REGION Network 17: IMMEDIATE STOP ALARMS / IMMEDIATE STOP
   RUNG wire#powerrail
      I_Contact( #CH_NOT_IN_SOFT_MODE )
      Not()
      { S7_GenerateENO := "TRUE" } Move(in := #DB_NUMBER, out1 => "DB440_MACHINE_ALARM_DECODING".GLOBAL_ALARMS_MACHINE.ALARM_DECODING)
      wire#w1
      { S7_Templates := "SrcType := Int" } EQ_Contact(in1 := #CHANNEL_NUM, in2 := 1)
      S_Coil( "DB440_MACHINE_ALARM_DECODING".ALARMS_UNIT_01.ST0_TRANSFER.IS_SEOC_ALARMS )
   END_RUNG
   RUNG wire#w1
      { S7_Templates := "SrcType := Int" } EQ_Contact(in1 := #CHANNEL_NUM, in2 := 2)
      S_Coil( "DB440_MACHINE_ALARM_DECODING".ALARMS_UNIT_01.ST3_CLADDING.IS_SEOC_ALARMS )
   END_RUNG
   RUNG wire#w1
      { S7_Templates := "SrcType := Int" } EQ_Contact(in1 := #CHANNEL_NUM, in2 := 3)
      S_Coil( "DB440_MACHINE_ALARM_DECODING".ALARMS_UNIT_01.ST4_CLEANING.IS_SEOC_ALARMS )
   END_RUNG
   RUNG wire#w1
      { S7_Templates := "SrcType := Int" } EQ_Contact(in1 := #CHANNEL_NUM, in2 := 4)
      S_Coil( "DB440_MACHINE_ALARM_DECODING".ALARMS_UNIT_02.ST0_TRANSFER.IS_SEOC_ALARMS )
   END_RUNG
   RUNG wire#w1
      { S7_Templates := "SrcType := Int" } EQ_Contact(in1 := #CHANNEL_NUM, in2 := 5)
      S_Coil( "DB440_MACHINE_ALARM_DECODING".ALARMS_UNIT_02.ST2_MEASURING.IS_SEOC_ALARMS )
   END_RUNG
   RUNG wire#w1
      { S7_Templates := "SrcType := Int" } EQ_Contact(in1 := #CHANNEL_NUM, in2 := 6)
      S_Coil( "DB440_MACHINE_ALARM_DECODING".ALARMS_UNIT_02.ST3_CLADDING.IS_SEOC_ALARMS )
   END_RUNG
   RUNG wire#w1
      { S7_Templates := "SrcType := Int" } EQ_Contact(in1 := #CHANNEL_NUM, in2 := 7)
      S_Coil( "DB440_MACHINE_ALARM_DECODING".ALARMS_UNIT_02.ST4_CLEANING.IS_SEOC_ALARMS )
   END_RUNG
   RUNG wire#w1
      { S7_Templates := "SrcType := Int" } EQ_Contact(in1 := #CHANNEL_NUM, in2 := 8)
      S_Coil( "DB440_MACHINE_ALARM_DECODING".ALARMS_UNIT_03.IS_SEOC_ALARMS )
   END_RUNG
   RUNG wire#w1
      { S7_Templates := "SrcType := Int" } EQ_Contact(in1 := #CHANNEL_NUM, in2 := 9)
      S_Coil( "DB440_MACHINE_ALARM_DECODING".ALARMS_UNIT_04.IS_SEOC_ALARMS )
   END_RUNG
   // the same network as SCL:
   // ENO of a box is taken as its EN; it also drops when the box reports an error
   #_w1 := NOT (NOT #CH_NOT_IN_SOFT_MODE);
   IF #_w1 THEN "DB440_MACHINE_ALARM_DECODING".GLOBAL_ALARMS_MACHINE.ALARM_DECODING := #DB_NUMBER; END_IF;
   IF #_w1 AND (#CHANNEL_NUM = 1) THEN
       "DB440_MACHINE_ALARM_DECODING".ALARMS_UNIT_01.ST0_TRANSFER.IS_SEOC_ALARMS := TRUE;
   END_IF;
   IF #_w1 AND (#CHANNEL_NUM = 2) THEN
       "DB440_MACHINE_ALARM_DECODING".ALARMS_UNIT_01.ST3_CLADDING.IS_SEOC_ALARMS := TRUE;
   END_IF;
   IF #_w1 AND (#CHANNEL_NUM = 3) THEN
       "DB440_MACHINE_ALARM_DECODING".ALARMS_UNIT_01.ST4_CLEANING.IS_SEOC_ALARMS := TRUE;
   END_IF;
   IF #_w1 AND (#CHANNEL_NUM = 4) THEN
       "DB440_MACHINE_ALARM_DECODING".ALARMS_UNIT_02.ST0_TRANSFER.IS_SEOC_ALARMS := TRUE;
   END_IF;
   IF #_w1 AND (#CHANNEL_NUM = 5) THEN
       "DB440_MACHINE_ALARM_DECODING".ALARMS_UNIT_02.ST2_MEASURING.IS_SEOC_ALARMS := TRUE;
   END_IF;
   IF #_w1 AND (#CHANNEL_NUM = 6) THEN
       "DB440_MACHINE_ALARM_DECODING".ALARMS_UNIT_02.ST3_CLADDING.IS_SEOC_ALARMS := TRUE;
   END_IF;
   IF #_w1 AND (#CHANNEL_NUM = 7) THEN
       "DB440_MACHINE_ALARM_DECODING".ALARMS_UNIT_02.ST4_CLEANING.IS_SEOC_ALARMS := TRUE;
   END_IF;
   IF #_w1 AND (#CHANNEL_NUM = 8) THEN
       "DB440_MACHINE_ALARM_DECODING".ALARMS_UNIT_03.IS_SEOC_ALARMS := TRUE;
   END_IF;
   IF #_w1 AND (#CHANNEL_NUM = 9) THEN
       "DB440_MACHINE_ALARM_DECODING".ALARMS_UNIT_04.IS_SEOC_ALARMS := TRUE;
   END_IF;
END_REGION

REGION Network 18: ANY AXIS OR CHANNEL BYPASSED
   RUNG wire#powerrail
      I_Contact( #NC_START_DUMMY_FOR_OPT )
      Not()
      S_Coil( "DB2100_GENERAL".ANY_AXIS_OR_CH_BYPASSED )
   END_RUNG
   // the same network as SCL:
   IF NOT (NOT #NC_START_DUMMY_FOR_OPT) THEN "DB2100_GENERAL".ANY_AXIS_OR_CH_BYPASSED := TRUE; END_IF;
END_REGION

REGION Network 19: PROGRAMMING ALARM
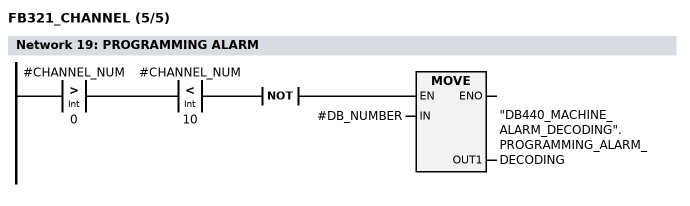
   RUNG wire#powerrail
      { S7_Templates := "SrcType := Int" } GT_Contact(in1 := #CHANNEL_NUM, in2 := 0)
      { S7_Templates := "SrcType := Int" } LT_Contact(in1 := #CHANNEL_NUM, in2 := 10)
      Not()
      Move(in := #DB_NUMBER, out1 => "DB440_MACHINE_ALARM_DECODING".PROGRAMMING_ALARM_DECODING)
   END_RUNG
   // the same network as SCL:
   IF NOT ((#CHANNEL_NUM > 0) AND (#CHANNEL_NUM < 10)) THEN
       "DB440_MACHINE_ALARM_DECODING".PROGRAMMING_ALARM_DECODING := #DB_NUMBER;
   END_IF;
END_REGION
END_FUNCTION_BLOCK

FUNCTION_BLOCK "FB331_M_CODE_EXTENDED"   // FB331, LAD
{ S7_Optimized_Access := 'FALSE' }
AUTHOR : ETXETAR
VERSION : 1.0
// stored: AutoNumber false, IsIECCheckEnabled false, SetENOAutomatically false, UDAEnableTagReadback false
   VAR_INPUT
      NC_Chan_Num_Chan : Int;   // Channel Number to monitoring
   END_VAR
   VAR DB_SPECIFIC
      INDEX : Int;
      M_code : Array[100..999] of Bool;   // EXTENDED M CODE
   END_VAR
   VAR_TEMP
      TEMP0 : Int;
      DB_Channel : Int;
      Inst_DB : Int;
   END_VAR
BEGIN

NETWORK
TITLE = READ DATA / Data block for monitoring channel

//DB from channel
      L     #NC_Chan_Num_Chan;
      +     20;
      T     #DB_Channel;
//set DB instance assigned to FB
      L     DINO;
      T     #Inst_DB;
      NOP   0;

NETWORK
TITLE = Reset signal from M Code
      LAR1  P#0.0;
      L     900;
R001: T     #TEMP0;
      OPN   DB [#Inst_DB];
      A     "M_ONE";
      R     DBX [AR1, P#4.0];
      +AR1  P#0.1;
      L     #TEMP0;
      LOOP  R001;

NETWORK
TITLE = Set signal from "M function 1 (DInt)"
      OPN   DB [#DB_Channel];
      A     %DBX58.0;  // M function 1 change
      JCN   END1;

      LAR1  P#0.0;
      L     100;
      T     #INDEX;
      L     900;
S001: T     #TEMP0;

      L     %DBW72;
      L     #INDEX;
      ==I;
      JC    Mse1;
      L     #INDEX;
      +     1;
      T     #INDEX;
      +AR1  P#0.1;
      L     #TEMP0;
      LOOP  S001;
      JU    END1;
Mse1: OPN   DB [#Inst_DB];
      S     DBX [AR1, P#4.0];

END1: NOP   0;

NETWORK
TITLE = Set signal from "M function 2 (DInt)"
      OPN   DB [#DB_Channel];
      A     %DBX58.1;  // M function 2 change
      JCN   END2;

      LAR1  P#0.0;
      L     100;
      T     #INDEX;
      L     900;
S002: T     #TEMP0;

      L     %DBW78;
      L     #INDEX;
      ==I;
      JC    Mse2;
      L     #INDEX;
      +     1;
      T     #INDEX;
      +AR1  P#0.1;
      L     #TEMP0;
      LOOP  S002;
      JU    END2;
Mse2: OPN   DB [#Inst_DB];
      S     DBX [AR1, P#4.0];

END2: NOP   0;

NETWORK
TITLE = Set signal from "M function 3 (DInt)"
      OPN   DB [#DB_Channel];
      A     %DBX58.2;  // M function 3 change
      JCN   END3;

      LAR1  P#0.0;
      L     100;
      T     #INDEX;
      L     900;
S003: T     #TEMP0;

      L     %DBW84;
      L     #INDEX;
      ==I;
      JC    Mse3;
      L     #INDEX;
      +     1;
      T     #INDEX;
      +AR1  P#0.1;
      L     #TEMP0;
      LOOP  S003;
      JU    END3;
Mse3: OPN   DB [#Inst_DB];
      S     DBX [AR1, P#4.0];

END3: NOP   0;

NETWORK
TITLE = Set signal from "M function 4 (DInt)"
      OPN   DB [#DB_Channel];
      A     %DBX58.3;  // M function 4 change
      JCN   END4;

      LAR1  P#0.0;
      L     100;
      T     #INDEX;
      L     900;
S004: T     #TEMP0;

      L     %DBW90;
      L     #INDEX;
      ==I;
      JC    Mse4;
      L     #INDEX;
      +     1;
      T     #INDEX;
      +AR1  P#0.1;
      L     #TEMP0;
      LOOP  S004;
      JU    END4;
Mse4: OPN   DB [#Inst_DB];
      S     DBX [AR1, P#4.0];

END4: NOP   0;

NETWORK
TITLE = Set signal from "M function 5 (DInt)"
      OPN   DB [#DB_Channel];
      A     %DBX58.4;  // M function 5 change
      JCN   END5;

      LAR1  P#0.0;
      L     100;
      T     #INDEX;
      L     900;
S005: T     #TEMP0;

      L     %DBW96;
      L     #INDEX;
      ==I;
      JC    Mse5;
      L     #INDEX;
      +     1;
      T     #INDEX;
      +AR1  P#0.1;
      L     #TEMP0;
      LOOP  S005;
      JU    END5;
Mse5: OPN   DB [#Inst_DB];
      S     DBX [AR1, P#4.0];

END5: NOP   0;

NETWORK
TITLE = 
      BE;

END_FUNCTION_BLOCK

FUNCTION "FC1100_MAIN_SEQUENCES" : Void   // FC1100, LAD
{ S7_Optimized_Access := 'FALSE' }
AUTHOR : ETXETAR
VERSION : 1.0
// stored: AutoNumber false, IsIECCheckEnabled false, SetENOAutomatically false, UDAEnableTagReadback false
   VAR_TEMP
      STEP_NUMBER : Int;
   END_VAR
BEGIN

REGION Network 1: CALL FC1103 MACHINING TWIN TWIN+
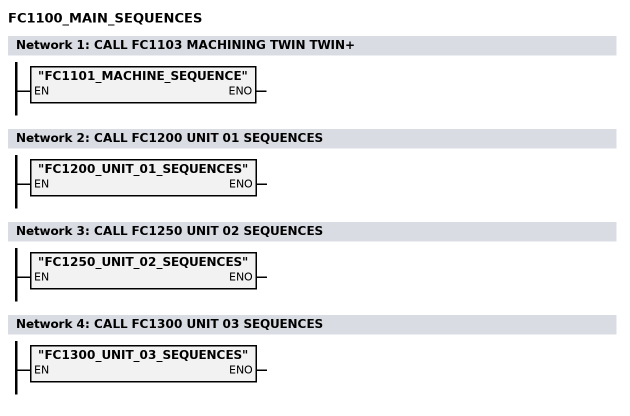
   RUNG wire#powerrail
      "FC1101_MACHINE_SEQUENCE"()
   END_RUNG
   // the same network as SCL:
   "FC1101_MACHINE_SEQUENCE"();
END_REGION

REGION Network 2: CALL FC1200 UNIT 01 SEQUENCES
   RUNG wire#powerrail
      "FC1200_UNIT_01_SEQUENCES"()
   END_RUNG
   // the same network as SCL:
   "FC1200_UNIT_01_SEQUENCES"();
END_REGION

REGION Network 3: CALL FC1250 UNIT 02 SEQUENCES
   RUNG wire#powerrail
      "FC1250_UNIT_02_SEQUENCES"()
   END_RUNG
   // the same network as SCL:
   "FC1250_UNIT_02_SEQUENCES"();
END_REGION

REGION Network 4: CALL FC1300 UNIT 03 SEQUENCES
   RUNG wire#powerrail
      "FC1300_UNIT_03_SEQUENCES"()
   END_RUNG
   // the same network as SCL:
   "FC1300_UNIT_03_SEQUENCES"();
END_REGION
END_FUNCTION

FUNCTION "FC1400_SERVICES_GENERAL" : Void   // FC1400, LAD
{ S7_Optimized_Access := 'FALSE' }
AUTHOR : ETXETAR
VERSION : 1.0
// stored: AutoNumber false, IsIECCheckEnabled false, SetENOAutomatically false, UDAEnableTagReadback false
BEGIN

REGION Network 1: CALL FC1401_UTILITY_SKIDS
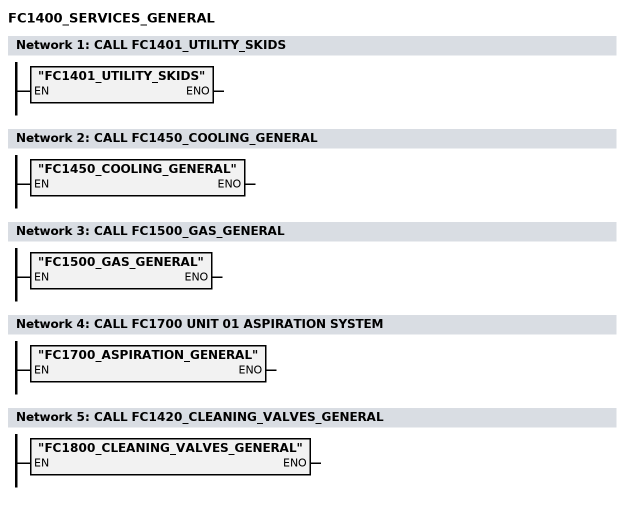
   RUNG wire#powerrail
      "FC1401_UTILITY_SKIDS"()
   END_RUNG
   // the same network as SCL:
   "FC1401_UTILITY_SKIDS"();
END_REGION

REGION Network 2: CALL FC1450_COOLING_GENERAL
   RUNG wire#powerrail
      "FC1450_COOLING_GENERAL"()
   END_RUNG
   // the same network as SCL:
   "FC1450_COOLING_GENERAL"();
END_REGION

REGION Network 3: CALL FC1500_GAS_GENERAL
   RUNG wire#powerrail
      "FC1500_GAS_GENERAL"()
   END_RUNG
   // the same network as SCL:
   "FC1500_GAS_GENERAL"();
END_REGION

REGION Network 4: CALL FC1700 UNIT 01 ASPIRATION SYSTEM
   RUNG wire#powerrail
      "FC1700_ASPIRATION_GENERAL"()
   END_RUNG
   // the same network as SCL:
   "FC1700_ASPIRATION_GENERAL"();
END_REGION

REGION Network 5: CALL FC1420_CLEANING_VALVES_GENERAL
   RUNG wire#powerrail
      "FC1800_CLEANING_VALVES_GENERAL"()
   END_RUNG
   // the same network as SCL:
   "FC1800_CLEANING_VALVES_GENERAL"();
END_REGION
END_FUNCTION

FUNCTION "FC1401_UTILITY_SKIDS" : Void   // FC1401, LAD
{ S7_Optimized_Access := 'TRUE' }
VERSION : 0.1
// stored: AutoNumber false, IsIECCheckEnabled false, SetENOAutomatically false, UDAEnableTagReadback false
   VAR CONSTANT
      FC_NUMBER : DInt := 1401;
   END_VAR
   VAR_TEMP   // added for the SCL form of the ladder/FBD networks
      _w1 : Bool;
      _w2 : Bool;
   END_VAR
BEGIN

REGION Network 1: <<<<<<<<<<<<<<<<<<<< PNEUMATIC SYSTEM >>>>>>>>>>>>>>>>>>>>
END_REGION

REGION Network 2: CALL FB1401 PNEUMATIC SYSTEM
   // 2#0000_0001 OPTIONS 0 BIT 0 PRESSURE PRESENT OPTION
   // 2#0000_0010 OPTIONS 0 BIT 1 CONNECTION SENSOR 1 OPTION
   // 2#0000_0100 OPTIONS 0 BIT 2 CONNECTION SENSOR 2 OPTION
   // 2#0000_1000 OPTIONS 0 BIT 3 DRIVE UNBLOCKED OPTION
   // 2#0001_0000 OPTIONS 0 BIT 4 PRESSURIZED OPTION
   // 2#0010_0000 OPTIONS 0 BIT 5 UNIT 01 GRIPPER PRESSURIZED OPTION
   // 2#0100_0000 OPTIONS 0 BIT 6 UNIT 01 LABERINT PRESSURIZED OPTION
   // 2#1000_0000 OPTIONS 0 BIT 7 UNIT 01 UPPER TABLE PRESSURIZED OPTION
   // 
   // 2#0000_0001 OPTIONS 1 BIT 0 UNIT 01 LOWER TABLE PRESSURIZED OPTION
   // 2#0000_0010 OPTIONS 1 BIT 1 UNIT 01 AXIS X CART PRESSURIZED OPTION
   // 2#0000_0100 OPTIONS 1 BIT 2 UNIT 01 STATION 3 MEASURMENT UNIT PRESSURIZED OPTION
   // 2#0000_1000 OPTIONS 1 BIT 3 UNIT 01 STATION 4 MEASURMENT UNIT PRESSURIZED OPTION
   // 2#0001_0000 OPTIONS 1 BIT 4 UNIT 02 GRIPPER PRESSURIZEDPRESSURIZED OPTION
   // 2#0010_0000 OPTIONS 1 BIT 5 UNIT 02 LABERINT PRESSURIZED OPTION
   // 2#0100_0000 OPTIONS 1 BIT 6 UNIT 02 UPPER TABLE PRESSURIZED OPTION
   // 2#1000_0000 OPTIONS 1 BIT 7 UNIT 02 LOWER TABLE PRESSURIZED OPTION
   // 
   // 2#0000_0001 OPTIONS 2 BIT 0 UNIT 02 AXIS X CART PRESSURIZED OPTION
   // 2#0000_0010 OPTIONS 2 BIT 1 UNIT 02 STATION 3 MEASURMENT UNIT PRESSURIZED OPTION
   // 2#0000_0100 OPTIONS 2 BIT 2 UNIT 02 STATION 4 MEASURMENT UNIT PRESSURIZED OPTION
   // 2#0000_1000 OPTIONS 2 BIT 3 INPUT FLOW  OPTION
   // 2#0001_0000 OPTIONS 2 BIT 4 INPUT TEMPERATURE OPTION
   // 2#0010_0000 OPTIONS 2 BIT 5 SPARE OPTION
   // 2#0100_0000 OPTIONS 2 BIT 6 SPARE OPTION
   // 2#1000_0000 OPTIONS 2 BIT 7 SPARE OPTION
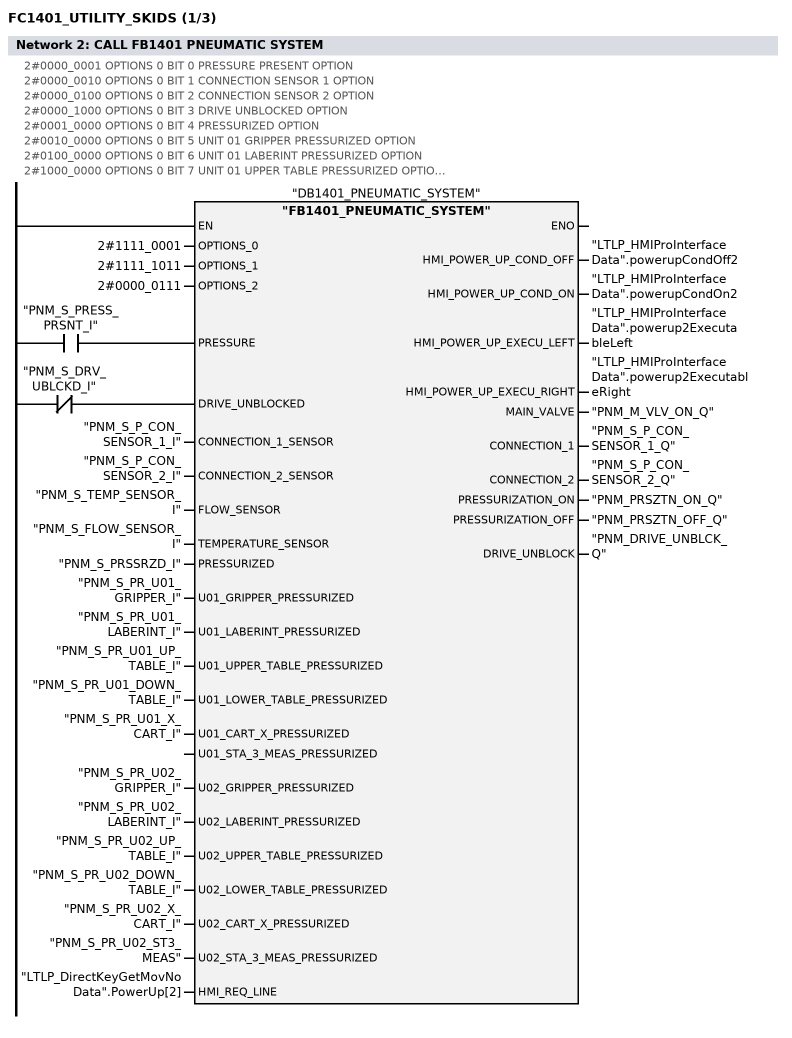
   RUNG wire#powerrail
      "DB1401_PNEUMATIC_SYSTEM"(PRESSURE := wire#w1, DRIVE_UNBLOCKED := wire#w2, OPTIONS_0 := 2#1111_0001, OPTIONS_1 := 2#1111_1011, OPTIONS_2 := 2#0000_0111, CONNECTION_1_SENSOR := "PNM_S_P_CON_SENSOR_1_I", CONNECTION_2_SENSOR := "PNM_S_P_CON_SENSOR_2_I", FLOW_SENSOR := "PNM_S_TEMP_SENSOR_I", TEMPERATURE_SENSOR := "PNM_S_FLOW_SENSOR_I", PRESSURIZED := "PNM_S_PRSSRZD_I", U01_GRIPPER_PRESSURIZED := "PNM_S_PR_U01_GRIPPER_I", U01_LABERINT_PRESSURIZED := "PNM_S_PR_U01_LABERINT_I", U01_UPPER_TABLE_PRESSURIZED := "PNM_S_PR_U01_UP_TABLE_I", U01_LOWER_TABLE_PRESSURIZED := "PNM_S_PR_U01_DOWN_TABLE_I", U01_CART_X_PRESSURIZED := "PNM_S_PR_U01_X_CART_I", U01_STA_3_MEAS_PRESSURIZED :=, U02_GRIPPER_PRESSURIZED := "PNM_S_PR_U02_GRIPPER_I", U02_LABERINT_PRESSURIZED := "PNM_S_PR_U02_LABERINT_I", U02_UPPER_TABLE_PRESSURIZED := "PNM_S_PR_U02_UP_TABLE_I", U02_LOWER_TABLE_PRESSURIZED := "PNM_S_PR_U02_DOWN_TABLE_I", U02_CART_X_PRESSURIZED := "PNM_S_PR_U02_X_CART_I", U02_STA_3_MEAS_PRESSURIZED := "PNM_S_PR_U02_ST3_MEAS", HMI_REQ_LINE := "LTLP_DirectKeyGetMovNoData".PowerUp[2], HMI_POWER_UP_COND_OFF => "LTLP_HMIProInterfaceData".powerupCondOff2, HMI_POWER_UP_COND_ON => "LTLP_HMIProInterfaceData".powerupCondOn2, HMI_POWER_UP_EXECU_LEFT => "LTLP_HMIProInterfaceData".powerup2ExecutableLeft, HMI_POWER_UP_EXECU_RIGHT => "LTLP_HMIProInterfaceData".powerup2ExecutableRight, MAIN_VALVE => "PNM_M_VLV_ON_Q", CONNECTION_1 => "PNM_S_P_CON_SENSOR_1_Q", CONNECTION_2 => "PNM_S_P_CON_SENSOR_2_Q", PRESSURIZATION_ON => "PNM_PRSZTN_ON_Q", PRESSURIZATION_OFF => "PNM_PRSZTN_OFF_Q", DRIVE_UNBLOCK => "PNM_DRIVE_UNBLCK_Q")
   END_RUNG
   RUNG wire#powerrail
      Contact( "PNM_S_PRESS_PRSNT_I" )
   END_RUNG wire#w1
   RUNG wire#powerrail
      I_Contact( "PNM_S_DRV_UBLCKD_I" )
   END_RUNG wire#w2
   // the same network as SCL:
   "DB1401_PNEUMATIC_SYSTEM"(OPTIONS_0 := 2#1111_0001,   // "FB1401_PNEUMATIC_SYSTEM"
                           OPTIONS_1 := 2#1111_1011,
                           OPTIONS_2 := 2#0000_0111,
                           PRESSURE := "PNM_S_PRESS_PRSNT_I",
                           DRIVE_UNBLOCKED := NOT "PNM_S_DRV_UBLCKD_I",
                           CONNECTION_1_SENSOR := "PNM_S_P_CON_SENSOR_1_I",
                           CONNECTION_2_SENSOR := "PNM_S_P_CON_SENSOR_2_I",
                           FLOW_SENSOR := "PNM_S_TEMP_SENSOR_I",
                           TEMPERATURE_SENSOR := "PNM_S_FLOW_SENSOR_I",
                           PRESSURIZED := "PNM_S_PRSSRZD_I",
                           U01_GRIPPER_PRESSURIZED := "PNM_S_PR_U01_GRIPPER_I",
                           U01_LABERINT_PRESSURIZED := "PNM_S_PR_U01_LABERINT_I",
                           U01_UPPER_TABLE_PRESSURIZED := "PNM_S_PR_U01_UP_TABLE_I",
                           U01_LOWER_TABLE_PRESSURIZED := "PNM_S_PR_U01_DOWN_TABLE_I",
                           U01_CART_X_PRESSURIZED := "PNM_S_PR_U01_X_CART_I",
                           U02_GRIPPER_PRESSURIZED := "PNM_S_PR_U02_GRIPPER_I",
                           U02_LABERINT_PRESSURIZED := "PNM_S_PR_U02_LABERINT_I",
                           U02_UPPER_TABLE_PRESSURIZED := "PNM_S_PR_U02_UP_TABLE_I",
                           U02_LOWER_TABLE_PRESSURIZED := "PNM_S_PR_U02_DOWN_TABLE_I",
                           U02_CART_X_PRESSURIZED := "PNM_S_PR_U02_X_CART_I",
                           U02_STA_3_MEAS_PRESSURIZED := "PNM_S_PR_U02_ST3_MEAS",
                           HMI_REQ_LINE := "LTLP_DirectKeyGetMovNoData".PowerUp[2],
                           HMI_POWER_UP_COND_OFF => "LTLP_HMIProInterfaceData".powerupCondOff2,
                           HMI_POWER_UP_COND_ON => "LTLP_HMIProInterfaceData".powerupCondOn2,
                           HMI_POWER_UP_EXECU_LEFT => "LTLP_HMIProInterfaceData".powerup2ExecutableLeft,
                           HMI_POWER_UP_EXECU_RIGHT => "LTLP_HMIProInterfaceData".powerup2ExecutableRight,
                           MAIN_VALVE => "PNM_M_VLV_ON_Q",
                           CONNECTION_1 => "PNM_S_P_CON_SENSOR_1_Q",
                           CONNECTION_2 => "PNM_S_P_CON_SENSOR_2_Q",
                           PRESSURIZATION_ON => "PNM_PRSZTN_ON_Q",
                           PRESSURIZATION_OFF => "PNM_PRSZTN_OFF_Q",
                           DRIVE_UNBLOCK => "PNM_DRIVE_UNBLCK_Q");
END_REGION

REGION Network 3: <<<<<<<<<<<<<<<<<<<< LUBRICATION SYSTEM >>>>>>>>>>>>>>>>>>>>
END_REGION

REGION Network 4: CALL FB1421 PROGRESSIVE LUBRICATION WITH GREASE
   // 2#0000_0001 OPTIONS 0 BIT 0 CIRCUIT BREAKER OPTION
   // 2#0000_0010 OPTIONS 0 BIT 1 LOW LEVEL ALARM OPTION
   // 2#0000_0100 OPTIONS 0 BIT 2 OVERPRESSURE ALARM OPTION
   // 2#0000_1000 OPTIONS 0 BIT 3 LUBRICATION BY TIME VALVE 1 AXIS X OPTION
   // 2#0001_0000 OPTIONS 0 BIT 4 LUBRICATION BY TIME VALVE 2 AXIS Z OPTION
   // 2#0010_0000 OPTIONS 0 BIT 5 LUBRICATION BY TIME VALVE 3 TURN UNIT OPTION
   // 2#0100_0000 OPTIONS 0 BIT 6 LUBRICATION BY TIME VALVE 4 OPTION
   // 2#1000_0000 OPTIONS 0 BIT 7 LUBRICATION DONE VALVE 1  AXIS X OPTION
   // 
   // 2#0000_0001 OPTIONS 1 BIT 0 LUBRICATION DONE VALVE 2 AXIS Z OPTION
   // 2#0000_0010 OPTIONS 1 BIT 1 LUBRICATION DONE VALVE 3 TURN UNIT OPTION
   // 2#0000_0100 OPTIONS 1 BIT 2 LUBRICATION DONE VALVE 4 OPTION
   // 2#0000_1000 OPTIONS 1 BIT 3 LUBRICATION DONE VALVE 5 OPTION
   // 2#0001_0000 OPTIONS 1 BIT 4 LUBRICATION DONE VALVE 6 OPTION
   // 2#0010_0000 OPTIONS 1 BIT 5 LUBRICATION DONE VALVE 7 OPTION
   // 2#0100_0000 OPTIONS 1 BIT 6 LUBRICATION DONE VALVE 8 OPTION
   // 2#1000_0000 OPTIONS 1 BIT 7 LUBRICATION DONE VALVE 9 OPTION
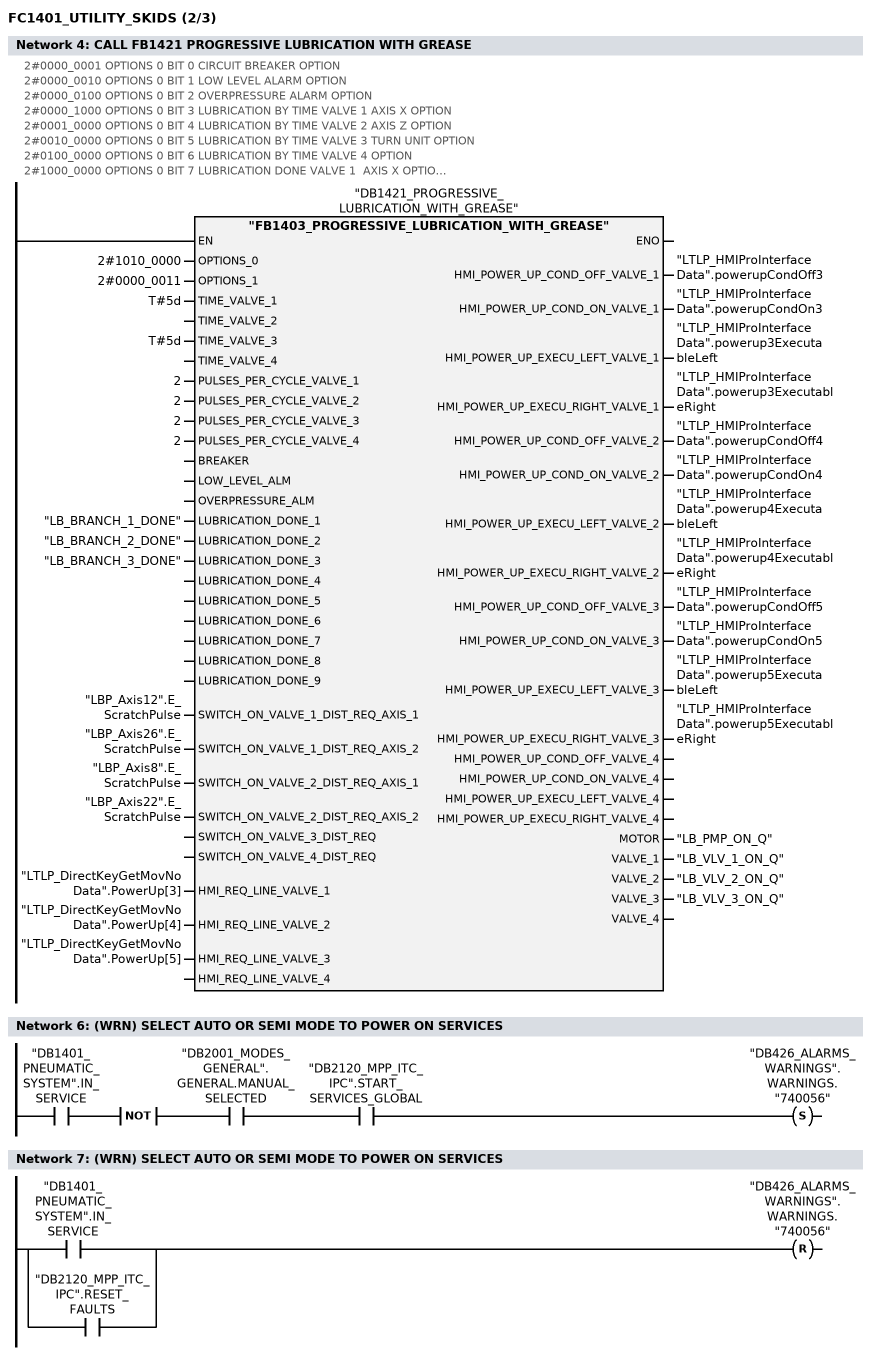
   RUNG wire#powerrail
      "DB1421_PROGRESSIVE_LUBRICATION_WITH_GREASE"(OPTIONS_0 := 2#1010_0000, OPTIONS_1 := 2#0000_0011, TIME_VALVE_1 := T#5d, TIME_VALVE_2 :=, TIME_VALVE_3 := T#5d, TIME_VALVE_4 :=, PULSES_PER_CYCLE_VALVE_1 := 2, PULSES_PER_CYCLE_VALVE_2 := 2, PULSES_PER_CYCLE_VALVE_3 := 2, PULSES_PER_CYCLE_VALVE_4 := 2, BREAKER :=, LOW_LEVEL_ALM :=, OVERPRESSURE_ALM :=, LUBRICATION_DONE_1 := "LB_BRANCH_1_DONE", LUBRICATION_DONE_2 := "LB_BRANCH_2_DONE", LUBRICATION_DONE_3 := "LB_BRANCH_3_DONE", LUBRICATION_DONE_4 :=, LUBRICATION_DONE_5 :=, LUBRICATION_DONE_6 :=, LUBRICATION_DONE_7 :=, LUBRICATION_DONE_8 :=, LUBRICATION_DONE_9 :=, SWITCH_ON_VALVE_1_DIST_REQ_AXIS_1 := "LBP_Axis12".E_ScratchPulse, SWITCH_ON_VALVE_1_DIST_REQ_AXIS_2 := "LBP_Axis26".E_ScratchPulse, SWITCH_ON_VALVE_2_DIST_REQ_AXIS_1 := "LBP_Axis8".E_ScratchPulse, SWITCH_ON_VALVE_2_DIST_REQ_AXIS_2 := "LBP_Axis22".E_ScratchPulse, SWITCH_ON_VALVE_3_DIST_REQ :=, SWITCH_ON_VALVE_4_DIST_REQ :=, HMI_REQ_LINE_VALVE_1 := "LTLP_DirectKeyGetMovNoData".PowerUp[3], HMI_REQ_LINE_VALVE_2 := "LTLP_DirectKeyGetMovNoData".PowerUp[4], HMI_REQ_LINE_VALVE_3 := "LTLP_DirectKeyGetMovNoData".PowerUp[5], HMI_REQ_LINE_VALVE_4 :=, HMI_POWER_UP_COND_OFF_VALVE_1 => "LTLP_HMIProInterfaceData".powerupCondOff3, HMI_POWER_UP_COND_ON_VALVE_1 => "LTLP_HMIProInterfaceData".powerupCondOn3, HMI_POWER_UP_EXECU_LEFT_VALVE_1 => "LTLP_HMIProInterfaceData".powerup3ExecutableLeft, HMI_POWER_UP_EXECU_RIGHT_VALVE_1 => "LTLP_HMIProInterfaceData".powerup3ExecutableRight, HMI_POWER_UP_COND_OFF_VALVE_2 => "LTLP_HMIProInterfaceData".powerupCondOff4, HMI_POWER_UP_COND_ON_VALVE_2 => "LTLP_HMIProInterfaceData".powerupCondOn4, HMI_POWER_UP_EXECU_LEFT_VALVE_2 => "LTLP_HMIProInterfaceData".powerup4ExecutableLeft, HMI_POWER_UP_EXECU_RIGHT_VALVE_2 => "LTLP_HMIProInterfaceData".powerup4ExecutableRight, HMI_POWER_UP_COND_OFF_VALVE_3 => "LTLP_HMIProInterfaceData".powerupCondOff5, HMI_POWER_UP_COND_ON_VALVE_3 => "LTLP_HMIProInterfaceData".powerupCondOn5, HMI_POWER_UP_EXECU_LEFT_VALVE_3 => "LTLP_HMIProInterfaceData".powerup5ExecutableLeft, HMI_POWER_UP_EXECU_RIGHT_VALVE_3 => "LTLP_HMIProInterfaceData".powerup5ExecutableRight, HMI_POWER_UP_COND_OFF_VALVE_4 =>, HMI_POWER_UP_COND_ON_VALVE_4 =>, HMI_POWER_UP_EXECU_LEFT_VALVE_4 =>, HMI_POWER_UP_EXECU_RIGHT_VALVE_4 =>, MOTOR => "LB_PMP_ON_Q", VALVE_1 => "LB_VLV_1_ON_Q", VALVE_2 => "LB_VLV_2_ON_Q", VALVE_3 => "LB_VLV_3_ON_Q", VALVE_4 =>)
   END_RUNG
   // the same network as SCL:
   "DB1421_PROGRESSIVE_LUBRICATION_WITH_GREASE"(OPTIONS_0 := 2#1010_0000,   // "FB1403_PROGRESSIVE_LUBRICATION_WITH_GREASE"
                           OPTIONS_1 := 2#0000_0011,
                           TIME_VALVE_1 := T#5d,
                           TIME_VALVE_3 := T#5d,
                           PULSES_PER_CYCLE_VALVE_1 := 2,
                           PULSES_PER_CYCLE_VALVE_2 := 2,
                           PULSES_PER_CYCLE_VALVE_3 := 2,
                           PULSES_PER_CYCLE_VALVE_4 := 2,
                           LUBRICATION_DONE_1 := "LB_BRANCH_1_DONE",
                           LUBRICATION_DONE_2 := "LB_BRANCH_2_DONE",
                           LUBRICATION_DONE_3 := "LB_BRANCH_3_DONE",
                           SWITCH_ON_VALVE_1_DIST_REQ_AXIS_1 := "LBP_Axis12".E_ScratchPulse,
                           SWITCH_ON_VALVE_1_DIST_REQ_AXIS_2 := "LBP_Axis26".E_ScratchPulse,
                           SWITCH_ON_VALVE_2_DIST_REQ_AXIS_1 := "LBP_Axis8".E_ScratchPulse,
                           SWITCH_ON_VALVE_2_DIST_REQ_AXIS_2 := "LBP_Axis22".E_ScratchPulse,
                           HMI_REQ_LINE_VALVE_1 := "LTLP_DirectKeyGetMovNoData".PowerUp[3],
                           HMI_REQ_LINE_VALVE_2 := "LTLP_DirectKeyGetMovNoData".PowerUp[4],
                           HMI_REQ_LINE_VALVE_3 := "LTLP_DirectKeyGetMovNoData".PowerUp[5],
                           HMI_POWER_UP_COND_OFF_VALVE_1 => "LTLP_HMIProInterfaceData".powerupCondOff3,
                           HMI_POWER_UP_COND_ON_VALVE_1 => "LTLP_HMIProInterfaceData".powerupCondOn3,
                           HMI_POWER_UP_EXECU_LEFT_VALVE_1 => "LTLP_HMIProInterfaceData".powerup3ExecutableLeft,
                           HMI_POWER_UP_EXECU_RIGHT_VALVE_1 => "LTLP_HMIProInterfaceData".powerup3ExecutableRight,
                           HMI_POWER_UP_COND_OFF_VALVE_2 => "LTLP_HMIProInterfaceData".powerupCondOff4,
                           HMI_POWER_UP_COND_ON_VALVE_2 => "LTLP_HMIProInterfaceData".powerupCondOn4,
                           HMI_POWER_UP_EXECU_LEFT_VALVE_2 => "LTLP_HMIProInterfaceData".powerup4ExecutableLeft,
                           HMI_POWER_UP_EXECU_RIGHT_VALVE_2 => "LTLP_HMIProInterfaceData".powerup4ExecutableRight,
                           HMI_POWER_UP_COND_OFF_VALVE_3 => "LTLP_HMIProInterfaceData".powerupCondOff5,
                           HMI_POWER_UP_COND_ON_VALVE_3 => "LTLP_HMIProInterfaceData".powerupCondOn5,
                           HMI_POWER_UP_EXECU_LEFT_VALVE_3 => "LTLP_HMIProInterfaceData".powerup5ExecutableLeft,
                           HMI_POWER_UP_EXECU_RIGHT_VALVE_3 => "LTLP_HMIProInterfaceData".powerup5ExecutableRight,
                           MOTOR => "LB_PMP_ON_Q",
                           VALVE_1 => "LB_VLV_1_ON_Q",
                           VALVE_2 => "LB_VLV_2_ON_Q",
                           VALVE_3 => "LB_VLV_3_ON_Q");
END_REGION

REGION Network 5: <<<<<<<<<<<<<<<<<<<< GENERAL WARNINGS >>>>>>>>>>>>>>>>>>>>
END_REGION

REGION Network 6: (WRN) SELECT AUTO OR SEMI MODE TO POWER ON SERVICES
   RUNG wire#powerrail
      Contact( "DB1401_PNEUMATIC_SYSTEM".IN_SERVICE )
      Not()
      Contact( "DB2001_MODES_GENERAL".GENERAL.MANUAL_SELECTED )
      Contact( "DB2120_MPP_ITC_IPC".START_SERVICES_GLOBAL )
      S_Coil( "DB426_ALARMS_WARNINGS".WARNINGS."740056" )
   END_RUNG
   // the same network as SCL:
   IF NOT "DB1401_PNEUMATIC_SYSTEM".IN_SERVICE AND "DB2001_MODES_GENERAL".GENERAL.MANUAL_SELECTED AND "DB2120_MPP_ITC_IPC".START_SERVICES_GLOBAL THEN
       "DB426_ALARMS_WARNINGS".WARNINGS."740056" := TRUE;
   END_IF;
END_REGION

REGION Network 7: (WRN) SELECT AUTO OR SEMI MODE TO POWER ON SERVICES
   RUNG wire#powerrail
      Contact( "DB1401_PNEUMATIC_SYSTEM".IN_SERVICE )
      wire#w1
      R_Coil( "DB426_ALARMS_WARNINGS".WARNINGS."740056" )
   END_RUNG
   RUNG wire#powerrail
      Contact( "DB2120_MPP_ITC_IPC".RESET_FAULTS )
   END_RUNG wire#w1
   // the same network as SCL:
   IF "DB1401_PNEUMATIC_SYSTEM".IN_SERVICE OR "DB2120_MPP_ITC_IPC".RESET_FAULTS THEN
       "DB426_ALARMS_WARNINGS".WARNINGS."740056" := FALSE;
   END_IF;
END_REGION

REGION Network 8: WARNINGS
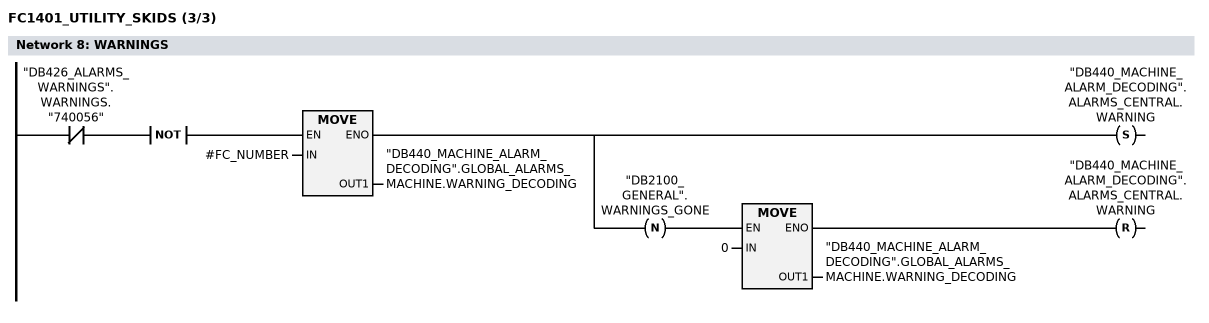
   RUNG wire#powerrail
      I_Contact( "DB426_ALARMS_WARNINGS".WARNINGS."740056" )
      Not()
      { S7_GenerateENO := "TRUE" } Move(in := #FC_NUMBER, out1 => "DB440_MACHINE_ALARM_DECODING".GLOBAL_ALARMS_MACHINE.WARNING_DECODING)
      wire#w1
      S_Coil( "DB440_MACHINE_ALARM_DECODING".ALARMS_CENTRAL.WARNING )
   END_RUNG
   RUNG wire#w1
      N_Trig( "DB2100_GENERAL".WARNINGS_GONE )
      { S7_GenerateENO := "TRUE" } Move(in := 0, out1 => "DB440_MACHINE_ALARM_DECODING".GLOBAL_ALARMS_MACHINE.WARNING_DECODING)
      R_Coil( "DB440_MACHINE_ALARM_DECODING".ALARMS_CENTRAL.WARNING )
   END_RUNG
   // the same network as SCL:
   // ENO of a box is taken as its EN; it also drops when the box reports an error
   #_w1 := NOT (NOT "DB426_ALARMS_WARNINGS".WARNINGS."740056");
   IF #_w1 THEN
       "DB440_MACHINE_ALARM_DECODING".GLOBAL_ALARMS_MACHINE.WARNING_DECODING := #FC_NUMBER;
       "DB440_MACHINE_ALARM_DECODING".ALARMS_CENTRAL.WARNING := TRUE;
   END_IF;
   #_w2 := NOT #_w1 AND "DB2100_GENERAL".WARNINGS_GONE;   // falling edge
   "DB2100_GENERAL".WARNINGS_GONE := #_w1;
   IF #_w2 THEN
       "DB440_MACHINE_ALARM_DECODING".GLOBAL_ALARMS_MACHINE.WARNING_DECODING := 0;
       "DB440_MACHINE_ALARM_DECODING".ALARMS_CENTRAL.WARNING := FALSE;
   END_IF;
END_REGION
END_FUNCTION

FUNCTION "FC1450_COOLING_GENERAL" : Void   // FC1450, LAD
{ S7_Optimized_Access := 'TRUE' }
VERSION : 0.1
// stored: AutoNumber false, IsIECCheckEnabled false, SetENOAutomatically false, UDAEnableTagReadback false
BEGIN

REGION Network 1: CALL FC1451_MACHINE_MAIN_COOLING_SYSTEM
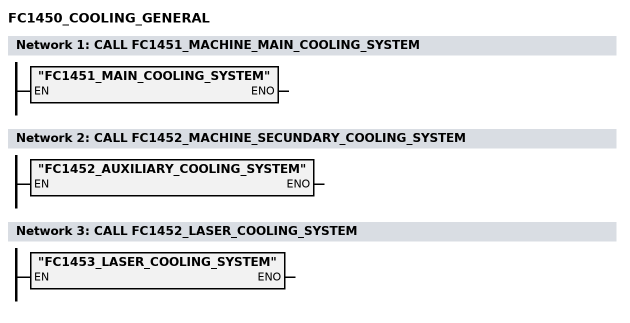
   RUNG wire#powerrail
      "FC1451_MAIN_COOLING_SYSTEM"()
   END_RUNG
   // the same network as SCL:
   "FC1451_MAIN_COOLING_SYSTEM"();
END_REGION

REGION Network 2: CALL FC1452_MACHINE_SECUNDARY_COOLING_SYSTEM
   RUNG wire#powerrail
      "FC1452_AUXILIARY_COOLING_SYSTEM"()
   END_RUNG
   // the same network as SCL:
   "FC1452_AUXILIARY_COOLING_SYSTEM"();
END_REGION

REGION Network 3: CALL FC1452_LASER_COOLING_SYSTEM
   RUNG wire#powerrail
      "FC1453_LASER_COOLING_SYSTEM"()
   END_RUNG
   // the same network as SCL:
   "FC1453_LASER_COOLING_SYSTEM"();
END_REGION
END_FUNCTION

FUNCTION "FC1500_GAS_GENERAL" : Void   // FC1500, LAD
{ S7_Optimized_Access := 'TRUE' }
VERSION : 0.1
// stored: AutoNumber false, IsIECCheckEnabled false, SetENOAutomatically false, UDAEnableTagReadback false
BEGIN

REGION Network 1: CALL FC1501_MAIN_GAS_VALVE
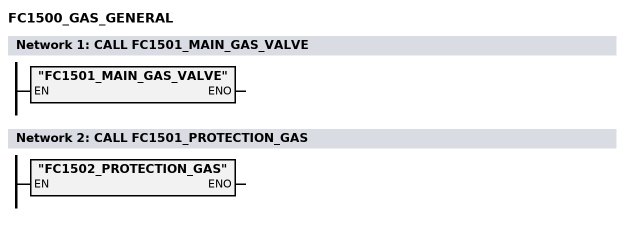
   RUNG wire#powerrail
      "FC1501_MAIN_GAS_VALVE"()
   END_RUNG
   // the same network as SCL:
   "FC1501_MAIN_GAS_VALVE"();
END_REGION

REGION Network 2: CALL FC1501_PROTECTION_GAS
   RUNG wire#powerrail
      "FC1502_PROTECTION_GAS"()
   END_RUNG
   // the same network as SCL:
   "FC1502_PROTECTION_GAS"();
END_REGION
END_FUNCTION

FUNCTION "FC1700_ASPIRATION_GENERAL" : Void   // FC1700, LAD
{ S7_Optimized_Access := 'FALSE' }
AUTHOR : ETXETAR
VERSION : 1.0
// stored: AutoNumber false, IsIECCheckEnabled false, SetENOAutomatically false, UDAEnableTagReadback false
   VAR CONSTANT
      FC_NUMBER : DInt := 1700;
   END_VAR
BEGIN

REGION Network 1: CALL FC1701_KELLER_ASPIRATION_CONTROL
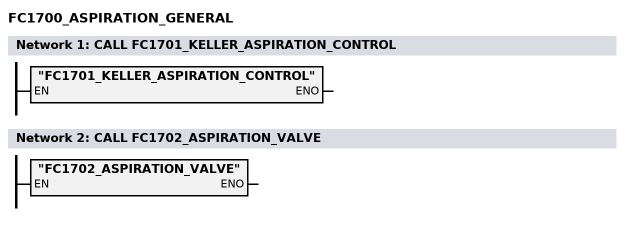
   RUNG wire#powerrail
      "FC1701_KELLER_ASPIRATION_CONTROL"()
   END_RUNG
   // the same network as SCL:
   "FC1701_KELLER_ASPIRATION_CONTROL"();
END_REGION

REGION Network 2: CALL FC1702_ASPIRATION_VALVE
   RUNG wire#powerrail
      "FC1702_ASPIRATION_VALVE"()
   END_RUNG
   // the same network as SCL:
   "FC1702_ASPIRATION_VALVE"();
END_REGION
END_FUNCTION

FUNCTION "FC1800_CLEANING_VALVES_GENERAL" : Void   // FC1800, LAD
{ S7_Optimized_Access := 'TRUE' }
VERSION : 0.1
// stored: AutoNumber false, IsIECCheckEnabled false, SetENOAutomatically false, UDAEnableTagReadback false
BEGIN

REGION Network 1: <<<<<<<<<<<<<<<<<<<< CLEANING VALVES >>>>>>>>>>>>>>>>>>>>
END_REGION

REGION Network 2: UNIT 01CLEANING VALVE
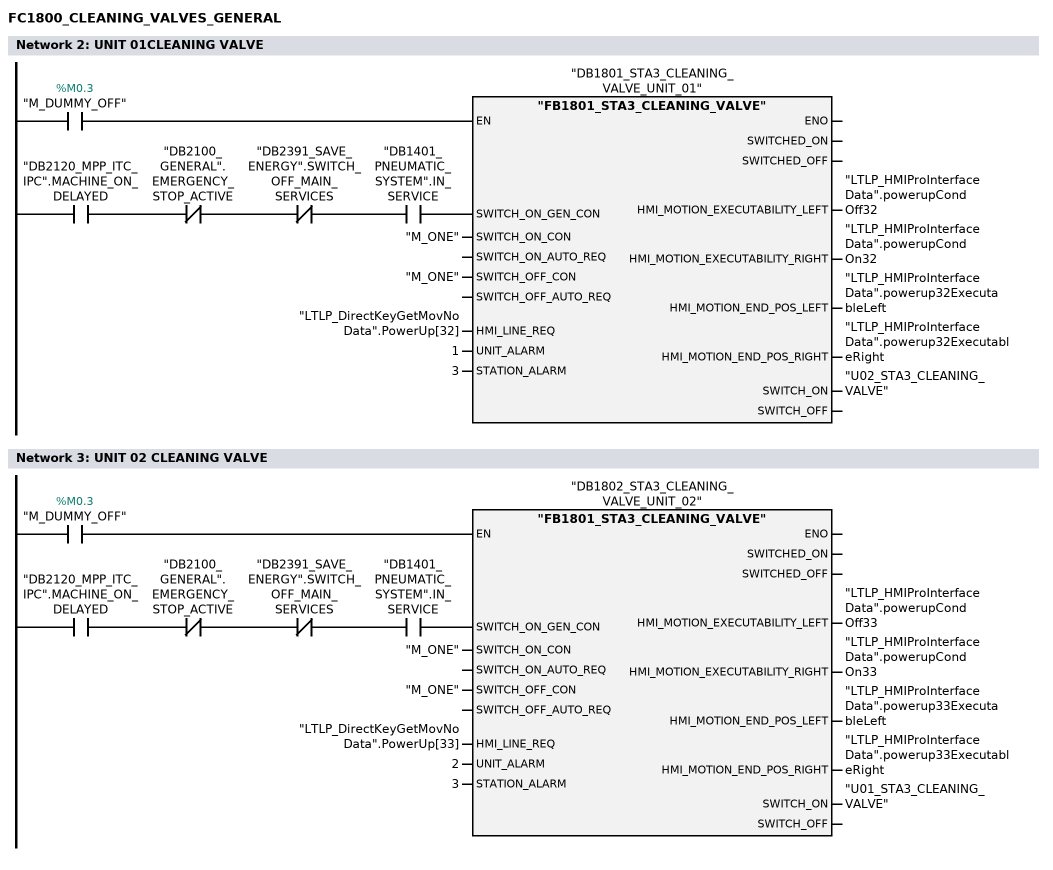
   RUNG wire#powerrail
      Contact( "M_DUMMY_OFF" )
      "DB1801_STA3_CLEANING_VALVE_UNIT_01"(SWITCH_ON_GEN_CON := wire#w1, SWITCH_ON_CON := "M_ONE", SWITCH_ON_AUTO_REQ :=, SWITCH_OFF_CON := "M_ONE", SWITCH_OFF_AUTO_REQ :=, HMI_LINE_REQ := "LTLP_DirectKeyGetMovNoData".PowerUp[32], UNIT_ALARM := 1, STATION_ALARM := 3, SWITCHED_ON =>, SWITCHED_OFF =>, HMI_MOTION_EXECUTABILITY_LEFT => "LTLP_HMIProInterfaceData".powerupCondOff32, HMI_MOTION_EXECUTABILITY_RIGHT => "LTLP_HMIProInterfaceData".powerupCondOn32, HMI_MOTION_END_POS_LEFT => "LTLP_HMIProInterfaceData".powerup32ExecutableLeft, HMI_MOTION_END_POS_RIGHT => "LTLP_HMIProInterfaceData".powerup32ExecutableRight, SWITCH_ON => "U02_STA3_CLEANING_VALVE", SWITCH_OFF =>)
   END_RUNG
   RUNG wire#powerrail
      Contact( "DB2120_MPP_ITC_IPC".MACHINE_ON_DELAYED )
      I_Contact( "DB2100_GENERAL".EMERGENCY_STOP_ACTIVE )
      I_Contact( "DB2391_SAVE_ENERGY".SWITCH_OFF_MAIN_SERVICES )
      Contact( "DB1401_PNEUMATIC_SYSTEM".IN_SERVICE )
   END_RUNG wire#w1
   // the same network as SCL:
   IF "M_DUMMY_OFF" THEN
       "DB1801_STA3_CLEANING_VALVE_UNIT_01"(SWITCH_ON_GEN_CON := "DB2120_MPP_ITC_IPC".MACHINE_ON_DELAYED AND NOT "DB2100_GENERAL".EMERGENCY_STOP_ACTIVE AND NOT "DB2391_SAVE_ENERGY".SWITCH_OFF_MAIN_SERVICES AND "DB1401_PNEUMATIC_SYSTEM".IN_SERVICE,   // "FB1801_STA3_CLEANING_VALVE"
                               SWITCH_ON_CON := "M_ONE",
                               SWITCH_OFF_CON := "M_ONE",
                               HMI_LINE_REQ := "LTLP_DirectKeyGetMovNoData".PowerUp[32],
                               UNIT_ALARM := 1,
                               STATION_ALARM := 3,
                               HMI_MOTION_EXECUTABILITY_LEFT => "LTLP_HMIProInterfaceData".powerupCondOff32,
                               HMI_MOTION_EXECUTABILITY_RIGHT => "LTLP_HMIProInterfaceData".powerupCondOn32,
                               HMI_MOTION_END_POS_LEFT => "LTLP_HMIProInterfaceData".powerup32ExecutableLeft,
                               HMI_MOTION_END_POS_RIGHT => "LTLP_HMIProInterfaceData".powerup32ExecutableRight,
                               SWITCH_ON => "U02_STA3_CLEANING_VALVE");
   END_IF;
END_REGION

REGION Network 3: UNIT 02 CLEANING VALVE
   RUNG wire#powerrail
      Contact( "M_DUMMY_OFF" )
      "DB1802_STA3_CLEANING_VALVE_UNIT_02"(SWITCH_ON_GEN_CON := wire#w1, SWITCH_ON_CON := "M_ONE", SWITCH_ON_AUTO_REQ :=, SWITCH_OFF_CON := "M_ONE", SWITCH_OFF_AUTO_REQ :=, HMI_LINE_REQ := "LTLP_DirectKeyGetMovNoData".PowerUp[33], UNIT_ALARM := 2, STATION_ALARM := 3, SWITCHED_ON =>, SWITCHED_OFF =>, HMI_MOTION_EXECUTABILITY_LEFT => "LTLP_HMIProInterfaceData".powerupCondOff33, HMI_MOTION_EXECUTABILITY_RIGHT => "LTLP_HMIProInterfaceData".powerupCondOn33, HMI_MOTION_END_POS_LEFT => "LTLP_HMIProInterfaceData".powerup33ExecutableLeft, HMI_MOTION_END_POS_RIGHT => "LTLP_HMIProInterfaceData".powerup33ExecutableRight, SWITCH_ON => "U01_STA3_CLEANING_VALVE", SWITCH_OFF =>)
   END_RUNG
   RUNG wire#powerrail
      Contact( "DB2120_MPP_ITC_IPC".MACHINE_ON_DELAYED )
      I_Contact( "DB2100_GENERAL".EMERGENCY_STOP_ACTIVE )
      I_Contact( "DB2391_SAVE_ENERGY".SWITCH_OFF_MAIN_SERVICES )
      Contact( "DB1401_PNEUMATIC_SYSTEM".IN_SERVICE )
   END_RUNG wire#w1
   // the same network as SCL:
   IF "M_DUMMY_OFF" THEN
       "DB1802_STA3_CLEANING_VALVE_UNIT_02"(SWITCH_ON_GEN_CON := "DB2120_MPP_ITC_IPC".MACHINE_ON_DELAYED AND NOT "DB2100_GENERAL".EMERGENCY_STOP_ACTIVE AND NOT "DB2391_SAVE_ENERGY".SWITCH_OFF_MAIN_SERVICES AND "DB1401_PNEUMATIC_SYSTEM".IN_SERVICE,   // "FB1801_STA3_CLEANING_VALVE"
                               SWITCH_ON_CON := "M_ONE",
                               SWITCH_OFF_CON := "M_ONE",
                               HMI_LINE_REQ := "LTLP_DirectKeyGetMovNoData".PowerUp[33],
                               UNIT_ALARM := 2,
                               STATION_ALARM := 3,
                               HMI_MOTION_EXECUTABILITY_LEFT => "LTLP_HMIProInterfaceData".powerupCondOff33,
                               HMI_MOTION_EXECUTABILITY_RIGHT => "LTLP_HMIProInterfaceData".powerupCondOn33,
                               HMI_MOTION_END_POS_LEFT => "LTLP_HMIProInterfaceData".powerup33ExecutableLeft,
                               HMI_MOTION_END_POS_RIGHT => "LTLP_HMIProInterfaceData".powerup33ExecutableRight,
                               SWITCH_ON => "U01_STA3_CLEANING_VALVE");
   END_IF;
END_REGION
END_FUNCTION

FUNCTION "FC2030_MACHINE_CYCLES" : Void   // FC2030, LAD
{ S7_Optimized_Access := 'FALSE' }
AUTHOR : ETXETAR
VERSION : 1.0
// stored: AutoNumber false, IsIECCheckEnabled false, SetENOAutomatically false, UDAEnableTagReadback false
BEGIN

REGION Network 1: CALL FC2031 MACHINE CONTINUOUS CYCLE
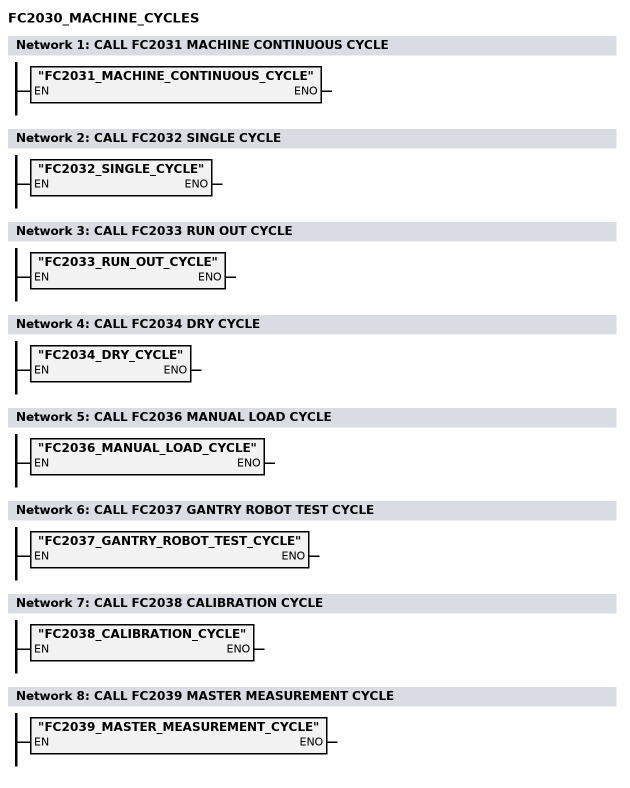
   RUNG wire#powerrail
      "FC2031_MACHINE_CONTINUOUS_CYCLE"()
   END_RUNG
   // the same network as SCL:
   "FC2031_MACHINE_CONTINUOUS_CYCLE"();
END_REGION

REGION Network 2: CALL FC2032 SINGLE CYCLE
   RUNG wire#powerrail
      "FC2032_SINGLE_CYCLE"()
   END_RUNG
   // the same network as SCL:
   "FC2032_SINGLE_CYCLE"();
END_REGION

REGION Network 3: CALL FC2033 RUN OUT CYCLE
   RUNG wire#powerrail
      "FC2033_RUN_OUT_CYCLE"()
   END_RUNG
   // the same network as SCL:
   "FC2033_RUN_OUT_CYCLE"();
END_REGION

REGION Network 4: CALL FC2034 DRY CYCLE
   RUNG wire#powerrail
      "FC2034_DRY_CYCLE"()
   END_RUNG
   // the same network as SCL:
   "FC2034_DRY_CYCLE"();
END_REGION

REGION Network 5: CALL FC2036 MANUAL LOAD CYCLE
   RUNG wire#powerrail
      "FC2036_MANUAL_LOAD_CYCLE"()
   END_RUNG
   // the same network as SCL:
   "FC2036_MANUAL_LOAD_CYCLE"();
END_REGION

REGION Network 6: CALL FC2037 GANTRY ROBOT TEST CYCLE
   RUNG wire#powerrail
      "FC2037_GANTRY_ROBOT_TEST_CYCLE"()
   END_RUNG
   // the same network as SCL:
   "FC2037_GANTRY_ROBOT_TEST_CYCLE"();
END_REGION

REGION Network 7: CALL FC2038 CALIBRATION CYCLE
   RUNG wire#powerrail
      "FC2038_CALIBRATION_CYCLE"()
   END_RUNG
   // the same network as SCL:
   "FC2038_CALIBRATION_CYCLE"();
END_REGION

REGION Network 8: CALL FC2039 MASTER MEASUREMENT CYCLE
   RUNG wire#powerrail
      "FC2039_MASTER_MEASUREMENT_CYCLE"()
   END_RUNG
   // the same network as SCL:
   "FC2039_MASTER_MEASUREMENT_CYCLE"();
END_REGION
END_FUNCTION

FUNCTION_BLOCK "FB2002_BA_MODE"   // FB2002, LAD
{ S7_Optimized_Access := 'FALSE' }
VERSION : 0.1
// stored: AutoNumber false, IsIECCheckEnabled false, SetENOAutomatically false, UDAEnableTagReadback false
   VAR_INPUT
      OPTIONS_0 { ExternalAccessible := 'False'; ExternalVisible := 'False'; ExternalWritable := 'False'} : Byte := 2#0000_0000;   // OPTIONS BYTE 0
      BA1_BUTTON_I { ExternalAccessible := 'False'; ExternalVisible := 'False'; ExternalWritable := 'False'} : Bool;   // BA1 BUTTON INPUT
      BA2_BUTTON_I { ExternalAccessible := 'False'; ExternalVisible := 'False'; ExternalWritable := 'False'} : Bool;   // BA2 BUTTON INPUT
      BA3_BUTTON_I { ExternalAccessible := 'False'; ExternalVisible := 'False'; ExternalWritable := 'False'} : Bool;   // BA3 BUTTON INPUT
      BA5_BUTTON_I { ExternalAccessible := 'False'; ExternalVisible := 'False'; ExternalWritable := 'False'} : Bool;   // BA5 BUTTON INPUT
      SAFETY_ENABLED_W_DOOR_OPENED { ExternalAccessible := 'False'; ExternalVisible := 'False'; ExternalWritable := 'False'} : Bool;   // SAFETY ENABLED WITH DOOR OPENED (ENABLING DEVICE AND HT10 ENABLE BUTTON)
      SAFETY_GATES_CLSD_AND_LCKD { ExternalAccessible := 'False'; ExternalVisible := 'False'; ExternalWritable := 'False'} : Bool;   // SAFETY GATES CLOSED AND LOCKED
      START_SERVICES_GLOBAL { ExternalAccessible := 'False'; ExternalVisible := 'False'; ExternalWritable := 'False'} : Bool;   // START SERVICES GLOBAL
      ANY_MCH_CYCLE_RUN { ExternalAccessible := 'False'; ExternalVisible := 'False'; ExternalWritable := 'False'} : Bool;   // ANY MACHINE CYCLE RUNNING
      MCH_RESET_FAULTS { ExternalAccessible := 'False'; ExternalVisible := 'False'; ExternalWritable := 'False'} : Bool;   // MACHINE_RESET_FAULTS
   END_VAR
   VAR_OUTPUT
      NO_BA_MODE_SLCTD_WRN { ExternalAccessible := 'False'; ExternalVisible := 'False'; ExternalWritable := 'False'} : Bool;   // NO BA MODE SELECTED WARNING
      CHANGE_TO_BA1_MODE_WRN { ExternalAccessible := 'False'; ExternalVisible := 'False'; ExternalWritable := 'False'} : Bool;   // CHANGE TO BA1 MODE WARNING
      CHANGE_TO_BA2_MODE_WRN { ExternalAccessible := 'False'; ExternalVisible := 'False'; ExternalWritable := 'False'} : Bool;   // CHANGE TO BA2 MODE WARNING
      CHANGE_TO_BA3_MODE_WRN { ExternalAccessible := 'False'; ExternalVisible := 'False'; ExternalWritable := 'False'} : Bool;   // CHANGE TO BA3 MODE WARNING
      CHANGE_TO_BA5_MODE_WRN { ExternalAccessible := 'False'; ExternalVisible := 'False'; ExternalWritable := 'False'} : Bool;   // CHANGE TO BA5 MODE WARNING
      BA1_MODE_LED_O { ExternalAccessible := 'False'; ExternalVisible := 'False'; ExternalWritable := 'False'} : Bool;   // BA1 MODE BUTTON LED OUTPUT
      BA2_MODE_LED_O { ExternalAccessible := 'False'; ExternalVisible := 'False'; ExternalWritable := 'False'} : Bool;   // BA2 MODE BUTTON LED OUTPUT
      BA3_MODE_LED_O { ExternalAccessible := 'False'; ExternalVisible := 'False'; ExternalWritable := 'False'} : Bool;   // BA3 MODE BUTTON LED OUTPUT
   END_VAR
   VAR_IN_OUT
      MODE_GROUP_GENERAL_DB : "AUTO_SINGLE_SEMI_MANUAL";
      MODE_GROUP_BA_DB : "BA_MODE";
   END_VAR
   VAR_TEMP
      INPUTS_MASK : Byte;   // INPUT MASK
      O_BYTE_0 : Struct   // OPTIONS BYTE 0
         BA_BUTTONS : Bool;   // BA MODE BUTTONS OPTION
         CHANGE_MODE_SEOC_ALARM : Bool;   // CHANGE MODE SEOC ALARM OPTION
         MODE_SELECTED_MEMORY : Bool;   // MODE SELECTED MEMORY OPTION
         SPARE : Bool;
         SPARE_1 : Bool;
         SPARE_2 : Bool;
         SPARE_3 : Bool;
         SPARE_4 : Bool;
      END_STRUCT;
      DB_NUMBER : DInt;   // DB NUMBER FOR ALARM DECODING
   END_VAR
   VAR_TEMP   // added for the SCL form of the ladder/FBD networks
      _w1 : Bool;
      _w2 : Bool;
   END_VAR
BEGIN

NETWORK
TITLE = READ INSTANCE DB
      L     DINO;
      +     10#800000;
      T     #DB_NUMBER;


REGION Network 2: OPTIONS
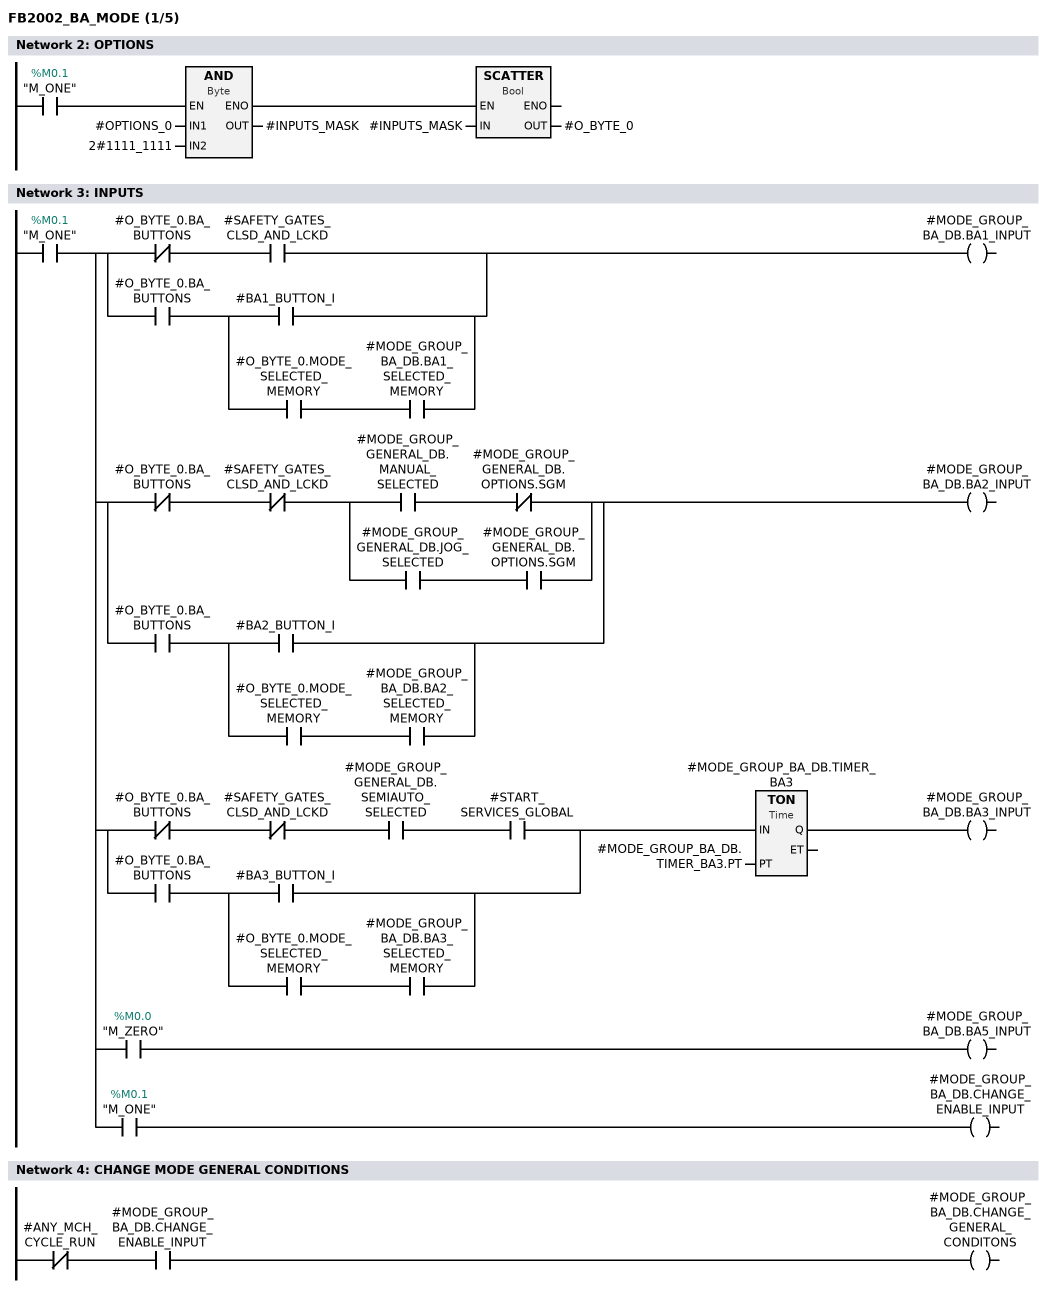
   RUNG wire#powerrail
      Contact( "M_ONE" )
      { S7_Templates := "SrcType := Byte"; S7_GenerateENO := "TRUE" } And(in1 := #OPTIONS_0, in2 := 2#1111_1111, out => #INPUTS_MASK)
      { S7_Templates := "[dest_type := Bool, src_type := Byte]" } SCATTER(IN := #INPUTS_MASK, OUT => #O_BYTE_0)
   END_RUNG
   // the same network as SCL:
   IF "M_ONE" THEN
       #INPUTS_MASK := #OPTIONS_0 AND 2#1111_1111;
       SCATTER(IN := #INPUTS_MASK, OUT => #O_BYTE_0);
   END_IF;
END_REGION

REGION Network 3: INPUTS
   RUNG wire#powerrail
      Contact( "M_ONE" )
      wire#w1
      I_Contact( #O_BYTE_0.BA_BUTTONS )
      Contact( #SAFETY_GATES_CLSD_AND_LCKD )
      wire#w2
      Coil( #MODE_GROUP_BA_DB.BA1_INPUT )
   END_RUNG
   RUNG wire#w1
      Contact( #O_BYTE_0.BA_BUTTONS )
      wire#w3
      Contact( #BA1_BUTTON_I )
   END_RUNG wire#w2
   RUNG wire#w3
      Contact( #O_BYTE_0.MODE_SELECTED_MEMORY )
      Contact( #MODE_GROUP_BA_DB.BA1_SELECTED_MEMORY )
   END_RUNG wire#w2
   RUNG wire#w1
      I_Contact( #O_BYTE_0.BA_BUTTONS )
      I_Contact( #SAFETY_GATES_CLSD_AND_LCKD )
      wire#w4
      Contact( #MODE_GROUP_GENERAL_DB.MANUAL_SELECTED )
      I_Contact( #MODE_GROUP_GENERAL_DB.OPTIONS.SGM )
      wire#w5
      Coil( #MODE_GROUP_BA_DB.BA2_INPUT )
   END_RUNG
   RUNG wire#w4
      Contact( #MODE_GROUP_GENERAL_DB.JOG_SELECTED )
      Contact( #MODE_GROUP_GENERAL_DB.OPTIONS.SGM )
   END_RUNG wire#w5
   RUNG wire#w1
      Contact( #O_BYTE_0.BA_BUTTONS )
      wire#w6
      Contact( #BA2_BUTTON_I )
   END_RUNG wire#w5
   RUNG wire#w6
      Contact( #O_BYTE_0.MODE_SELECTED_MEMORY )
      Contact( #MODE_GROUP_BA_DB.BA2_SELECTED_MEMORY )
   END_RUNG wire#w5
   RUNG wire#w1
      I_Contact( #O_BYTE_0.BA_BUTTONS )
      I_Contact( #SAFETY_GATES_CLSD_AND_LCKD )
      Contact( #MODE_GROUP_GENERAL_DB.SEMIAUTO_SELECTED )
      Contact( #START_SERVICES_GLOBAL )
      wire#w7
      { S7_Templates := "time_type := Time" } #MODE_GROUP_BA_DB.TIMER_BA3.TON(pt := #MODE_GROUP_BA_DB.TIMER_BA3.PT, et =>)
      Coil( #MODE_GROUP_BA_DB.BA3_INPUT )
   END_RUNG
   RUNG wire#w1
      Contact( #O_BYTE_0.BA_BUTTONS )
      wire#w8
      Contact( #BA3_BUTTON_I )
   END_RUNG wire#w7
   RUNG wire#w8
      Contact( #O_BYTE_0.MODE_SELECTED_MEMORY )
      Contact( #MODE_GROUP_BA_DB.BA3_SELECTED_MEMORY )
   END_RUNG wire#w7
   RUNG wire#w1
      Contact( "M_ZERO" )
      Coil( #MODE_GROUP_BA_DB.BA5_INPUT )
   END_RUNG
   RUNG wire#w1
      Contact( "M_ONE" )
      Coil( #MODE_GROUP_BA_DB.CHANGE_ENABLE_INPUT )
   END_RUNG
   // the same network as SCL:
   #MODE_GROUP_BA_DB.BA1_INPUT := "M_ONE" AND ((NOT #O_BYTE_0.BA_BUTTONS AND #SAFETY_GATES_CLSD_AND_LCKD) OR (#O_BYTE_0.BA_BUTTONS AND (#BA1_BUTTON_I OR (#O_BYTE_0.MODE_SELECTED_MEMORY AND #MODE_GROUP_BA_DB.BA1_SELECTED_MEMORY))));
   #MODE_GROUP_BA_DB.BA2_INPUT := "M_ONE" AND ((NOT #O_BYTE_0.BA_BUTTONS AND NOT #SAFETY_GATES_CLSD_AND_LCKD AND ((#MODE_GROUP_GENERAL_DB.MANUAL_SELECTED AND NOT #MODE_GROUP_GENERAL_DB.OPTIONS.SGM) OR (#MODE_GROUP_GENERAL_DB.JOG_SELECTED AND #MODE_GROUP_GENERAL_DB.OPTIONS.SGM))) OR (#O_BYTE_0.BA_BUTTONS AND (#BA2_BUTTON_I OR (#O_BYTE_0.MODE_SELECTED_MEMORY AND #MODE_GROUP_BA_DB.BA2_SELECTED_MEMORY))));
   #MODE_GROUP_BA_DB.TIMER_BA3.TON(IN := "M_ONE" AND ((NOT #O_BYTE_0.BA_BUTTONS AND NOT #SAFETY_GATES_CLSD_AND_LCKD AND #MODE_GROUP_GENERAL_DB.SEMIAUTO_SELECTED AND #START_SERVICES_GLOBAL) OR (#O_BYTE_0.BA_BUTTONS AND (#BA3_BUTTON_I OR (#O_BYTE_0.MODE_SELECTED_MEMORY AND #MODE_GROUP_BA_DB.BA3_SELECTED_MEMORY)))),
                           PT := #MODE_GROUP_BA_DB.TIMER_BA3.PT);
   #MODE_GROUP_BA_DB.BA3_INPUT := #MODE_GROUP_BA_DB.TIMER_BA3.Q;
   #MODE_GROUP_BA_DB.BA5_INPUT := "M_ONE" AND "M_ZERO";
   #MODE_GROUP_BA_DB.CHANGE_ENABLE_INPUT := "M_ONE" AND "M_ONE";
END_REGION

REGION Network 4: CHANGE MODE GENERAL CONDITIONS
   RUNG wire#powerrail
      I_Contact( #ANY_MCH_CYCLE_RUN )
      Contact( #MODE_GROUP_BA_DB.CHANGE_ENABLE_INPUT )
      Coil( #MODE_GROUP_BA_DB.CHANGE_GENERAL_CONDITONS )
   END_RUNG
   // the same network as SCL:
   #MODE_GROUP_BA_DB.CHANGE_GENERAL_CONDITONS := NOT #ANY_MCH_CYCLE_RUN AND #MODE_GROUP_BA_DB.CHANGE_ENABLE_INPUT;
END_REGION

REGION Network 5: OPERATOR HELP
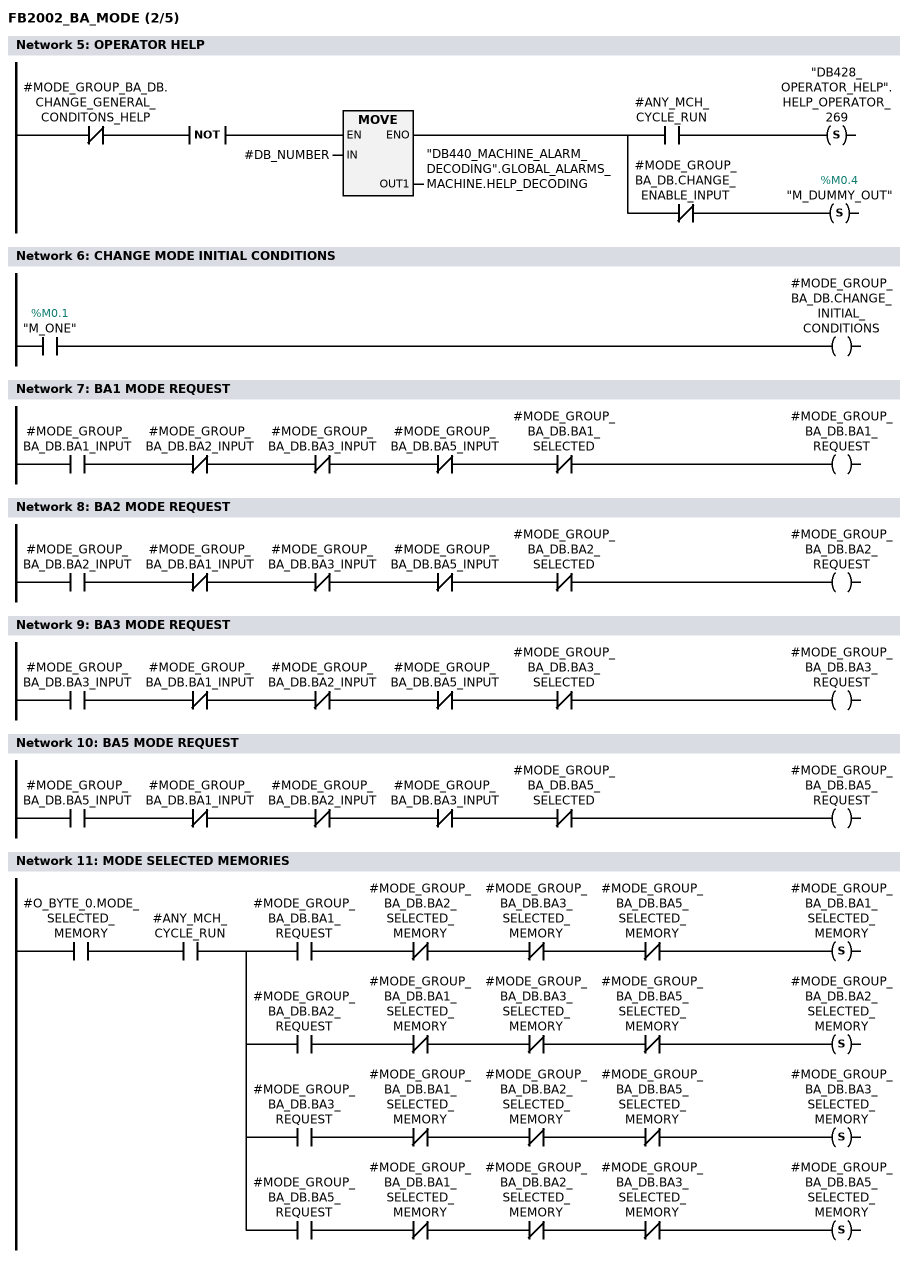
   RUNG wire#powerrail
      I_Contact( #MODE_GROUP_BA_DB.CHANGE_GENERAL_CONDITONS_HELP )
      Not()
      { S7_GenerateENO := "TRUE" } Move(in := #DB_NUMBER, out1 => "DB440_MACHINE_ALARM_DECODING".GLOBAL_ALARMS_MACHINE.HELP_DECODING)
      wire#w1
      Contact( #ANY_MCH_CYCLE_RUN )
      S_Coil( "DB428_OPERATOR_HELP".HELP_OPERATOR_269 )
   END_RUNG
   RUNG wire#w1
      I_Contact( #MODE_GROUP_BA_DB.CHANGE_ENABLE_INPUT )
      S_Coil( "M_DUMMY_OUT" )
   END_RUNG
   // the same network as SCL:
   // ENO of a box is taken as its EN; it also drops when the box reports an error
   #_w1 := NOT (NOT #MODE_GROUP_BA_DB.CHANGE_GENERAL_CONDITONS_HELP);
   IF #_w1 THEN "DB440_MACHINE_ALARM_DECODING".GLOBAL_ALARMS_MACHINE.HELP_DECODING := #DB_NUMBER; END_IF;
   IF #_w1 AND #ANY_MCH_CYCLE_RUN THEN "DB428_OPERATOR_HELP".HELP_OPERATOR_269 := TRUE; END_IF;
   IF #_w1 AND NOT #MODE_GROUP_BA_DB.CHANGE_ENABLE_INPUT THEN "M_DUMMY_OUT" := TRUE; END_IF;
END_REGION

REGION Network 6: CHANGE MODE INITIAL CONDITIONS
   RUNG wire#powerrail
      Contact( "M_ONE" )
      Coil( #MODE_GROUP_BA_DB.CHANGE_INITIAL_CONDITIONS )
   END_RUNG
   // the same network as SCL:
   #MODE_GROUP_BA_DB.CHANGE_INITIAL_CONDITIONS := "M_ONE";
END_REGION

REGION Network 7: BA1 MODE REQUEST
   RUNG wire#powerrail
      Contact( #MODE_GROUP_BA_DB.BA1_INPUT )
      I_Contact( #MODE_GROUP_BA_DB.BA2_INPUT )
      I_Contact( #MODE_GROUP_BA_DB.BA3_INPUT )
      I_Contact( #MODE_GROUP_BA_DB.BA5_INPUT )
      I_Contact( #MODE_GROUP_BA_DB.BA1_SELECTED )
      Coil( #MODE_GROUP_BA_DB.BA1_REQUEST )
   END_RUNG
   // the same network as SCL:
   #MODE_GROUP_BA_DB.BA1_REQUEST := #MODE_GROUP_BA_DB.BA1_INPUT AND NOT #MODE_GROUP_BA_DB.BA2_INPUT AND NOT #MODE_GROUP_BA_DB.BA3_INPUT AND NOT #MODE_GROUP_BA_DB.BA5_INPUT AND NOT #MODE_GROUP_BA_DB.BA1_SELECTED;
END_REGION

REGION Network 8: BA2 MODE REQUEST
   RUNG wire#powerrail
      Contact( #MODE_GROUP_BA_DB.BA2_INPUT )
      I_Contact( #MODE_GROUP_BA_DB.BA1_INPUT )
      I_Contact( #MODE_GROUP_BA_DB.BA3_INPUT )
      I_Contact( #MODE_GROUP_BA_DB.BA5_INPUT )
      I_Contact( #MODE_GROUP_BA_DB.BA2_SELECTED )
      Coil( #MODE_GROUP_BA_DB.BA2_REQUEST )
   END_RUNG
   // the same network as SCL:
   #MODE_GROUP_BA_DB.BA2_REQUEST := #MODE_GROUP_BA_DB.BA2_INPUT AND NOT #MODE_GROUP_BA_DB.BA1_INPUT AND NOT #MODE_GROUP_BA_DB.BA3_INPUT AND NOT #MODE_GROUP_BA_DB.BA5_INPUT AND NOT #MODE_GROUP_BA_DB.BA2_SELECTED;
END_REGION

REGION Network 9: BA3 MODE REQUEST
   RUNG wire#powerrail
      Contact( #MODE_GROUP_BA_DB.BA3_INPUT )
      I_Contact( #MODE_GROUP_BA_DB.BA1_INPUT )
      I_Contact( #MODE_GROUP_BA_DB.BA2_INPUT )
      I_Contact( #MODE_GROUP_BA_DB.BA5_INPUT )
      I_Contact( #MODE_GROUP_BA_DB.BA3_SELECTED )
      Coil( #MODE_GROUP_BA_DB.BA3_REQUEST )
   END_RUNG
   // the same network as SCL:
   #MODE_GROUP_BA_DB.BA3_REQUEST := #MODE_GROUP_BA_DB.BA3_INPUT AND NOT #MODE_GROUP_BA_DB.BA1_INPUT AND NOT #MODE_GROUP_BA_DB.BA2_INPUT AND NOT #MODE_GROUP_BA_DB.BA5_INPUT AND NOT #MODE_GROUP_BA_DB.BA3_SELECTED;
END_REGION

REGION Network 10: BA5 MODE REQUEST
   RUNG wire#powerrail
      Contact( #MODE_GROUP_BA_DB.BA5_INPUT )
      I_Contact( #MODE_GROUP_BA_DB.BA1_INPUT )
      I_Contact( #MODE_GROUP_BA_DB.BA2_INPUT )
      I_Contact( #MODE_GROUP_BA_DB.BA3_INPUT )
      I_Contact( #MODE_GROUP_BA_DB.BA5_SELECTED )
      Coil( #MODE_GROUP_BA_DB.BA5_REQUEST )
   END_RUNG
   // the same network as SCL:
   #MODE_GROUP_BA_DB.BA5_REQUEST := #MODE_GROUP_BA_DB.BA5_INPUT AND NOT #MODE_GROUP_BA_DB.BA1_INPUT AND NOT #MODE_GROUP_BA_DB.BA2_INPUT AND NOT #MODE_GROUP_BA_DB.BA3_INPUT AND NOT #MODE_GROUP_BA_DB.BA5_SELECTED;
END_REGION

REGION Network 11: MODE SELECTED MEMORIES
   RUNG wire#powerrail
      Contact( #O_BYTE_0.MODE_SELECTED_MEMORY )
      Contact( #ANY_MCH_CYCLE_RUN )
      wire#w1
      Contact( #MODE_GROUP_BA_DB.BA1_REQUEST )
      I_Contact( #MODE_GROUP_BA_DB.BA2_SELECTED_MEMORY )
      I_Contact( #MODE_GROUP_BA_DB.BA3_SELECTED_MEMORY )
      I_Contact( #MODE_GROUP_BA_DB.BA5_SELECTED_MEMORY )
      S_Coil( #MODE_GROUP_BA_DB.BA1_SELECTED_MEMORY )
   END_RUNG
   RUNG wire#w1
      Contact( #MODE_GROUP_BA_DB.BA2_REQUEST )
      I_Contact( #MODE_GROUP_BA_DB.BA1_SELECTED_MEMORY )
      I_Contact( #MODE_GROUP_BA_DB.BA3_SELECTED_MEMORY )
      I_Contact( #MODE_GROUP_BA_DB.BA5_SELECTED_MEMORY )
      S_Coil( #MODE_GROUP_BA_DB.BA2_SELECTED_MEMORY )
   END_RUNG
   RUNG wire#w1
      Contact( #MODE_GROUP_BA_DB.BA3_REQUEST )
      I_Contact( #MODE_GROUP_BA_DB.BA1_SELECTED_MEMORY )
      I_Contact( #MODE_GROUP_BA_DB.BA2_SELECTED_MEMORY )
      I_Contact( #MODE_GROUP_BA_DB.BA5_SELECTED_MEMORY )
      S_Coil( #MODE_GROUP_BA_DB.BA3_SELECTED_MEMORY )
   END_RUNG
   RUNG wire#w1
      Contact( #MODE_GROUP_BA_DB.BA5_REQUEST )
      I_Contact( #MODE_GROUP_BA_DB.BA1_SELECTED_MEMORY )
      I_Contact( #MODE_GROUP_BA_DB.BA2_SELECTED_MEMORY )
      I_Contact( #MODE_GROUP_BA_DB.BA3_SELECTED_MEMORY )
      S_Coil( #MODE_GROUP_BA_DB.BA5_SELECTED_MEMORY )
   END_RUNG
   // the same network as SCL:
   #_w1 := #O_BYTE_0.MODE_SELECTED_MEMORY AND #ANY_MCH_CYCLE_RUN;
   IF #_w1 AND #MODE_GROUP_BA_DB.BA1_REQUEST AND NOT #MODE_GROUP_BA_DB.BA2_SELECTED_MEMORY AND NOT #MODE_GROUP_BA_DB.BA3_SELECTED_MEMORY AND NOT #MODE_GROUP_BA_DB.BA5_SELECTED_MEMORY THEN
       #MODE_GROUP_BA_DB.BA1_SELECTED_MEMORY := TRUE;
   END_IF;
   IF #_w1 AND #MODE_GROUP_BA_DB.BA2_REQUEST AND NOT #MODE_GROUP_BA_DB.BA1_SELECTED_MEMORY AND NOT #MODE_GROUP_BA_DB.BA3_SELECTED_MEMORY AND NOT #MODE_GROUP_BA_DB.BA5_SELECTED_MEMORY THEN
       #MODE_GROUP_BA_DB.BA2_SELECTED_MEMORY := TRUE;
   END_IF;
   IF #_w1 AND #MODE_GROUP_BA_DB.BA3_REQUEST AND NOT #MODE_GROUP_BA_DB.BA1_SELECTED_MEMORY AND NOT #MODE_GROUP_BA_DB.BA2_SELECTED_MEMORY AND NOT #MODE_GROUP_BA_DB.BA5_SELECTED_MEMORY THEN
       #MODE_GROUP_BA_DB.BA3_SELECTED_MEMORY := TRUE;
   END_IF;
   IF #_w1 AND #MODE_GROUP_BA_DB.BA5_REQUEST AND NOT #MODE_GROUP_BA_DB.BA1_SELECTED_MEMORY AND NOT #MODE_GROUP_BA_DB.BA2_SELECTED_MEMORY AND NOT #MODE_GROUP_BA_DB.BA3_SELECTED_MEMORY THEN
       #MODE_GROUP_BA_DB.BA5_SELECTED_MEMORY := TRUE;
   END_IF;
END_REGION

REGION Network 12: BA1 MODE SELECTED
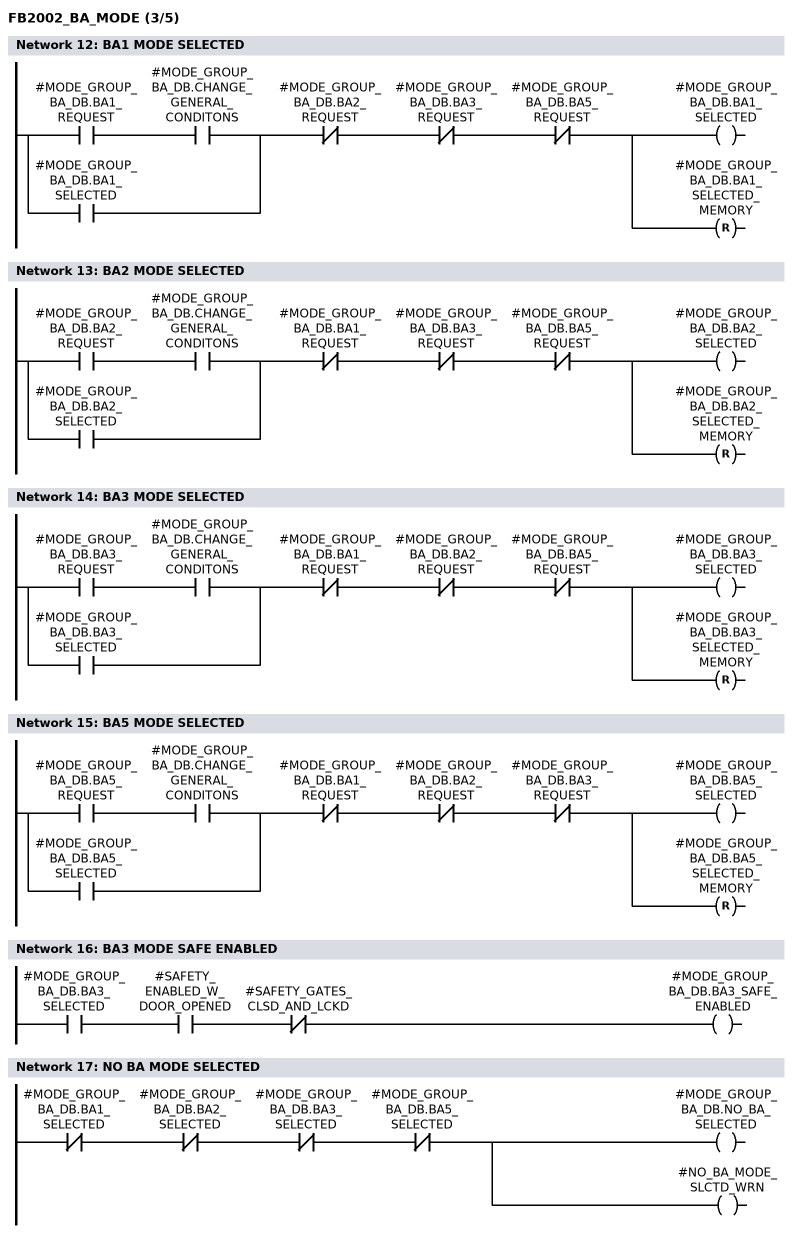
   RUNG wire#powerrail
      Contact( #MODE_GROUP_BA_DB.BA1_REQUEST )
      Contact( #MODE_GROUP_BA_DB.CHANGE_GENERAL_CONDITONS )
      wire#w1
      I_Contact( #MODE_GROUP_BA_DB.BA2_REQUEST )
      I_Contact( #MODE_GROUP_BA_DB.BA3_REQUEST )
      I_Contact( #MODE_GROUP_BA_DB.BA5_REQUEST )
      wire#w2
      Coil( #MODE_GROUP_BA_DB.BA1_SELECTED )
   END_RUNG
   RUNG wire#powerrail
      Contact( #MODE_GROUP_BA_DB.BA1_SELECTED )
   END_RUNG wire#w1
   RUNG wire#w2
      R_Coil( #MODE_GROUP_BA_DB.BA1_SELECTED_MEMORY )
   END_RUNG
   // the same network as SCL:
   #MODE_GROUP_BA_DB.BA1_SELECTED := ((#MODE_GROUP_BA_DB.BA1_REQUEST AND #MODE_GROUP_BA_DB.CHANGE_GENERAL_CONDITONS) OR #MODE_GROUP_BA_DB.BA1_SELECTED) AND NOT #MODE_GROUP_BA_DB.BA2_REQUEST AND NOT #MODE_GROUP_BA_DB.BA3_REQUEST AND NOT #MODE_GROUP_BA_DB.BA5_REQUEST;
   IF #MODE_GROUP_BA_DB.BA1_SELECTED THEN #MODE_GROUP_BA_DB.BA1_SELECTED_MEMORY := FALSE; END_IF;
END_REGION

REGION Network 13: BA2 MODE SELECTED
   RUNG wire#powerrail
      Contact( #MODE_GROUP_BA_DB.BA2_REQUEST )
      Contact( #MODE_GROUP_BA_DB.CHANGE_GENERAL_CONDITONS )
      wire#w1
      I_Contact( #MODE_GROUP_BA_DB.BA1_REQUEST )
      I_Contact( #MODE_GROUP_BA_DB.BA3_REQUEST )
      I_Contact( #MODE_GROUP_BA_DB.BA5_REQUEST )
      wire#w2
      Coil( #MODE_GROUP_BA_DB.BA2_SELECTED )
   END_RUNG
   RUNG wire#powerrail
      Contact( #MODE_GROUP_BA_DB.BA2_SELECTED )
   END_RUNG wire#w1
   RUNG wire#w2
      R_Coil( #MODE_GROUP_BA_DB.BA2_SELECTED_MEMORY )
   END_RUNG
   // the same network as SCL:
   #MODE_GROUP_BA_DB.BA2_SELECTED := ((#MODE_GROUP_BA_DB.BA2_REQUEST AND #MODE_GROUP_BA_DB.CHANGE_GENERAL_CONDITONS) OR #MODE_GROUP_BA_DB.BA2_SELECTED) AND NOT #MODE_GROUP_BA_DB.BA1_REQUEST AND NOT #MODE_GROUP_BA_DB.BA3_REQUEST AND NOT #MODE_GROUP_BA_DB.BA5_REQUEST;
   IF #MODE_GROUP_BA_DB.BA2_SELECTED THEN #MODE_GROUP_BA_DB.BA2_SELECTED_MEMORY := FALSE; END_IF;
END_REGION

REGION Network 14: BA3 MODE SELECTED
   RUNG wire#powerrail
      Contact( #MODE_GROUP_BA_DB.BA3_REQUEST )
      Contact( #MODE_GROUP_BA_DB.CHANGE_GENERAL_CONDITONS )
      wire#w1
      I_Contact( #MODE_GROUP_BA_DB.BA1_REQUEST )
      I_Contact( #MODE_GROUP_BA_DB.BA2_REQUEST )
      I_Contact( #MODE_GROUP_BA_DB.BA5_REQUEST )
      wire#w2
      Coil( #MODE_GROUP_BA_DB.BA3_SELECTED )
   END_RUNG
   RUNG wire#powerrail
      Contact( #MODE_GROUP_BA_DB.BA3_SELECTED )
   END_RUNG wire#w1
   RUNG wire#w2
      R_Coil( #MODE_GROUP_BA_DB.BA3_SELECTED_MEMORY )
   END_RUNG
   // the same network as SCL:
   #MODE_GROUP_BA_DB.BA3_SELECTED := ((#MODE_GROUP_BA_DB.BA3_REQUEST AND #MODE_GROUP_BA_DB.CHANGE_GENERAL_CONDITONS) OR #MODE_GROUP_BA_DB.BA3_SELECTED) AND NOT #MODE_GROUP_BA_DB.BA1_REQUEST AND NOT #MODE_GROUP_BA_DB.BA2_REQUEST AND NOT #MODE_GROUP_BA_DB.BA5_REQUEST;
   IF #MODE_GROUP_BA_DB.BA3_SELECTED THEN #MODE_GROUP_BA_DB.BA3_SELECTED_MEMORY := FALSE; END_IF;
END_REGION

REGION Network 15: BA5 MODE SELECTED
   RUNG wire#powerrail
      Contact( #MODE_GROUP_BA_DB.BA5_REQUEST )
      Contact( #MODE_GROUP_BA_DB.CHANGE_GENERAL_CONDITONS )
      wire#w1
      I_Contact( #MODE_GROUP_BA_DB.BA1_REQUEST )
      I_Contact( #MODE_GROUP_BA_DB.BA2_REQUEST )
      I_Contact( #MODE_GROUP_BA_DB.BA3_REQUEST )
      wire#w2
      Coil( #MODE_GROUP_BA_DB.BA5_SELECTED )
   END_RUNG
   RUNG wire#powerrail
      Contact( #MODE_GROUP_BA_DB.BA5_SELECTED )
   END_RUNG wire#w1
   RUNG wire#w2
      R_Coil( #MODE_GROUP_BA_DB.BA5_SELECTED_MEMORY )
   END_RUNG
   // the same network as SCL:
   #MODE_GROUP_BA_DB.BA5_SELECTED := ((#MODE_GROUP_BA_DB.BA5_REQUEST AND #MODE_GROUP_BA_DB.CHANGE_GENERAL_CONDITONS) OR #MODE_GROUP_BA_DB.BA5_SELECTED) AND NOT #MODE_GROUP_BA_DB.BA1_REQUEST AND NOT #MODE_GROUP_BA_DB.BA2_REQUEST AND NOT #MODE_GROUP_BA_DB.BA3_REQUEST;
   IF #MODE_GROUP_BA_DB.BA5_SELECTED THEN #MODE_GROUP_BA_DB.BA5_SELECTED_MEMORY := FALSE; END_IF;
END_REGION

REGION Network 16: BA3 MODE SAFE ENABLED
   RUNG wire#powerrail
      Contact( #MODE_GROUP_BA_DB.BA3_SELECTED )
      Contact( #SAFETY_ENABLED_W_DOOR_OPENED )
      I_Contact( #SAFETY_GATES_CLSD_AND_LCKD )
      Coil( #MODE_GROUP_BA_DB.BA3_SAFE_ENABLED )
   END_RUNG
   // the same network as SCL:
   #MODE_GROUP_BA_DB.BA3_SAFE_ENABLED := #MODE_GROUP_BA_DB.BA3_SELECTED AND #SAFETY_ENABLED_W_DOOR_OPENED AND NOT #SAFETY_GATES_CLSD_AND_LCKD;
END_REGION

REGION Network 17: NO BA MODE SELECTED
   RUNG wire#powerrail
      I_Contact( #MODE_GROUP_BA_DB.BA1_SELECTED )
      I_Contact( #MODE_GROUP_BA_DB.BA2_SELECTED )
      I_Contact( #MODE_GROUP_BA_DB.BA3_SELECTED )
      I_Contact( #MODE_GROUP_BA_DB.BA5_SELECTED )
      wire#w1
      Coil( #MODE_GROUP_BA_DB.NO_BA_SELECTED )
   END_RUNG
   RUNG wire#w1
      Coil( #NO_BA_MODE_SLCTD_WRN )
   END_RUNG
   // the same network as SCL:
   #MODE_GROUP_BA_DB.NO_BA_SELECTED := NOT #MODE_GROUP_BA_DB.BA1_SELECTED AND NOT #MODE_GROUP_BA_DB.BA2_SELECTED AND NOT #MODE_GROUP_BA_DB.BA3_SELECTED AND NOT #MODE_GROUP_BA_DB.BA5_SELECTED;
   #NO_BA_MODE_SLCTD_WRN := #MODE_GROUP_BA_DB.NO_BA_SELECTED;
END_REGION

REGION Network 18: CHANGE TO BA1 MODE ALARM
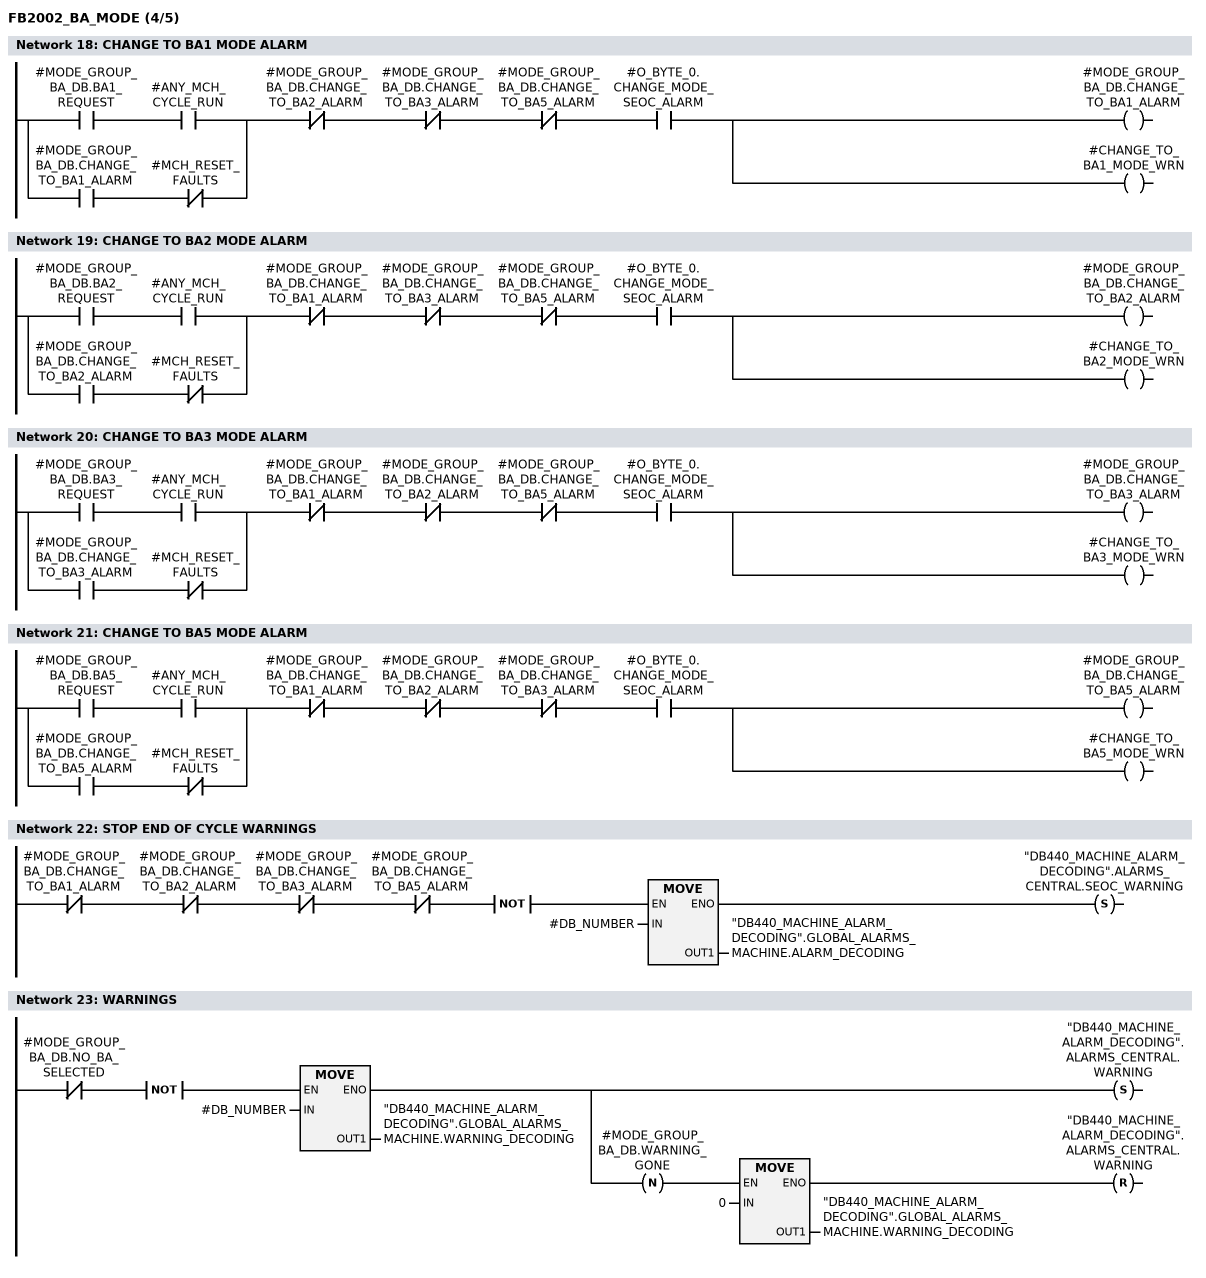
   RUNG wire#powerrail
      Contact( #MODE_GROUP_BA_DB.BA1_REQUEST )
      Contact( #ANY_MCH_CYCLE_RUN )
      wire#w1
      I_Contact( #MODE_GROUP_BA_DB.CHANGE_TO_BA2_ALARM )
      I_Contact( #MODE_GROUP_BA_DB.CHANGE_TO_BA3_ALARM )
      I_Contact( #MODE_GROUP_BA_DB.CHANGE_TO_BA5_ALARM )
      Contact( #O_BYTE_0.CHANGE_MODE_SEOC_ALARM )
      wire#w2
      Coil( #MODE_GROUP_BA_DB.CHANGE_TO_BA1_ALARM )
   END_RUNG
   RUNG wire#powerrail
      Contact( #MODE_GROUP_BA_DB.CHANGE_TO_BA1_ALARM )
      I_Contact( #MCH_RESET_FAULTS )
   END_RUNG wire#w1
   RUNG wire#w2
      Coil( #CHANGE_TO_BA1_MODE_WRN )
   END_RUNG
   // the same network as SCL:
   #MODE_GROUP_BA_DB.CHANGE_TO_BA1_ALARM := ((#MODE_GROUP_BA_DB.BA1_REQUEST AND #ANY_MCH_CYCLE_RUN) OR (#MODE_GROUP_BA_DB.CHANGE_TO_BA1_ALARM AND NOT #MCH_RESET_FAULTS)) AND NOT #MODE_GROUP_BA_DB.CHANGE_TO_BA2_ALARM AND NOT #MODE_GROUP_BA_DB.CHANGE_TO_BA3_ALARM AND NOT #MODE_GROUP_BA_DB.CHANGE_TO_BA5_ALARM AND #O_BYTE_0.CHANGE_MODE_SEOC_ALARM;
   #CHANGE_TO_BA1_MODE_WRN := #MODE_GROUP_BA_DB.CHANGE_TO_BA1_ALARM;
END_REGION

REGION Network 19: CHANGE TO BA2 MODE ALARM
   RUNG wire#powerrail
      Contact( #MODE_GROUP_BA_DB.BA2_REQUEST )
      Contact( #ANY_MCH_CYCLE_RUN )
      wire#w1
      I_Contact( #MODE_GROUP_BA_DB.CHANGE_TO_BA1_ALARM )
      I_Contact( #MODE_GROUP_BA_DB.CHANGE_TO_BA3_ALARM )
      I_Contact( #MODE_GROUP_BA_DB.CHANGE_TO_BA5_ALARM )
      Contact( #O_BYTE_0.CHANGE_MODE_SEOC_ALARM )
      wire#w2
      Coil( #MODE_GROUP_BA_DB.CHANGE_TO_BA2_ALARM )
   END_RUNG
   RUNG wire#powerrail
      Contact( #MODE_GROUP_BA_DB.CHANGE_TO_BA2_ALARM )
      I_Contact( #MCH_RESET_FAULTS )
   END_RUNG wire#w1
   RUNG wire#w2
      Coil( #CHANGE_TO_BA2_MODE_WRN )
   END_RUNG
   // the same network as SCL:
   #MODE_GROUP_BA_DB.CHANGE_TO_BA2_ALARM := ((#MODE_GROUP_BA_DB.BA2_REQUEST AND #ANY_MCH_CYCLE_RUN) OR (#MODE_GROUP_BA_DB.CHANGE_TO_BA2_ALARM AND NOT #MCH_RESET_FAULTS)) AND NOT #MODE_GROUP_BA_DB.CHANGE_TO_BA1_ALARM AND NOT #MODE_GROUP_BA_DB.CHANGE_TO_BA3_ALARM AND NOT #MODE_GROUP_BA_DB.CHANGE_TO_BA5_ALARM AND #O_BYTE_0.CHANGE_MODE_SEOC_ALARM;
   #CHANGE_TO_BA2_MODE_WRN := #MODE_GROUP_BA_DB.CHANGE_TO_BA2_ALARM;
END_REGION

REGION Network 20: CHANGE TO BA3 MODE ALARM
   RUNG wire#powerrail
      Contact( #MODE_GROUP_BA_DB.BA3_REQUEST )
      Contact( #ANY_MCH_CYCLE_RUN )
      wire#w1
      I_Contact( #MODE_GROUP_BA_DB.CHANGE_TO_BA1_ALARM )
      I_Contact( #MODE_GROUP_BA_DB.CHANGE_TO_BA2_ALARM )
      I_Contact( #MODE_GROUP_BA_DB.CHANGE_TO_BA5_ALARM )
      Contact( #O_BYTE_0.CHANGE_MODE_SEOC_ALARM )
      wire#w2
      Coil( #MODE_GROUP_BA_DB.CHANGE_TO_BA3_ALARM )
   END_RUNG
   RUNG wire#powerrail
      Contact( #MODE_GROUP_BA_DB.CHANGE_TO_BA3_ALARM )
      I_Contact( #MCH_RESET_FAULTS )
   END_RUNG wire#w1
   RUNG wire#w2
      Coil( #CHANGE_TO_BA3_MODE_WRN )
   END_RUNG
   // the same network as SCL:
   #MODE_GROUP_BA_DB.CHANGE_TO_BA3_ALARM := ((#MODE_GROUP_BA_DB.BA3_REQUEST AND #ANY_MCH_CYCLE_RUN) OR (#MODE_GROUP_BA_DB.CHANGE_TO_BA3_ALARM AND NOT #MCH_RESET_FAULTS)) AND NOT #MODE_GROUP_BA_DB.CHANGE_TO_BA1_ALARM AND NOT #MODE_GROUP_BA_DB.CHANGE_TO_BA2_ALARM AND NOT #MODE_GROUP_BA_DB.CHANGE_TO_BA5_ALARM AND #O_BYTE_0.CHANGE_MODE_SEOC_ALARM;
   #CHANGE_TO_BA3_MODE_WRN := #MODE_GROUP_BA_DB.CHANGE_TO_BA3_ALARM;
END_REGION

REGION Network 21: CHANGE TO BA5 MODE ALARM
   RUNG wire#powerrail
      Contact( #MODE_GROUP_BA_DB.BA5_REQUEST )
      Contact( #ANY_MCH_CYCLE_RUN )
      wire#w1
      I_Contact( #MODE_GROUP_BA_DB.CHANGE_TO_BA1_ALARM )
      I_Contact( #MODE_GROUP_BA_DB.CHANGE_TO_BA2_ALARM )
      I_Contact( #MODE_GROUP_BA_DB.CHANGE_TO_BA3_ALARM )
      Contact( #O_BYTE_0.CHANGE_MODE_SEOC_ALARM )
      wire#w2
      Coil( #MODE_GROUP_BA_DB.CHANGE_TO_BA5_ALARM )
   END_RUNG
   RUNG wire#powerrail
      Contact( #MODE_GROUP_BA_DB.CHANGE_TO_BA5_ALARM )
      I_Contact( #MCH_RESET_FAULTS )
   END_RUNG wire#w1
   RUNG wire#w2
      Coil( #CHANGE_TO_BA5_MODE_WRN )
   END_RUNG
   // the same network as SCL:
   #MODE_GROUP_BA_DB.CHANGE_TO_BA5_ALARM := ((#MODE_GROUP_BA_DB.BA5_REQUEST AND #ANY_MCH_CYCLE_RUN) OR (#MODE_GROUP_BA_DB.CHANGE_TO_BA5_ALARM AND NOT #MCH_RESET_FAULTS)) AND NOT #MODE_GROUP_BA_DB.CHANGE_TO_BA1_ALARM AND NOT #MODE_GROUP_BA_DB.CHANGE_TO_BA2_ALARM AND NOT #MODE_GROUP_BA_DB.CHANGE_TO_BA3_ALARM AND #O_BYTE_0.CHANGE_MODE_SEOC_ALARM;
   #CHANGE_TO_BA5_MODE_WRN := #MODE_GROUP_BA_DB.CHANGE_TO_BA5_ALARM;
END_REGION

REGION Network 22: STOP END OF CYCLE WARNINGS
   RUNG wire#powerrail
      I_Contact( #MODE_GROUP_BA_DB.CHANGE_TO_BA1_ALARM )
      I_Contact( #MODE_GROUP_BA_DB.CHANGE_TO_BA2_ALARM )
      I_Contact( #MODE_GROUP_BA_DB.CHANGE_TO_BA3_ALARM )
      I_Contact( #MODE_GROUP_BA_DB.CHANGE_TO_BA5_ALARM )
      Not()
      { S7_GenerateENO := "TRUE" } Move(in := #DB_NUMBER, out1 => "DB440_MACHINE_ALARM_DECODING".GLOBAL_ALARMS_MACHINE.ALARM_DECODING)
      S_Coil( "DB440_MACHINE_ALARM_DECODING".ALARMS_CENTRAL.SEOC_WARNING )
   END_RUNG
   // the same network as SCL:
   // ENO of a box is taken as its EN; it also drops when the box reports an error
   IF NOT (NOT #MODE_GROUP_BA_DB.CHANGE_TO_BA1_ALARM AND NOT #MODE_GROUP_BA_DB.CHANGE_TO_BA2_ALARM AND NOT #MODE_GROUP_BA_DB.CHANGE_TO_BA3_ALARM AND NOT #MODE_GROUP_BA_DB.CHANGE_TO_BA5_ALARM) THEN
       "DB440_MACHINE_ALARM_DECODING".GLOBAL_ALARMS_MACHINE.ALARM_DECODING := #DB_NUMBER;
       "DB440_MACHINE_ALARM_DECODING".ALARMS_CENTRAL.SEOC_WARNING := TRUE;
   END_IF;
END_REGION

REGION Network 23: WARNINGS
   RUNG wire#powerrail
      I_Contact( #MODE_GROUP_BA_DB.NO_BA_SELECTED )
      Not()
      Move(in := #DB_NUMBER, out1 => "DB440_MACHINE_ALARM_DECODING".GLOBAL_ALARMS_MACHINE.WARNING_DECODING)
      wire#w1
      S_Coil( "DB440_MACHINE_ALARM_DECODING".ALARMS_CENTRAL.WARNING )
   END_RUNG
   RUNG wire#w1
      N_Trig( #MODE_GROUP_BA_DB.WARNING_GONE )
      Move(in := 0, out1 => "DB440_MACHINE_ALARM_DECODING".GLOBAL_ALARMS_MACHINE.WARNING_DECODING)
      R_Coil( "DB440_MACHINE_ALARM_DECODING".ALARMS_CENTRAL.WARNING )
   END_RUNG
   // the same network as SCL:
   #_w1 := NOT (NOT #MODE_GROUP_BA_DB.NO_BA_SELECTED);
   IF #_w1 THEN
       "DB440_MACHINE_ALARM_DECODING".GLOBAL_ALARMS_MACHINE.WARNING_DECODING := #DB_NUMBER;
       "DB440_MACHINE_ALARM_DECODING".ALARMS_CENTRAL.WARNING := TRUE;
   END_IF;
   #_w2 := NOT #_w1 AND #MODE_GROUP_BA_DB.WARNING_GONE;   // falling edge
   #MODE_GROUP_BA_DB.WARNING_GONE := #_w1;
   IF #_w2 THEN
       "DB440_MACHINE_ALARM_DECODING".GLOBAL_ALARMS_MACHINE.WARNING_DECODING := 0;
       "DB440_MACHINE_ALARM_DECODING".ALARMS_CENTRAL.WARNING := FALSE;
   END_IF;
END_REGION

REGION Network 24: CHANGE MODE GENERAL CONDITIONS HELP
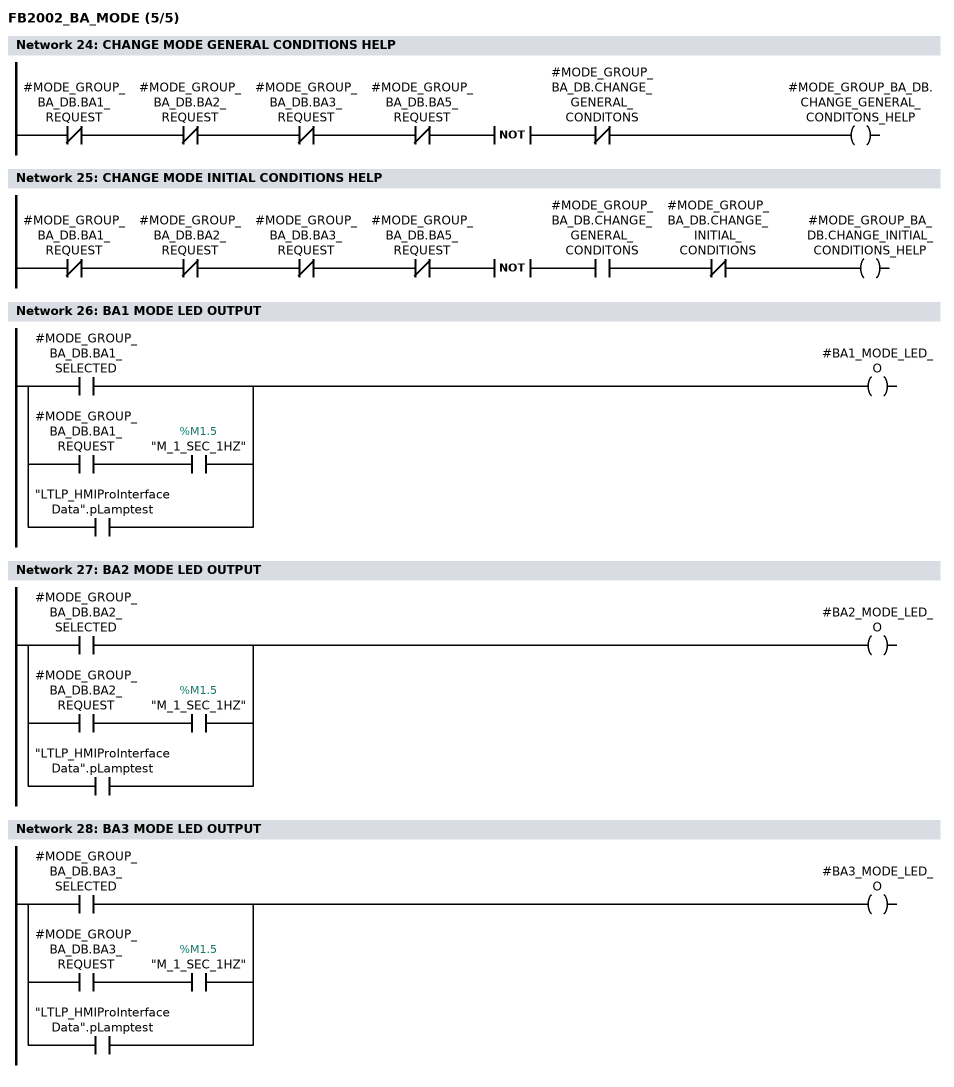
   RUNG wire#powerrail
      I_Contact( #MODE_GROUP_BA_DB.BA1_REQUEST )
      I_Contact( #MODE_GROUP_BA_DB.BA2_REQUEST )
      I_Contact( #MODE_GROUP_BA_DB.BA3_REQUEST )
      I_Contact( #MODE_GROUP_BA_DB.BA5_REQUEST )
      Not()
      I_Contact( #MODE_GROUP_BA_DB.CHANGE_GENERAL_CONDITONS )
      Coil( #MODE_GROUP_BA_DB.CHANGE_GENERAL_CONDITONS_HELP )
   END_RUNG
   // the same network as SCL:
   #MODE_GROUP_BA_DB.CHANGE_GENERAL_CONDITONS_HELP := NOT (NOT #MODE_GROUP_BA_DB.BA1_REQUEST AND NOT #MODE_GROUP_BA_DB.BA2_REQUEST AND NOT #MODE_GROUP_BA_DB.BA3_REQUEST AND NOT #MODE_GROUP_BA_DB.BA5_REQUEST) AND NOT #MODE_GROUP_BA_DB.CHANGE_GENERAL_CONDITONS;
END_REGION

REGION Network 25: CHANGE MODE INITIAL CONDITIONS HELP
   RUNG wire#powerrail
      I_Contact( #MODE_GROUP_BA_DB.BA1_REQUEST )
      I_Contact( #MODE_GROUP_BA_DB.BA2_REQUEST )
      I_Contact( #MODE_GROUP_BA_DB.BA3_REQUEST )
      I_Contact( #MODE_GROUP_BA_DB.BA5_REQUEST )
      Not()
      Contact( #MODE_GROUP_BA_DB.CHANGE_GENERAL_CONDITONS )
      I_Contact( #MODE_GROUP_BA_DB.CHANGE_INITIAL_CONDITIONS )
      Coil( #MODE_GROUP_BA_DB.CHANGE_INITIAL_CONDITIONS_HELP )
   END_RUNG
   // the same network as SCL:
   #MODE_GROUP_BA_DB.CHANGE_INITIAL_CONDITIONS_HELP := NOT (NOT #MODE_GROUP_BA_DB.BA1_REQUEST AND NOT #MODE_GROUP_BA_DB.BA2_REQUEST AND NOT #MODE_GROUP_BA_DB.BA3_REQUEST AND NOT #MODE_GROUP_BA_DB.BA5_REQUEST) AND #MODE_GROUP_BA_DB.CHANGE_GENERAL_CONDITONS AND NOT #MODE_GROUP_BA_DB.CHANGE_INITIAL_CONDITIONS;
END_REGION

REGION Network 26: BA1 MODE LED OUTPUT
   RUNG wire#powerrail
      Contact( #MODE_GROUP_BA_DB.BA1_SELECTED )
      wire#w1
      Coil( #BA1_MODE_LED_O )
   END_RUNG
   RUNG wire#powerrail
      Contact( #MODE_GROUP_BA_DB.BA1_REQUEST )
      Contact( "M_1_SEC_1HZ" )
   END_RUNG wire#w1
   RUNG wire#powerrail
      Contact( "LTLP_HMIProInterfaceData".pLamptest )
   END_RUNG wire#w1
   // the same network as SCL:
   #BA1_MODE_LED_O := #MODE_GROUP_BA_DB.BA1_SELECTED OR (#MODE_GROUP_BA_DB.BA1_REQUEST AND "M_1_SEC_1HZ") OR "LTLP_HMIProInterfaceData".pLamptest;
END_REGION

REGION Network 27: BA2 MODE LED OUTPUT
   RUNG wire#powerrail
      Contact( #MODE_GROUP_BA_DB.BA2_SELECTED )
      wire#w1
      Coil( #BA2_MODE_LED_O )
   END_RUNG
   RUNG wire#powerrail
      Contact( #MODE_GROUP_BA_DB.BA2_REQUEST )
      Contact( "M_1_SEC_1HZ" )
   END_RUNG wire#w1
   RUNG wire#powerrail
      Contact( "LTLP_HMIProInterfaceData".pLamptest )
   END_RUNG wire#w1
   // the same network as SCL:
   #BA2_MODE_LED_O := #MODE_GROUP_BA_DB.BA2_SELECTED OR (#MODE_GROUP_BA_DB.BA2_REQUEST AND "M_1_SEC_1HZ") OR "LTLP_HMIProInterfaceData".pLamptest;
END_REGION

REGION Network 28: BA3 MODE LED OUTPUT
   RUNG wire#powerrail
      Contact( #MODE_GROUP_BA_DB.BA3_SELECTED )
      wire#w1
      Coil( #BA3_MODE_LED_O )
   END_RUNG
   RUNG wire#powerrail
      Contact( #MODE_GROUP_BA_DB.BA3_REQUEST )
      Contact( "M_1_SEC_1HZ" )
   END_RUNG wire#w1
   RUNG wire#powerrail
      Contact( "LTLP_HMIProInterfaceData".pLamptest )
   END_RUNG wire#w1
   // the same network as SCL:
   #BA3_MODE_LED_O := #MODE_GROUP_BA_DB.BA3_SELECTED OR (#MODE_GROUP_BA_DB.BA3_REQUEST AND "M_1_SEC_1HZ") OR "LTLP_HMIProInterfaceData".pLamptest;
END_REGION
END_FUNCTION_BLOCK

FUNCTION_BLOCK "FB2123_PANEL_BUTTON"   // FB2123, LAD
{ S7_Optimized_Access := 'FALSE' }
AUTHOR : ETXETAR
VERSION : 1.0
// stored: AutoNumber false, IsIECCheckEnabled false, SetENOAutomatically false, UDAEnableTagReadback false
   VAR_INPUT
      OPTIONS_0 : Byte := 2#0000_0000;   // OPTIONS 0
      START_CYCLE : Bool;   // START CYCLE / INPUT START CYCLE
      STOP_END_CYCLE : Bool;   // STOP END OF CYCLE / INPUT STOP END CYCLE
      IMMEDIATE_STOP : Bool;   // INMEDIATE STOP / INPUT IMMEDIATE STOP
      EMERGENCY_STOP : Bool;   // EMERGENCY STOP / INPUT EMERGENCY STOP
      HOME_POSITION : Bool;   // INPUT HOME POSITION
      RESET_FAULT : Bool;   // RESET FAULT / INPUT RESET FAULT
      AUTO_SELECTOR : Bool;   // INPUT SELECTOR AUTO SELECTED
      MANUAL_LOAD_SELECTOR : Bool;   // INPUT SELECTOR MANUAL LOAD SELECTED
      LOCK_UNLOCK_GATES : Bool;   // LOCK UNLOCK GATES / INPUT LOCK UNLOCK GATES
      DOOR_LAMP_COND : Bool;   // INPUT DOOR LAMP CONDITIONS
      BHG_BYPASS_GATES : Bool;   // BY PASSED SAFETY GATES MAIN PANEL / INPUT BHG BYPASS GATES
      UNLOAD_PARTS : Bool;   // INPUT UNLOAD FIXTURE PARTS
      UNLOAD_PARTS_FIXT_COND : Bool;   // INPUT UNLOAD PARTS FIXTURE CONDITIONS
      LOAD_PARTS : Bool;   // INPUT LOAD FIXTURE PARTS
      LOAD_PARTS_FIXT_COND : Bool;   // INPUT LOAD PARTS FIXTURE CONDITIONS
   END_VAR
   VAR_OUTPUT
      START_CYCLE_LAMP : Bool;   // START CYCLE LAMP
      END_OF_CYCLE_LAMP : Bool;   // END OF CYCLE LAMP
      HOME_LAMP : Bool;   // HOME POSITION LAMP
      RESET_LAMP : Bool;   // RESET LAMP
      LOCK_DOOR_LAMP : Bool;   // LOCK DOOR LAMP
      UNLOAD_LAMP : Bool;   // UNLOAD PARTS LAMP
      LOAD_LAMP : Bool;   // LOAD PARTS LAMP
      EMERGENCY_STOP_ALARM : Bool;   // EMERGENCY STOP FAULT / EMERGENCY STOP ALARM
   END_VAR
   VAR DB_SPECIFIC
      MANUAL_REQUEST : Bool;   // MANUAL REQUEST
      SEMI_REQUEST : Bool;   // SEMI REQUEST
      AUTO_REQUEST : Bool;   // AUTO REQUEST
      SETUP_REQUEST : Bool;   // SETUP REQUEST
      PARTS_UNLOADED : Bool;   // PARTS UNLOADED
      PARTS_LOADED : Bool;   // PARTS LOADED
      END_OF_CYCLE_ALARM : Bool;   // END OF CYCLE ALARM
      IMMEDIATE_STOP_ALARM : Bool;   // IMMEDIATE STOP ALARM
      HOME_POSITION_ALARM : Bool;   // HOME POSITION ALARM
      SEOC_BY_OPERATOR : Bool;   // STOP END OF CYCLE BY OPERATOR / SEOC BY OPERATOR
      MANUAL_LOADING_SEL_BUTTO : Bool;   // MANUAL LOADING SELECTOR BUTTON / MANUAL LOADING SEL BUTTO
      WARNING_GONE : Bool;   // WARNING GONE
      E_RETURN_PULSE : Bool;   // EMERGENCY RETURN PULSE
      AUX1 : Bool;   // AUX1
      AUX2 : Bool;   // AUX2
      AUX3 : Bool;   // AUX3
      AUX4 : Bool;   // AUX4
      CONDITION_HELP : Bool;   // CONDITION HELP
   END_VAR
   VAR_TEMP
      INPUTS_MASK : Byte;   // INPUT MASK
      O_BYTE_0 : Struct   // OPTIONS BYTE 0
         CHANGE_MODE_WO_PANEL_ACTIVE : Bool;   // CHANGE MODE WITHOUT PANEL ACTIVE OPTION
         MAGAZINE_PANEL : Bool;   // MAGAZINE PANEL OPTION
         PHD_PANEL : Bool;   // PART HANDLING DEVICE PANEL OPTION
         BIMANUAL_PANEL : Bool;   // SPARE OPTION
         SPARE_4 : Bool;   // SPARE OPTION
         SPARE_5 : Bool;   // SPARE OPTION
         SPARE_6 : Bool;   // SPARE OPTION
         SPARE_7 : Bool;   // SPARE OPTION
      END_STRUCT;
      DB_NUMBER : DInt;   // DB NUMBER FOR ALARM AND HELP DECODING
   END_VAR
   VAR_TEMP   // added for the SCL form of the ladder/FBD networks
      _w1 : Bool;
      _w2 : Bool;
      _w3 : Bool;
   END_VAR
BEGIN

NETWORK
TITLE = READ INSTANCE DB
      L     DINO;
      +     10#800000;
      T     #DB_NUMBER;


REGION Network 2: OPTIONS
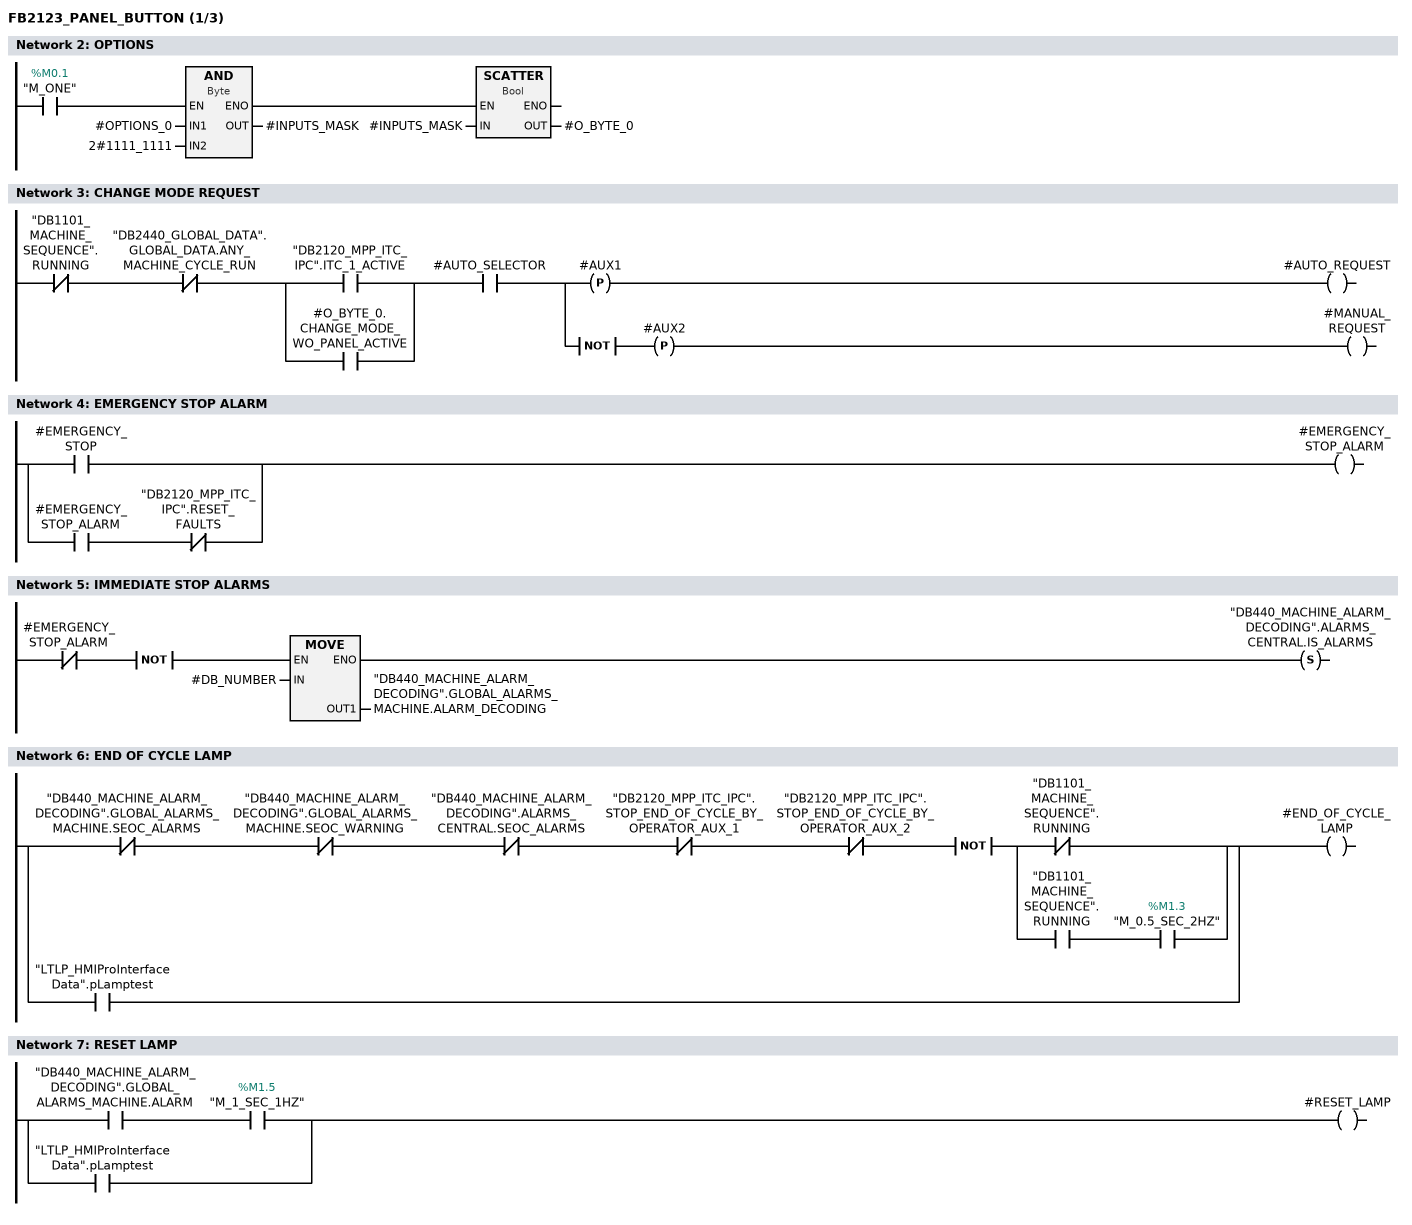
   RUNG wire#powerrail
      Contact( "M_ONE" )
      { S7_Templates := "SrcType := Byte"; S7_GenerateENO := "TRUE" } And(in1 := #OPTIONS_0, in2 := 2#1111_1111, out => #INPUTS_MASK)
      { S7_Templates := "[dest_type := Bool, src_type := Byte]" } SCATTER(IN := #INPUTS_MASK, OUT => #O_BYTE_0)
   END_RUNG
   // the same network as SCL:
   IF "M_ONE" THEN
       #INPUTS_MASK := #OPTIONS_0 AND 2#1111_1111;
       SCATTER(IN := #INPUTS_MASK, OUT => #O_BYTE_0);
   END_IF;
END_REGION

REGION Network 3: CHANGE MODE REQUEST
   RUNG wire#powerrail
      I_Contact( "DB1101_MACHINE_SEQUENCE".RUNNING )
      I_Contact( "DB2440_GLOBAL_DATA".GLOBAL_DATA.ANY_MACHINE_CYCLE_RUN )
      wire#w1
      Contact( "DB2120_MPP_ITC_IPC".ITC_1_ACTIVE )
      wire#w2
      Contact( #AUTO_SELECTOR )
      wire#w3
      P_Trig( #AUX1 )
      Coil( #AUTO_REQUEST )
   END_RUNG
   RUNG wire#w1
      Contact( #O_BYTE_0.CHANGE_MODE_WO_PANEL_ACTIVE )
   END_RUNG wire#w2
   RUNG wire#w3
      Not()
      P_Trig( #AUX2 )
      Coil( #MANUAL_REQUEST )
   END_RUNG
   // the same network as SCL:
   #_w1 := NOT "DB1101_MACHINE_SEQUENCE".RUNNING AND NOT "DB2440_GLOBAL_DATA".GLOBAL_DATA.ANY_MACHINE_CYCLE_RUN AND ("DB2120_MPP_ITC_IPC".ITC_1_ACTIVE OR #O_BYTE_0.CHANGE_MODE_WO_PANEL_ACTIVE) AND #AUTO_SELECTOR;
   #_w2 := #_w1 AND NOT #AUX1;   // rising edge
   #AUX1 := #_w1;
   #AUTO_REQUEST := #_w2;
   #_w3 := NOT #_w1 AND NOT #AUX2;   // rising edge
   #AUX2 := NOT #_w1;
   #MANUAL_REQUEST := #_w3;
END_REGION

REGION Network 4: EMERGENCY STOP ALARM
   RUNG wire#powerrail
      Contact( #EMERGENCY_STOP )
      wire#w1
      Coil( #EMERGENCY_STOP_ALARM )
   END_RUNG
   RUNG wire#powerrail
      Contact( #EMERGENCY_STOP_ALARM )
      I_Contact( "DB2120_MPP_ITC_IPC".RESET_FAULTS )
   END_RUNG wire#w1
   // the same network as SCL:
   #EMERGENCY_STOP_ALARM := #EMERGENCY_STOP OR (#EMERGENCY_STOP_ALARM AND NOT "DB2120_MPP_ITC_IPC".RESET_FAULTS);
END_REGION

REGION Network 5: IMMEDIATE STOP ALARMS
   RUNG wire#powerrail
      I_Contact( #EMERGENCY_STOP_ALARM )
      Not()
      { S7_GenerateENO := "TRUE" } Move(in := #DB_NUMBER, out1 => "DB440_MACHINE_ALARM_DECODING".GLOBAL_ALARMS_MACHINE.ALARM_DECODING)
      S_Coil( "DB440_MACHINE_ALARM_DECODING".ALARMS_CENTRAL.IS_ALARMS )
   END_RUNG
   // the same network as SCL:
   // ENO of a box is taken as its EN; it also drops when the box reports an error
   IF NOT (NOT #EMERGENCY_STOP_ALARM) THEN
       "DB440_MACHINE_ALARM_DECODING".GLOBAL_ALARMS_MACHINE.ALARM_DECODING := #DB_NUMBER;
       "DB440_MACHINE_ALARM_DECODING".ALARMS_CENTRAL.IS_ALARMS := TRUE;
   END_IF;
END_REGION

REGION Network 6: END OF CYCLE LAMP
   RUNG wire#powerrail
      I_Contact( "DB440_MACHINE_ALARM_DECODING".GLOBAL_ALARMS_MACHINE.SEOC_ALARMS )
      I_Contact( "DB440_MACHINE_ALARM_DECODING".GLOBAL_ALARMS_MACHINE.SEOC_WARNING )
      I_Contact( "DB440_MACHINE_ALARM_DECODING".ALARMS_CENTRAL.SEOC_ALARMS )
      I_Contact( "DB2120_MPP_ITC_IPC".STOP_END_OF_CYCLE_BY_OPERATOR_AUX_1 )
      I_Contact( "DB2120_MPP_ITC_IPC".STOP_END_OF_CYCLE_BY_OPERATOR_AUX_2 )
      Not()
      wire#w1
      I_Contact( "DB1101_MACHINE_SEQUENCE".RUNNING )
      wire#w2
      Coil( #END_OF_CYCLE_LAMP )
   END_RUNG
   RUNG wire#w1
      Contact( "DB1101_MACHINE_SEQUENCE".RUNNING )
      Contact( "M_0.5_SEC_2HZ" )
   END_RUNG wire#w2
   RUNG wire#powerrail
      Contact( "LTLP_HMIProInterfaceData".pLamptest )
   END_RUNG wire#w2
   // the same network as SCL:
   #END_OF_CYCLE_LAMP := (NOT (NOT "DB440_MACHINE_ALARM_DECODING".GLOBAL_ALARMS_MACHINE.SEOC_ALARMS AND NOT "DB440_MACHINE_ALARM_DECODING".GLOBAL_ALARMS_MACHINE.SEOC_WARNING AND NOT "DB440_MACHINE_ALARM_DECODING".ALARMS_CENTRAL.SEOC_ALARMS AND NOT "DB2120_MPP_ITC_IPC".STOP_END_OF_CYCLE_BY_OPERATOR_AUX_1 AND NOT "DB2120_MPP_ITC_IPC".STOP_END_OF_CYCLE_BY_OPERATOR_AUX_2) AND (NOT "DB1101_MACHINE_SEQUENCE".RUNNING OR ("DB1101_MACHINE_SEQUENCE".RUNNING AND "M_0.5_SEC_2HZ"))) OR "LTLP_HMIProInterfaceData".pLamptest;
END_REGION

REGION Network 7: RESET LAMP
   RUNG wire#powerrail
      Contact( "DB440_MACHINE_ALARM_DECODING".GLOBAL_ALARMS_MACHINE.ALARM )
      Contact( "M_1_SEC_1HZ" )
      wire#w1
      Coil( #RESET_LAMP )
   END_RUNG
   RUNG wire#powerrail
      Contact( "LTLP_HMIProInterfaceData".pLamptest )
   END_RUNG wire#w1
   // the same network as SCL:
   #RESET_LAMP := ("DB440_MACHINE_ALARM_DECODING".GLOBAL_ALARMS_MACHINE.ALARM AND "M_1_SEC_1HZ") OR "LTLP_HMIProInterfaceData".pLamptest;
END_REGION

REGION Network 8: START CYCLE LAMP
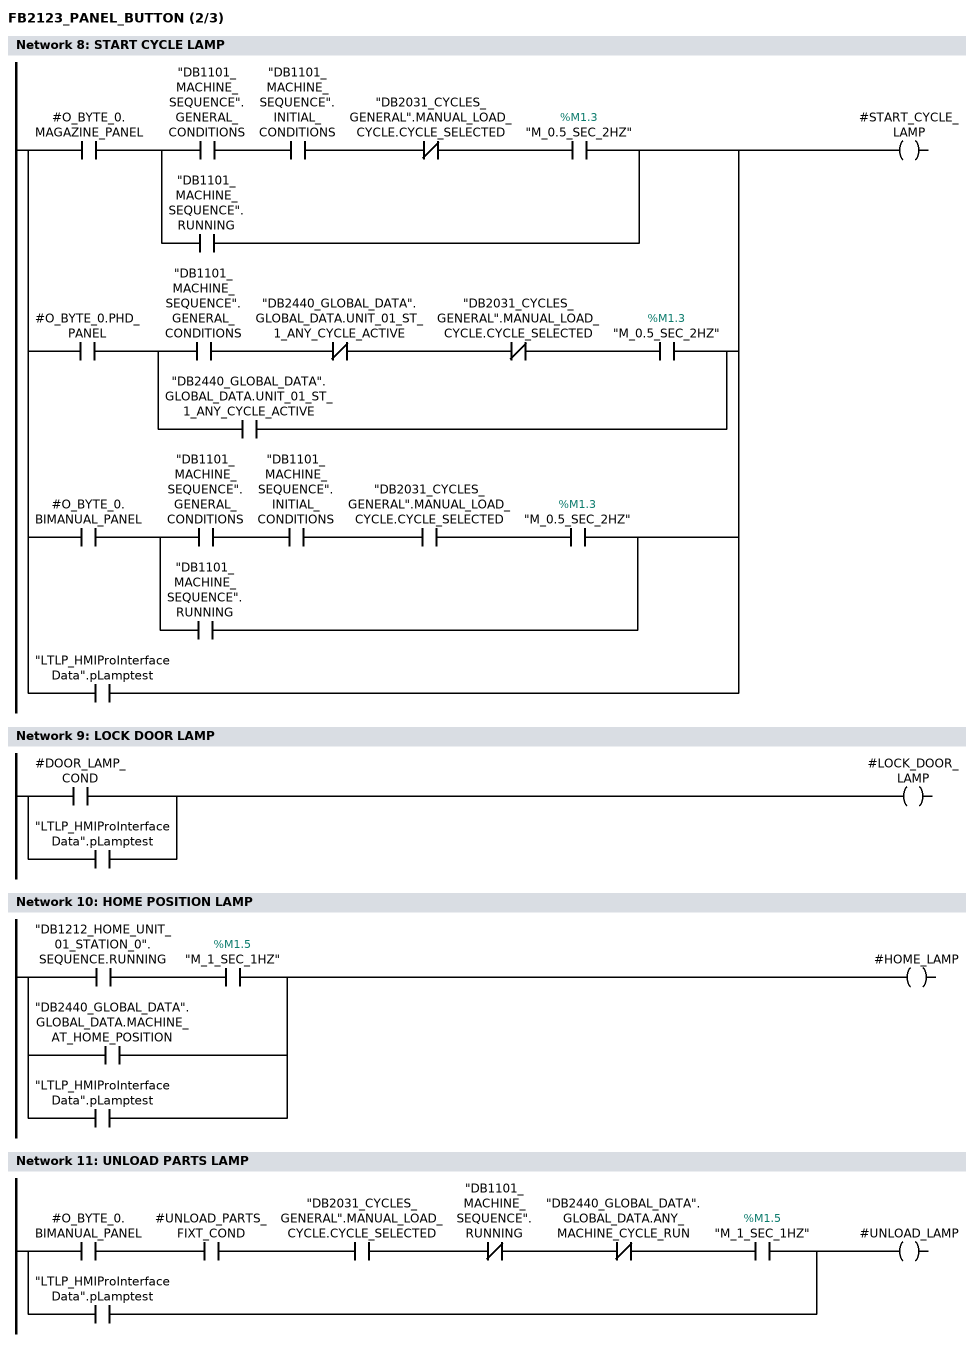
   RUNG wire#powerrail
      Contact( #O_BYTE_0.MAGAZINE_PANEL )
      wire#w1
      Contact( "DB1101_MACHINE_SEQUENCE".GENERAL_CONDITIONS )
      Contact( "DB1101_MACHINE_SEQUENCE".INITIAL_CONDITIONS )
      I_Contact( "DB2031_CYCLES_GENERAL".MANUAL_LOAD_CYCLE.CYCLE_SELECTED )
      Contact( "M_0.5_SEC_2HZ" )
      wire#w2
      Coil( #START_CYCLE_LAMP )
   END_RUNG
   RUNG wire#w1
      Contact( "DB1101_MACHINE_SEQUENCE".RUNNING )
   END_RUNG wire#w2
   RUNG wire#powerrail
      Contact( #O_BYTE_0.PHD_PANEL )
      wire#w3
      Contact( "DB1101_MACHINE_SEQUENCE".GENERAL_CONDITIONS )
      I_Contact( "DB2440_GLOBAL_DATA".GLOBAL_DATA.UNIT_01_ST_1_ANY_CYCLE_ACTIVE )
      I_Contact( "DB2031_CYCLES_GENERAL".MANUAL_LOAD_CYCLE.CYCLE_SELECTED )
      Contact( "M_0.5_SEC_2HZ" )
   END_RUNG wire#w2
   RUNG wire#w3
      Contact( "DB2440_GLOBAL_DATA".GLOBAL_DATA.UNIT_01_ST_1_ANY_CYCLE_ACTIVE )
   END_RUNG wire#w2
   RUNG wire#powerrail
      Contact( #O_BYTE_0.BIMANUAL_PANEL )
      wire#w4
      Contact( "DB1101_MACHINE_SEQUENCE".GENERAL_CONDITIONS )
      Contact( "DB1101_MACHINE_SEQUENCE".INITIAL_CONDITIONS )
      Contact( "DB2031_CYCLES_GENERAL".MANUAL_LOAD_CYCLE.CYCLE_SELECTED )
      Contact( "M_0.5_SEC_2HZ" )
   END_RUNG wire#w2
   RUNG wire#w4
      Contact( "DB1101_MACHINE_SEQUENCE".RUNNING )
   END_RUNG wire#w2
   RUNG wire#powerrail
      Contact( "LTLP_HMIProInterfaceData".pLamptest )
   END_RUNG wire#w2
   // the same network as SCL:
   #START_CYCLE_LAMP := (#O_BYTE_0.MAGAZINE_PANEL AND (("DB1101_MACHINE_SEQUENCE".GENERAL_CONDITIONS AND "DB1101_MACHINE_SEQUENCE".INITIAL_CONDITIONS AND NOT "DB2031_CYCLES_GENERAL".MANUAL_LOAD_CYCLE.CYCLE_SELECTED AND "M_0.5_SEC_2HZ") OR "DB1101_MACHINE_SEQUENCE".RUNNING)) OR (#O_BYTE_0.PHD_PANEL AND (("DB1101_MACHINE_SEQUENCE".GENERAL_CONDITIONS AND NOT "DB2440_GLOBAL_DATA".GLOBAL_DATA.UNIT_01_ST_1_ANY_CYCLE_ACTIVE AND NOT "DB2031_CYCLES_GENERAL".MANUAL_LOAD_CYCLE.CYCLE_SELECTED AND "M_0.5_SEC_2HZ") OR "DB2440_GLOBAL_DATA".GLOBAL_DATA.UNIT_01_ST_1_ANY_CYCLE_ACTIVE)) OR (#O_BYTE_0.BIMANUAL_PANEL AND (("DB1101_MACHINE_SEQUENCE".GENERAL_CONDITIONS AND "DB1101_MACHINE_SEQUENCE".INITIAL_CONDITIONS AND "DB2031_CYCLES_GENERAL".MANUAL_LOAD_CYCLE.CYCLE_SELECTED AND "M_0.5_SEC_2HZ") OR "DB1101_MACHINE_SEQUENCE".RUNNING)) OR "LTLP_HMIProInterfaceData".pLamptest;
END_REGION

REGION Network 9: LOCK DOOR LAMP
   RUNG wire#powerrail
      Contact( #DOOR_LAMP_COND )
      wire#w1
      Coil( #LOCK_DOOR_LAMP )
   END_RUNG
   RUNG wire#powerrail
      Contact( "LTLP_HMIProInterfaceData".pLamptest )
   END_RUNG wire#w1
   // the same network as SCL:
   #LOCK_DOOR_LAMP := #DOOR_LAMP_COND OR "LTLP_HMIProInterfaceData".pLamptest;
END_REGION

REGION Network 10: HOME POSITION LAMP
   RUNG wire#powerrail
      Contact( "DB1212_HOME_UNIT_01_STATION_0".SEQUENCE.RUNNING )
      Contact( "M_1_SEC_1HZ" )
      wire#w1
      Coil( #HOME_LAMP )
   END_RUNG
   RUNG wire#powerrail
      Contact( "DB2440_GLOBAL_DATA".GLOBAL_DATA.MACHINE_AT_HOME_POSITION )
   END_RUNG wire#w1
   RUNG wire#powerrail
      Contact( "LTLP_HMIProInterfaceData".pLamptest )
   END_RUNG wire#w1
   // the same network as SCL:
   #HOME_LAMP := ("DB1212_HOME_UNIT_01_STATION_0".SEQUENCE.RUNNING AND "M_1_SEC_1HZ") OR "DB2440_GLOBAL_DATA".GLOBAL_DATA.MACHINE_AT_HOME_POSITION OR "LTLP_HMIProInterfaceData".pLamptest;
END_REGION

REGION Network 11: UNLOAD PARTS LAMP
   RUNG wire#powerrail
      Contact( #O_BYTE_0.BIMANUAL_PANEL )
      Contact( #UNLOAD_PARTS_FIXT_COND )
      Contact( "DB2031_CYCLES_GENERAL".MANUAL_LOAD_CYCLE.CYCLE_SELECTED )
      I_Contact( "DB1101_MACHINE_SEQUENCE".RUNNING )
      I_Contact( "DB2440_GLOBAL_DATA".GLOBAL_DATA.ANY_MACHINE_CYCLE_RUN )
      Contact( "M_1_SEC_1HZ" )
      wire#w1
      Coil( #UNLOAD_LAMP )
   END_RUNG
   RUNG wire#powerrail
      Contact( "LTLP_HMIProInterfaceData".pLamptest )
   END_RUNG wire#w1
   // the same network as SCL:
   #UNLOAD_LAMP := (#O_BYTE_0.BIMANUAL_PANEL AND #UNLOAD_PARTS_FIXT_COND AND "DB2031_CYCLES_GENERAL".MANUAL_LOAD_CYCLE.CYCLE_SELECTED AND NOT "DB1101_MACHINE_SEQUENCE".RUNNING AND NOT "DB2440_GLOBAL_DATA".GLOBAL_DATA.ANY_MACHINE_CYCLE_RUN AND "M_1_SEC_1HZ") OR "LTLP_HMIProInterfaceData".pLamptest;
END_REGION

REGION Network 12: LOAD PARTS LAMP
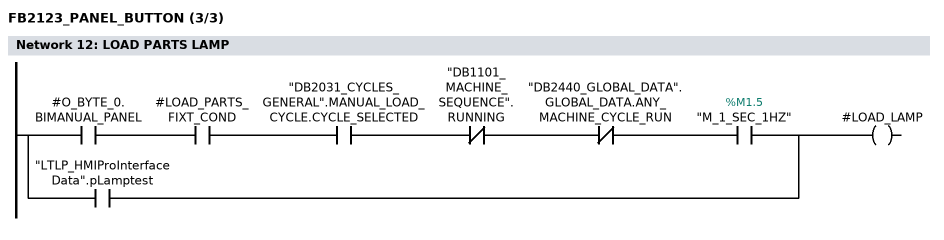
   RUNG wire#powerrail
      Contact( #O_BYTE_0.BIMANUAL_PANEL )
      Contact( #LOAD_PARTS_FIXT_COND )
      Contact( "DB2031_CYCLES_GENERAL".MANUAL_LOAD_CYCLE.CYCLE_SELECTED )
      I_Contact( "DB1101_MACHINE_SEQUENCE".RUNNING )
      I_Contact( "DB2440_GLOBAL_DATA".GLOBAL_DATA.ANY_MACHINE_CYCLE_RUN )
      Contact( "M_1_SEC_1HZ" )
      wire#w1
      Coil( #LOAD_LAMP )
   END_RUNG
   RUNG wire#powerrail
      Contact( "LTLP_HMIProInterfaceData".pLamptest )
   END_RUNG wire#w1
   // the same network as SCL:
   #LOAD_LAMP := (#O_BYTE_0.BIMANUAL_PANEL AND #LOAD_PARTS_FIXT_COND AND "DB2031_CYCLES_GENERAL".MANUAL_LOAD_CYCLE.CYCLE_SELECTED AND NOT "DB1101_MACHINE_SEQUENCE".RUNNING AND NOT "DB2440_GLOBAL_DATA".GLOBAL_DATA.ANY_MACHINE_CYCLE_RUN AND "M_1_SEC_1HZ") OR "LTLP_HMIProInterfaceData".pLamptest;
END_REGION
END_FUNCTION_BLOCK

FUNCTION "FC2101_LINE_CONTACTOR" : Void   // FC2101, LAD
{ S7_Optimized_Access := 'FALSE' }
AUTHOR : ETXETAR
VERSION : 1.0
// stored: AutoNumber false, IsIECCheckEnabled false, SetENOAutomatically false, UDAEnableTagReadback false
   VAR CONSTANT
      FC_NUMBER : DInt := 2101;   // FC NUMBER
   END_VAR
   VAR_TEMP   // added for the SCL form of the ladder/FBD networks
      _w1 : Bool;
      _w2 : Bool;
   END_VAR
BEGIN

REGION Network 1: OPTIONS OFF
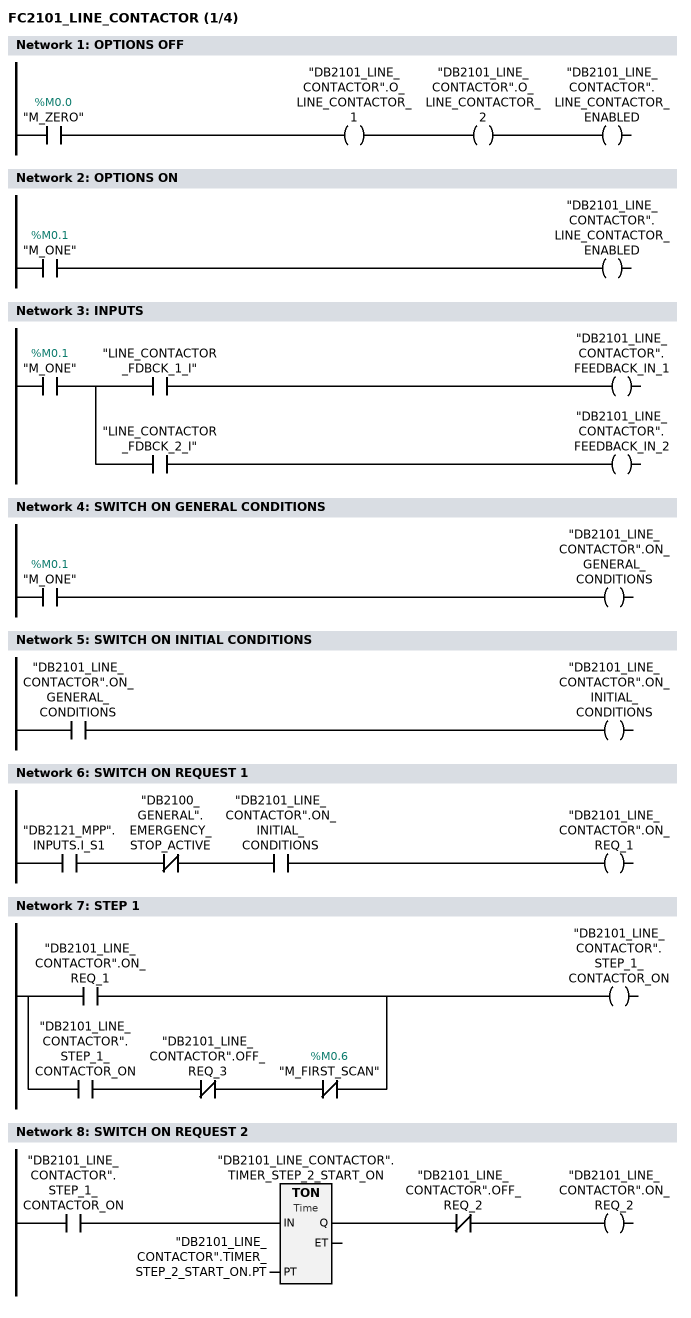
   RUNG wire#powerrail
      Contact( "M_ZERO" )
      Coil( "DB2101_LINE_CONTACTOR".O_LINE_CONTACTOR_1 )
      Coil( "DB2101_LINE_CONTACTOR".O_LINE_CONTACTOR_2 )
      Coil( "DB2101_LINE_CONTACTOR".LINE_CONTACTOR_ENABLED )
   END_RUNG
   // the same network as SCL:
   "DB2101_LINE_CONTACTOR".O_LINE_CONTACTOR_1 := "M_ZERO";
   "DB2101_LINE_CONTACTOR".O_LINE_CONTACTOR_2 := "M_ZERO";
   "DB2101_LINE_CONTACTOR".LINE_CONTACTOR_ENABLED := "M_ZERO";
END_REGION

REGION Network 2: OPTIONS ON
   RUNG wire#powerrail
      Contact( "M_ONE" )
      Coil( "DB2101_LINE_CONTACTOR".LINE_CONTACTOR_ENABLED )
   END_RUNG
   // the same network as SCL:
   "DB2101_LINE_CONTACTOR".LINE_CONTACTOR_ENABLED := "M_ONE";
END_REGION

REGION Network 3: INPUTS
   RUNG wire#powerrail
      Contact( "M_ONE" )
      wire#w1
      Contact( "LINE_CONTACTOR_FDBCK_1_I" )
      Coil( "DB2101_LINE_CONTACTOR".FEEDBACK_IN_1 )
   END_RUNG
   RUNG wire#w1
      Contact( "LINE_CONTACTOR_FDBCK_2_I" )
      Coil( "DB2101_LINE_CONTACTOR".FEEDBACK_IN_2 )
   END_RUNG
   // the same network as SCL:
   "DB2101_LINE_CONTACTOR".FEEDBACK_IN_1 := "M_ONE" AND "LINE_CONTACTOR_FDBCK_1_I";
   "DB2101_LINE_CONTACTOR".FEEDBACK_IN_2 := "M_ONE" AND "LINE_CONTACTOR_FDBCK_2_I";
END_REGION

REGION Network 4: SWITCH ON GENERAL CONDITIONS
   RUNG wire#powerrail
      Contact( "M_ONE" )
      Coil( "DB2101_LINE_CONTACTOR".ON_GENERAL_CONDITIONS )
   END_RUNG
   // the same network as SCL:
   "DB2101_LINE_CONTACTOR".ON_GENERAL_CONDITIONS := "M_ONE";
END_REGION

REGION Network 5: SWITCH ON INITIAL CONDITIONS
   RUNG wire#powerrail
      Contact( "DB2101_LINE_CONTACTOR".ON_GENERAL_CONDITIONS )
      Coil( "DB2101_LINE_CONTACTOR".ON_INITIAL_CONDITIONS )
   END_RUNG
   // the same network as SCL:
   "DB2101_LINE_CONTACTOR".ON_INITIAL_CONDITIONS := "DB2101_LINE_CONTACTOR".ON_GENERAL_CONDITIONS;
END_REGION

REGION Network 6: SWITCH ON REQUEST 1
   RUNG wire#powerrail
      Contact( "DB2121_MPP".INPUTS.I_S1 )
      I_Contact( "DB2100_GENERAL".EMERGENCY_STOP_ACTIVE )
      Contact( "DB2101_LINE_CONTACTOR".ON_INITIAL_CONDITIONS )
      Coil( "DB2101_LINE_CONTACTOR".ON_REQ_1 )
   END_RUNG
   // the same network as SCL:
   "DB2101_LINE_CONTACTOR".ON_REQ_1 := "DB2121_MPP".INPUTS.I_S1 AND NOT "DB2100_GENERAL".EMERGENCY_STOP_ACTIVE AND "DB2101_LINE_CONTACTOR".ON_INITIAL_CONDITIONS;
END_REGION

REGION Network 7: STEP 1
   RUNG wire#powerrail
      Contact( "DB2101_LINE_CONTACTOR".ON_REQ_1 )
      wire#w1
      Coil( "DB2101_LINE_CONTACTOR".STEP_1_CONTACTOR_ON )
   END_RUNG
   RUNG wire#powerrail
      Contact( "DB2101_LINE_CONTACTOR".STEP_1_CONTACTOR_ON )
      I_Contact( "DB2101_LINE_CONTACTOR".OFF_REQ_3 )
      I_Contact( "M_FIRST_SCAN" )
   END_RUNG wire#w1
   // the same network as SCL:
   "DB2101_LINE_CONTACTOR".STEP_1_CONTACTOR_ON := "DB2101_LINE_CONTACTOR".ON_REQ_1 OR ("DB2101_LINE_CONTACTOR".STEP_1_CONTACTOR_ON AND NOT "DB2101_LINE_CONTACTOR".OFF_REQ_3 AND NOT "M_FIRST_SCAN");
END_REGION

REGION Network 8: SWITCH ON REQUEST 2
   RUNG wire#powerrail
      Contact( "DB2101_LINE_CONTACTOR".STEP_1_CONTACTOR_ON )
      { S7_Templates := "time_type := Time" } "DB2101_LINE_CONTACTOR".TIMER_STEP_2_START_ON.TON(pt := "DB2101_LINE_CONTACTOR".TIMER_STEP_2_START_ON.PT, et =>)
      I_Contact( "DB2101_LINE_CONTACTOR".OFF_REQ_2 )
      Coil( "DB2101_LINE_CONTACTOR".ON_REQ_2 )
   END_RUNG
   // the same network as SCL:
   "DB2101_LINE_CONTACTOR".TIMER_STEP_2_START_ON.TON(IN := "DB2101_LINE_CONTACTOR".STEP_1_CONTACTOR_ON,
                           PT := "DB2101_LINE_CONTACTOR".TIMER_STEP_2_START_ON.PT);
   "DB2101_LINE_CONTACTOR".ON_REQ_2 := "DB2101_LINE_CONTACTOR".TIMER_STEP_2_START_ON.Q AND NOT "DB2101_LINE_CONTACTOR".OFF_REQ_2;
END_REGION

REGION Network 9: STEP 2
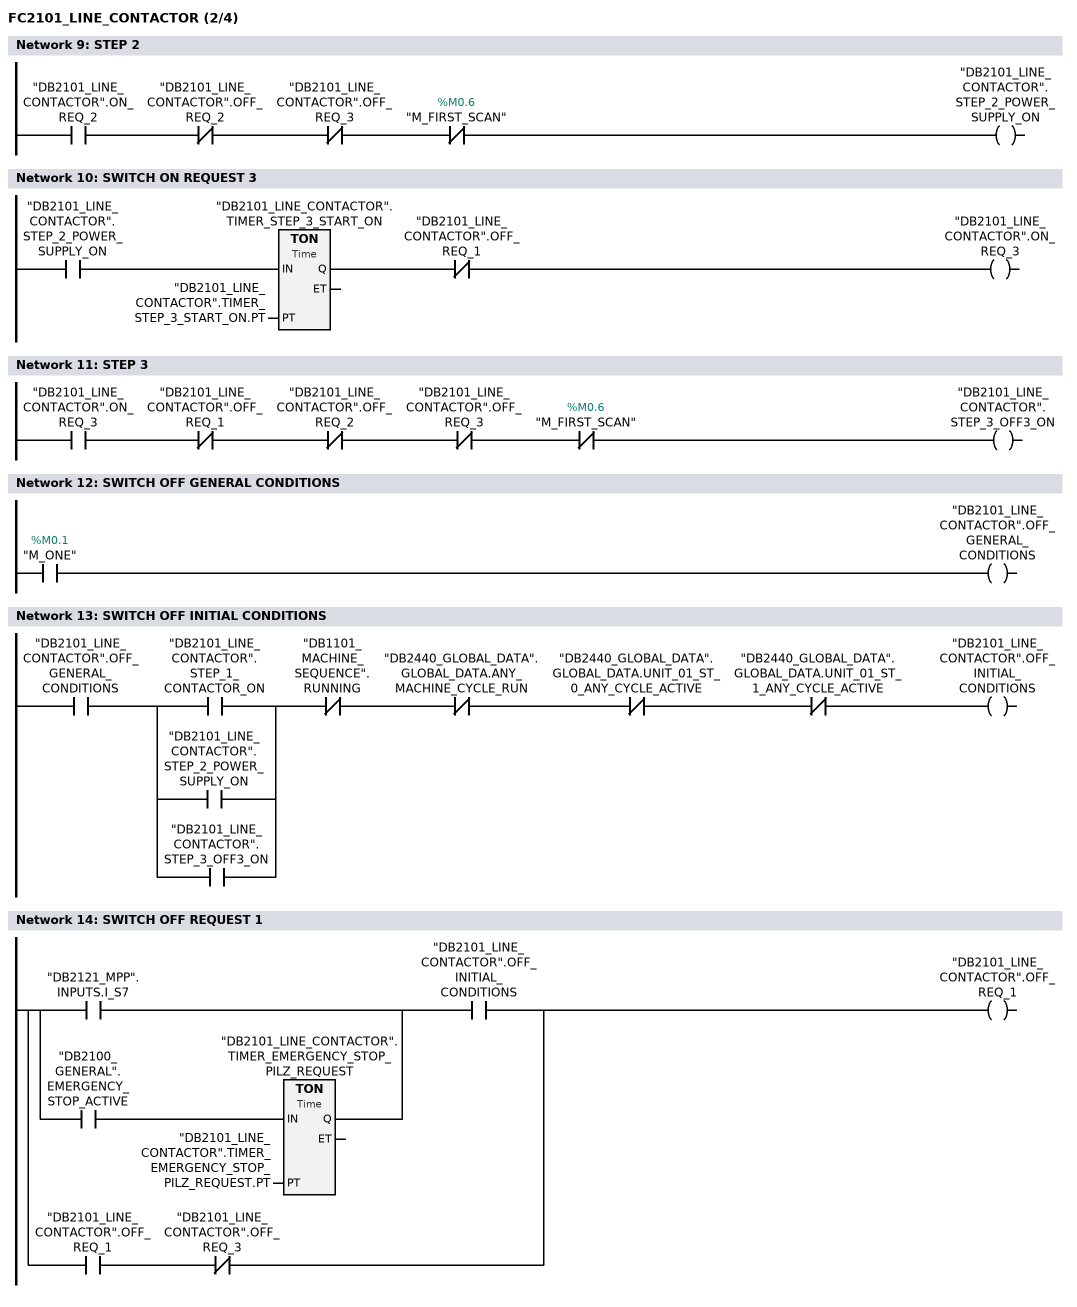
   RUNG wire#powerrail
      Contact( "DB2101_LINE_CONTACTOR".ON_REQ_2 )
      I_Contact( "DB2101_LINE_CONTACTOR".OFF_REQ_2 )
      I_Contact( "DB2101_LINE_CONTACTOR".OFF_REQ_3 )
      I_Contact( "M_FIRST_SCAN" )
      Coil( "DB2101_LINE_CONTACTOR".STEP_2_POWER_SUPPLY_ON )
   END_RUNG
   // the same network as SCL:
   "DB2101_LINE_CONTACTOR".STEP_2_POWER_SUPPLY_ON := "DB2101_LINE_CONTACTOR".ON_REQ_2 AND NOT "DB2101_LINE_CONTACTOR".OFF_REQ_2 AND NOT "DB2101_LINE_CONTACTOR".OFF_REQ_3 AND NOT "M_FIRST_SCAN";
END_REGION

REGION Network 10: SWITCH ON REQUEST 3
   RUNG wire#powerrail
      Contact( "DB2101_LINE_CONTACTOR".STEP_2_POWER_SUPPLY_ON )
      { S7_Templates := "time_type := Time" } "DB2101_LINE_CONTACTOR".TIMER_STEP_3_START_ON.TON(pt := "DB2101_LINE_CONTACTOR".TIMER_STEP_3_START_ON.PT, et =>)
      I_Contact( "DB2101_LINE_CONTACTOR".OFF_REQ_1 )
      Coil( "DB2101_LINE_CONTACTOR".ON_REQ_3 )
   END_RUNG
   // the same network as SCL:
   "DB2101_LINE_CONTACTOR".TIMER_STEP_3_START_ON.TON(IN := "DB2101_LINE_CONTACTOR".STEP_2_POWER_SUPPLY_ON,
                           PT := "DB2101_LINE_CONTACTOR".TIMER_STEP_3_START_ON.PT);
   "DB2101_LINE_CONTACTOR".ON_REQ_3 := "DB2101_LINE_CONTACTOR".TIMER_STEP_3_START_ON.Q AND NOT "DB2101_LINE_CONTACTOR".OFF_REQ_1;
END_REGION

REGION Network 11: STEP 3
   RUNG wire#powerrail
      Contact( "DB2101_LINE_CONTACTOR".ON_REQ_3 )
      I_Contact( "DB2101_LINE_CONTACTOR".OFF_REQ_1 )
      I_Contact( "DB2101_LINE_CONTACTOR".OFF_REQ_2 )
      I_Contact( "DB2101_LINE_CONTACTOR".OFF_REQ_3 )
      I_Contact( "M_FIRST_SCAN" )
      Coil( "DB2101_LINE_CONTACTOR".STEP_3_OFF3_ON )
   END_RUNG
   // the same network as SCL:
   "DB2101_LINE_CONTACTOR".STEP_3_OFF3_ON := "DB2101_LINE_CONTACTOR".ON_REQ_3 AND NOT "DB2101_LINE_CONTACTOR".OFF_REQ_1 AND NOT "DB2101_LINE_CONTACTOR".OFF_REQ_2 AND NOT "DB2101_LINE_CONTACTOR".OFF_REQ_3 AND NOT "M_FIRST_SCAN";
END_REGION

REGION Network 12: SWITCH OFF GENERAL CONDITIONS
   RUNG wire#powerrail
      Contact( "M_ONE" )
      Coil( "DB2101_LINE_CONTACTOR".OFF_GENERAL_CONDITIONS )
   END_RUNG
   // the same network as SCL:
   "DB2101_LINE_CONTACTOR".OFF_GENERAL_CONDITIONS := "M_ONE";
END_REGION

REGION Network 13: SWITCH OFF INITIAL CONDITIONS
   RUNG wire#powerrail
      Contact( "DB2101_LINE_CONTACTOR".OFF_GENERAL_CONDITIONS )
      wire#w1
      Contact( "DB2101_LINE_CONTACTOR".STEP_1_CONTACTOR_ON )
      wire#w2
      I_Contact( "DB1101_MACHINE_SEQUENCE".RUNNING )
      I_Contact( "DB2440_GLOBAL_DATA".GLOBAL_DATA.ANY_MACHINE_CYCLE_RUN )
      I_Contact( "DB2440_GLOBAL_DATA".GLOBAL_DATA.UNIT_01_ST_0_ANY_CYCLE_ACTIVE )
      I_Contact( "DB2440_GLOBAL_DATA".GLOBAL_DATA.UNIT_01_ST_1_ANY_CYCLE_ACTIVE )
      Coil( "DB2101_LINE_CONTACTOR".OFF_INITIAL_CONDITIONS )
   END_RUNG
   RUNG wire#w1
      Contact( "DB2101_LINE_CONTACTOR".STEP_2_POWER_SUPPLY_ON )
   END_RUNG wire#w2
   RUNG wire#w1
      Contact( "DB2101_LINE_CONTACTOR".STEP_3_OFF3_ON )
   END_RUNG wire#w2
   // the same network as SCL:
   "DB2101_LINE_CONTACTOR".OFF_INITIAL_CONDITIONS := "DB2101_LINE_CONTACTOR".OFF_GENERAL_CONDITIONS AND ("DB2101_LINE_CONTACTOR".STEP_1_CONTACTOR_ON OR "DB2101_LINE_CONTACTOR".STEP_2_POWER_SUPPLY_ON OR "DB2101_LINE_CONTACTOR".STEP_3_OFF3_ON) AND NOT "DB1101_MACHINE_SEQUENCE".RUNNING AND NOT "DB2440_GLOBAL_DATA".GLOBAL_DATA.ANY_MACHINE_CYCLE_RUN AND NOT "DB2440_GLOBAL_DATA".GLOBAL_DATA.UNIT_01_ST_0_ANY_CYCLE_ACTIVE AND NOT "DB2440_GLOBAL_DATA".GLOBAL_DATA.UNIT_01_ST_1_ANY_CYCLE_ACTIVE;
END_REGION

REGION Network 14: SWITCH OFF REQUEST 1
   RUNG wire#powerrail
      Contact( "DB2121_MPP".INPUTS.I_S7 )
      wire#w1
      Contact( "DB2101_LINE_CONTACTOR".OFF_INITIAL_CONDITIONS )
      wire#w2
      Coil( "DB2101_LINE_CONTACTOR".OFF_REQ_1 )
   END_RUNG
   RUNG wire#powerrail
      Contact( "DB2100_GENERAL".EMERGENCY_STOP_ACTIVE )
      { S7_Templates := "time_type := Time" } "DB2101_LINE_CONTACTOR".TIMER_EMERGENCY_STOP_PILZ_REQUEST.TON(pt := "DB2101_LINE_CONTACTOR".TIMER_EMERGENCY_STOP_PILZ_REQUEST.PT, et =>)
   END_RUNG wire#w1
   RUNG wire#powerrail
      Contact( "DB2101_LINE_CONTACTOR".OFF_REQ_1 )
      I_Contact( "DB2101_LINE_CONTACTOR".OFF_REQ_3 )
   END_RUNG wire#w2
   // the same network as SCL:
   "DB2101_LINE_CONTACTOR".TIMER_EMERGENCY_STOP_PILZ_REQUEST.TON(IN := "DB2100_GENERAL".EMERGENCY_STOP_ACTIVE,
                           PT := "DB2101_LINE_CONTACTOR".TIMER_EMERGENCY_STOP_PILZ_REQUEST.PT);
   "DB2101_LINE_CONTACTOR".OFF_REQ_1 := (("DB2121_MPP".INPUTS.I_S7 OR "DB2101_LINE_CONTACTOR".TIMER_EMERGENCY_STOP_PILZ_REQUEST.Q) AND "DB2101_LINE_CONTACTOR".OFF_INITIAL_CONDITIONS) OR ("DB2101_LINE_CONTACTOR".OFF_REQ_1 AND NOT "DB2101_LINE_CONTACTOR".OFF_REQ_3);
END_REGION

REGION Network 15: SWITCH OFF REQUEST 2
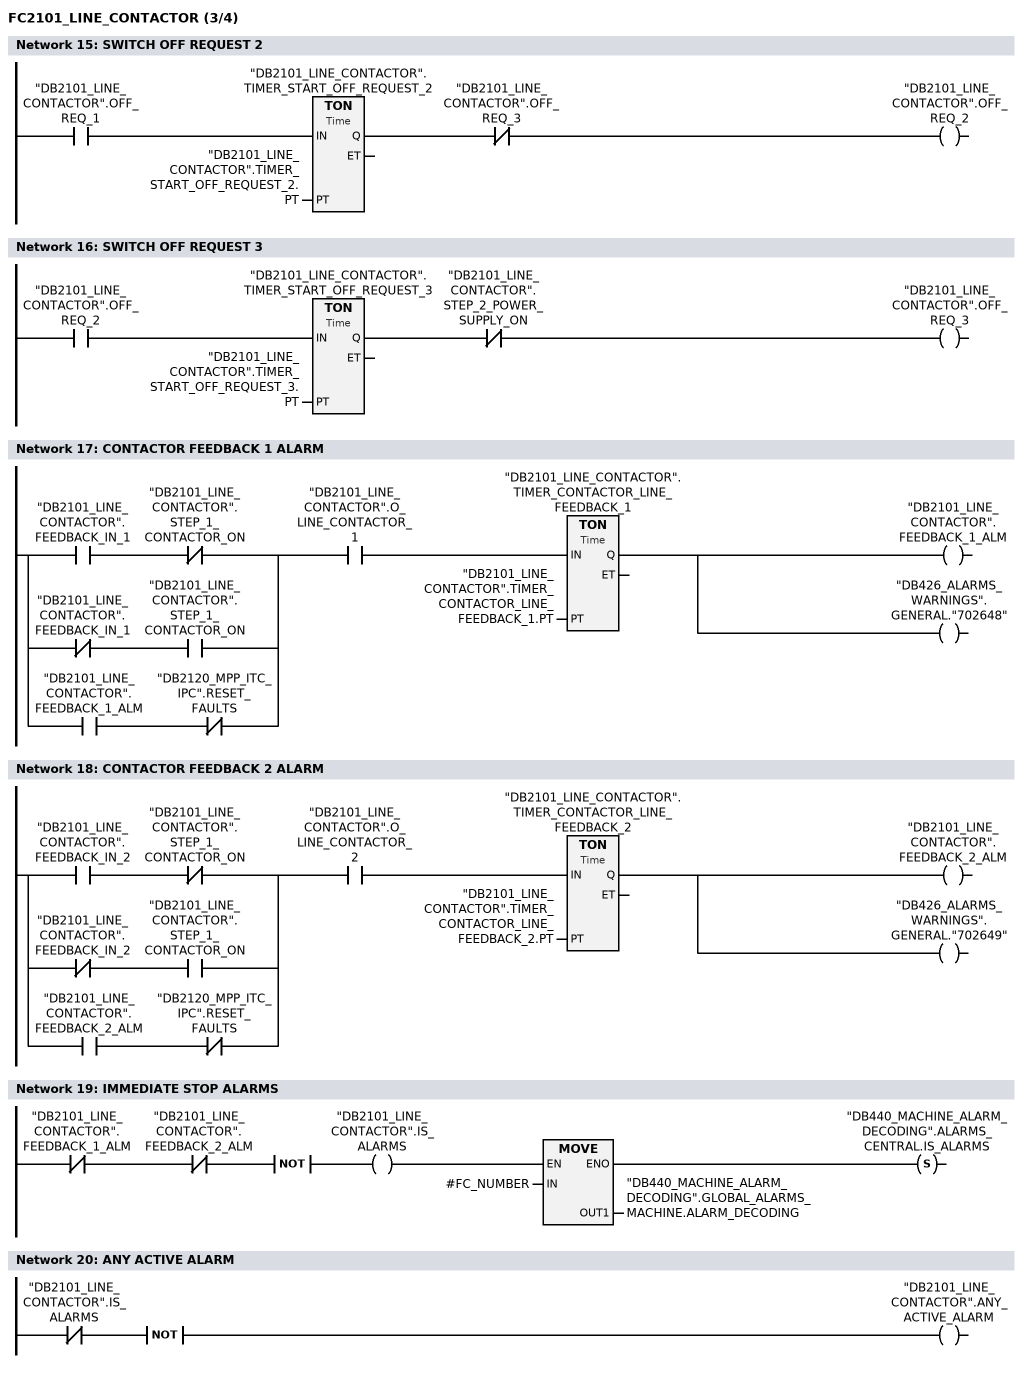
   RUNG wire#powerrail
      Contact( "DB2101_LINE_CONTACTOR".OFF_REQ_1 )
      { S7_Templates := "time_type := Time" } "DB2101_LINE_CONTACTOR".TIMER_START_OFF_REQUEST_2.TON(pt := "DB2101_LINE_CONTACTOR".TIMER_START_OFF_REQUEST_2.PT, et =>)
      I_Contact( "DB2101_LINE_CONTACTOR".OFF_REQ_3 )
      Coil( "DB2101_LINE_CONTACTOR".OFF_REQ_2 )
   END_RUNG
   // the same network as SCL:
   "DB2101_LINE_CONTACTOR".TIMER_START_OFF_REQUEST_2.TON(IN := "DB2101_LINE_CONTACTOR".OFF_REQ_1,
                           PT := "DB2101_LINE_CONTACTOR".TIMER_START_OFF_REQUEST_2.PT);
   "DB2101_LINE_CONTACTOR".OFF_REQ_2 := "DB2101_LINE_CONTACTOR".TIMER_START_OFF_REQUEST_2.Q AND NOT "DB2101_LINE_CONTACTOR".OFF_REQ_3;
END_REGION

REGION Network 16: SWITCH OFF REQUEST 3
   RUNG wire#powerrail
      Contact( "DB2101_LINE_CONTACTOR".OFF_REQ_2 )
      { S7_Templates := "time_type := Time" } "DB2101_LINE_CONTACTOR".TIMER_START_OFF_REQUEST_3.TON(pt := "DB2101_LINE_CONTACTOR".TIMER_START_OFF_REQUEST_3.PT, et =>)
      I_Contact( "DB2101_LINE_CONTACTOR".STEP_2_POWER_SUPPLY_ON )
      Coil( "DB2101_LINE_CONTACTOR".OFF_REQ_3 )
   END_RUNG
   // the same network as SCL:
   "DB2101_LINE_CONTACTOR".TIMER_START_OFF_REQUEST_3.TON(IN := "DB2101_LINE_CONTACTOR".OFF_REQ_2,
                           PT := "DB2101_LINE_CONTACTOR".TIMER_START_OFF_REQUEST_3.PT);
   "DB2101_LINE_CONTACTOR".OFF_REQ_3 := "DB2101_LINE_CONTACTOR".TIMER_START_OFF_REQUEST_3.Q AND NOT "DB2101_LINE_CONTACTOR".STEP_2_POWER_SUPPLY_ON;
END_REGION

REGION Network 17: CONTACTOR FEEDBACK 1 ALARM
   RUNG wire#powerrail
      Contact( "DB2101_LINE_CONTACTOR".FEEDBACK_IN_1 )
      I_Contact( "DB2101_LINE_CONTACTOR".STEP_1_CONTACTOR_ON )
      wire#w1
      Contact( "DB2101_LINE_CONTACTOR".O_LINE_CONTACTOR_1 )
      { S7_Templates := "time_type := Time" } "DB2101_LINE_CONTACTOR".TIMER_CONTACTOR_LINE_FEEDBACK_1.TON(pt := "DB2101_LINE_CONTACTOR".TIMER_CONTACTOR_LINE_FEEDBACK_1.PT, et =>)
      wire#w2
      Coil( "DB2101_LINE_CONTACTOR".FEEDBACK_1_ALM )
   END_RUNG
   RUNG wire#powerrail
      I_Contact( "DB2101_LINE_CONTACTOR".FEEDBACK_IN_1 )
      Contact( "DB2101_LINE_CONTACTOR".STEP_1_CONTACTOR_ON )
   END_RUNG wire#w1
   RUNG wire#powerrail
      Contact( "DB2101_LINE_CONTACTOR".FEEDBACK_1_ALM )
      I_Contact( "DB2120_MPP_ITC_IPC".RESET_FAULTS )
   END_RUNG wire#w1
   RUNG wire#w2
      Coil( "DB426_ALARMS_WARNINGS".GENERAL."702648" )
   END_RUNG
   // the same network as SCL:
   "DB2101_LINE_CONTACTOR".TIMER_CONTACTOR_LINE_FEEDBACK_1.TON(IN := (("DB2101_LINE_CONTACTOR".FEEDBACK_IN_1 AND NOT "DB2101_LINE_CONTACTOR".STEP_1_CONTACTOR_ON) OR (NOT "DB2101_LINE_CONTACTOR".FEEDBACK_IN_1 AND "DB2101_LINE_CONTACTOR".STEP_1_CONTACTOR_ON) OR ("DB2101_LINE_CONTACTOR".FEEDBACK_1_ALM AND NOT "DB2120_MPP_ITC_IPC".RESET_FAULTS)) AND "DB2101_LINE_CONTACTOR".O_LINE_CONTACTOR_1,
                           PT := "DB2101_LINE_CONTACTOR".TIMER_CONTACTOR_LINE_FEEDBACK_1.PT);
   "DB2101_LINE_CONTACTOR".FEEDBACK_1_ALM := "DB2101_LINE_CONTACTOR".TIMER_CONTACTOR_LINE_FEEDBACK_1.Q;
   "DB426_ALARMS_WARNINGS".GENERAL."702648" := "DB2101_LINE_CONTACTOR".TIMER_CONTACTOR_LINE_FEEDBACK_1.Q;
END_REGION

REGION Network 18: CONTACTOR FEEDBACK 2 ALARM
   RUNG wire#powerrail
      Contact( "DB2101_LINE_CONTACTOR".FEEDBACK_IN_2 )
      I_Contact( "DB2101_LINE_CONTACTOR".STEP_1_CONTACTOR_ON )
      wire#w1
      Contact( "DB2101_LINE_CONTACTOR".O_LINE_CONTACTOR_2 )
      { S7_Templates := "time_type := Time" } "DB2101_LINE_CONTACTOR".TIMER_CONTACTOR_LINE_FEEDBACK_2.TON(pt := "DB2101_LINE_CONTACTOR".TIMER_CONTACTOR_LINE_FEEDBACK_2.PT, et =>)
      wire#w2
      Coil( "DB2101_LINE_CONTACTOR".FEEDBACK_2_ALM )
   END_RUNG
   RUNG wire#powerrail
      I_Contact( "DB2101_LINE_CONTACTOR".FEEDBACK_IN_2 )
      Contact( "DB2101_LINE_CONTACTOR".STEP_1_CONTACTOR_ON )
   END_RUNG wire#w1
   RUNG wire#powerrail
      Contact( "DB2101_LINE_CONTACTOR".FEEDBACK_2_ALM )
      I_Contact( "DB2120_MPP_ITC_IPC".RESET_FAULTS )
   END_RUNG wire#w1
   RUNG wire#w2
      Coil( "DB426_ALARMS_WARNINGS".GENERAL."702649" )
   END_RUNG
   // the same network as SCL:
   "DB2101_LINE_CONTACTOR".TIMER_CONTACTOR_LINE_FEEDBACK_2.TON(IN := (("DB2101_LINE_CONTACTOR".FEEDBACK_IN_2 AND NOT "DB2101_LINE_CONTACTOR".STEP_1_CONTACTOR_ON) OR (NOT "DB2101_LINE_CONTACTOR".FEEDBACK_IN_2 AND "DB2101_LINE_CONTACTOR".STEP_1_CONTACTOR_ON) OR ("DB2101_LINE_CONTACTOR".FEEDBACK_2_ALM AND NOT "DB2120_MPP_ITC_IPC".RESET_FAULTS)) AND "DB2101_LINE_CONTACTOR".O_LINE_CONTACTOR_2,
                           PT := "DB2101_LINE_CONTACTOR".TIMER_CONTACTOR_LINE_FEEDBACK_2.PT);
   "DB2101_LINE_CONTACTOR".FEEDBACK_2_ALM := "DB2101_LINE_CONTACTOR".TIMER_CONTACTOR_LINE_FEEDBACK_2.Q;
   "DB426_ALARMS_WARNINGS".GENERAL."702649" := "DB2101_LINE_CONTACTOR".TIMER_CONTACTOR_LINE_FEEDBACK_2.Q;
END_REGION

REGION Network 19: IMMEDIATE STOP ALARMS
   RUNG wire#powerrail
      I_Contact( "DB2101_LINE_CONTACTOR".FEEDBACK_1_ALM )
      I_Contact( "DB2101_LINE_CONTACTOR".FEEDBACK_2_ALM )
      Not()
      Coil( "DB2101_LINE_CONTACTOR".IS_ALARMS )
      Move(in := #FC_NUMBER, out1 => "DB440_MACHINE_ALARM_DECODING".GLOBAL_ALARMS_MACHINE.ALARM_DECODING)
      S_Coil( "DB440_MACHINE_ALARM_DECODING".ALARMS_CENTRAL.IS_ALARMS )
   END_RUNG
   // the same network as SCL:
   "DB2101_LINE_CONTACTOR".IS_ALARMS := NOT (NOT "DB2101_LINE_CONTACTOR".FEEDBACK_1_ALM AND NOT "DB2101_LINE_CONTACTOR".FEEDBACK_2_ALM);
   IF "DB2101_LINE_CONTACTOR".IS_ALARMS THEN
       "DB440_MACHINE_ALARM_DECODING".GLOBAL_ALARMS_MACHINE.ALARM_DECODING := #FC_NUMBER;
       "DB440_MACHINE_ALARM_DECODING".ALARMS_CENTRAL.IS_ALARMS := TRUE;
   END_IF;
END_REGION

REGION Network 20: ANY ACTIVE ALARM
   RUNG wire#powerrail
      I_Contact( "DB2101_LINE_CONTACTOR".IS_ALARMS )
      Not()
      Coil( "DB2101_LINE_CONTACTOR".ANY_ACTIVE_ALARM )
   END_RUNG
   // the same network as SCL:
   "DB2101_LINE_CONTACTOR".ANY_ACTIVE_ALARM := NOT (NOT "DB2101_LINE_CONTACTOR".IS_ALARMS);
END_REGION

REGION Network 21: LINE CONTACTOR NOT SWITCHED ON WARNING
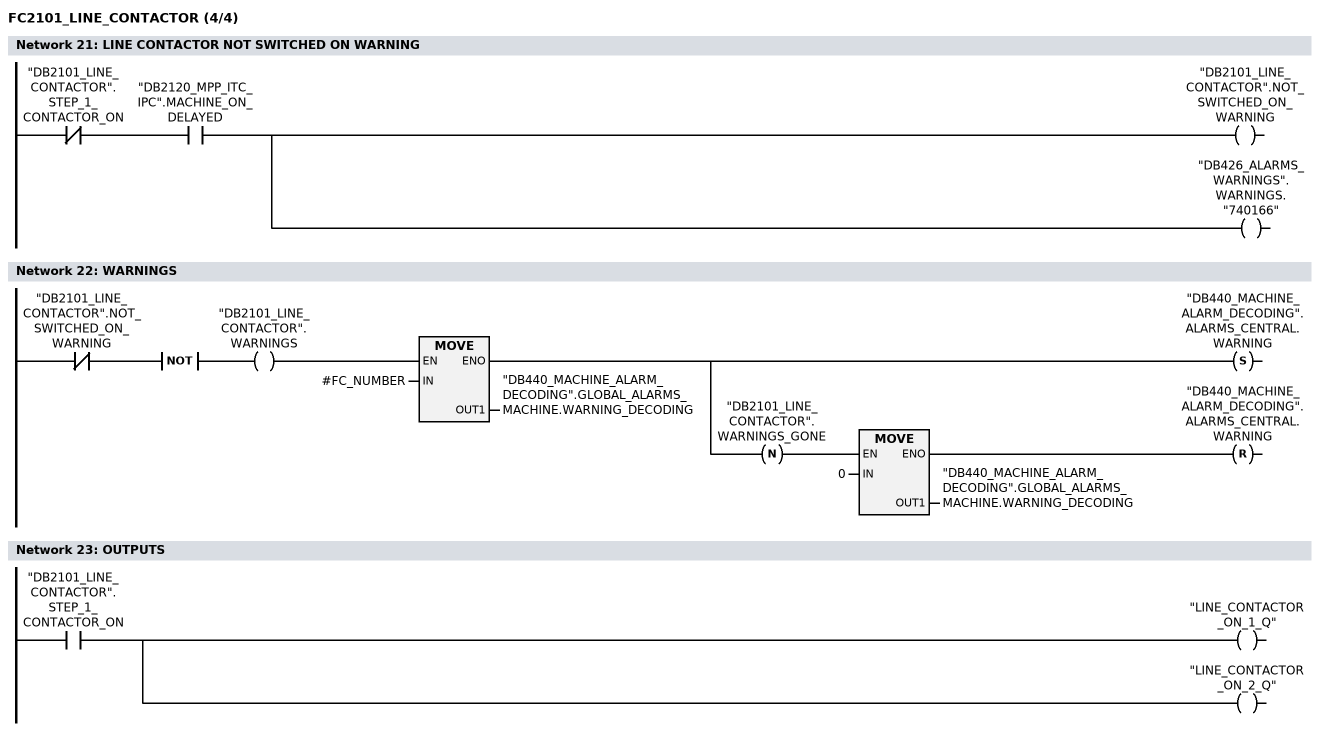
   RUNG wire#powerrail
      I_Contact( "DB2101_LINE_CONTACTOR".STEP_1_CONTACTOR_ON )
      Contact( "DB2120_MPP_ITC_IPC".MACHINE_ON_DELAYED )
      wire#w1
      Coil( "DB2101_LINE_CONTACTOR".NOT_SWITCHED_ON_WARNING )
   END_RUNG
   RUNG wire#w1
      Coil( "DB426_ALARMS_WARNINGS".WARNINGS."740166" )
   END_RUNG
   // the same network as SCL:
   "DB2101_LINE_CONTACTOR".NOT_SWITCHED_ON_WARNING := NOT "DB2101_LINE_CONTACTOR".STEP_1_CONTACTOR_ON AND "DB2120_MPP_ITC_IPC".MACHINE_ON_DELAYED;
   "DB426_ALARMS_WARNINGS".WARNINGS."740166" := "DB2101_LINE_CONTACTOR".NOT_SWITCHED_ON_WARNING;
END_REGION

REGION Network 22: WARNINGS
   RUNG wire#powerrail
      I_Contact( "DB2101_LINE_CONTACTOR".NOT_SWITCHED_ON_WARNING )
      Not()
      Coil( "DB2101_LINE_CONTACTOR".WARNINGS )
      Move(in := #FC_NUMBER, out1 => "DB440_MACHINE_ALARM_DECODING".GLOBAL_ALARMS_MACHINE.WARNING_DECODING)
      wire#w1
      S_Coil( "DB440_MACHINE_ALARM_DECODING".ALARMS_CENTRAL.WARNING )
   END_RUNG
   RUNG wire#w1
      N_Trig( "DB2101_LINE_CONTACTOR".WARNINGS_GONE )
      Move(in := 0, out1 => "DB440_MACHINE_ALARM_DECODING".GLOBAL_ALARMS_MACHINE.WARNING_DECODING)
      R_Coil( "DB440_MACHINE_ALARM_DECODING".ALARMS_CENTRAL.WARNING )
   END_RUNG
   // the same network as SCL:
   "DB2101_LINE_CONTACTOR".WARNINGS := NOT (NOT "DB2101_LINE_CONTACTOR".NOT_SWITCHED_ON_WARNING);
   #_w1 := NOT (NOT "DB2101_LINE_CONTACTOR".NOT_SWITCHED_ON_WARNING);
   IF #_w1 THEN
       "DB440_MACHINE_ALARM_DECODING".GLOBAL_ALARMS_MACHINE.WARNING_DECODING := #FC_NUMBER;
       "DB440_MACHINE_ALARM_DECODING".ALARMS_CENTRAL.WARNING := TRUE;
   END_IF;
   #_w2 := NOT #_w1 AND "DB2101_LINE_CONTACTOR".WARNINGS_GONE;   // falling edge
   "DB2101_LINE_CONTACTOR".WARNINGS_GONE := #_w1;
   IF #_w2 THEN
       "DB440_MACHINE_ALARM_DECODING".GLOBAL_ALARMS_MACHINE.WARNING_DECODING := 0;
       "DB440_MACHINE_ALARM_DECODING".ALARMS_CENTRAL.WARNING := FALSE;
   END_IF;
END_REGION

REGION Network 23: OUTPUTS
   RUNG wire#powerrail
      Contact( "DB2101_LINE_CONTACTOR".STEP_1_CONTACTOR_ON )
      wire#w1
      Coil( "LINE_CONTACTOR_ON_1_Q" )
   END_RUNG
   RUNG wire#w1
      Coil( "LINE_CONTACTOR_ON_2_Q" )
   END_RUNG
   // the same network as SCL:
   "LINE_CONTACTOR_ON_1_Q" := "DB2101_LINE_CONTACTOR".STEP_1_CONTACTOR_ON;
   "LINE_CONTACTOR_ON_2_Q" := "DB2101_LINE_CONTACTOR".STEP_1_CONTACTOR_ON;
END_REGION
END_FUNCTION

FUNCTION "FC2102_INFEED_MODULE" : Void   // FC2102, LAD
{ S7_Optimized_Access := 'FALSE' }
AUTHOR : ETXETAR
VERSION : 1.0
// stored: AutoNumber false, IsIECCheckEnabled false, SetENOAutomatically false, UDAEnableTagReadback false
   VAR_TEMP
      O_BYTE_0 : Struct   // OPTIONS BYTE 0
         POWER_SUPPLY_2 : Bool;   // POWER SUPPLY 2 OPTION
      END_STRUCT;
   END_VAR
   VAR CONSTANT
      FC_NUMBER : DInt := 2102;
   END_VAR
   VAR_TEMP   // added for the SCL form of the ladder/FBD networks
      _w1 : Bool;
   END_VAR
BEGIN

REGION Network 1: OPTIONS OFF
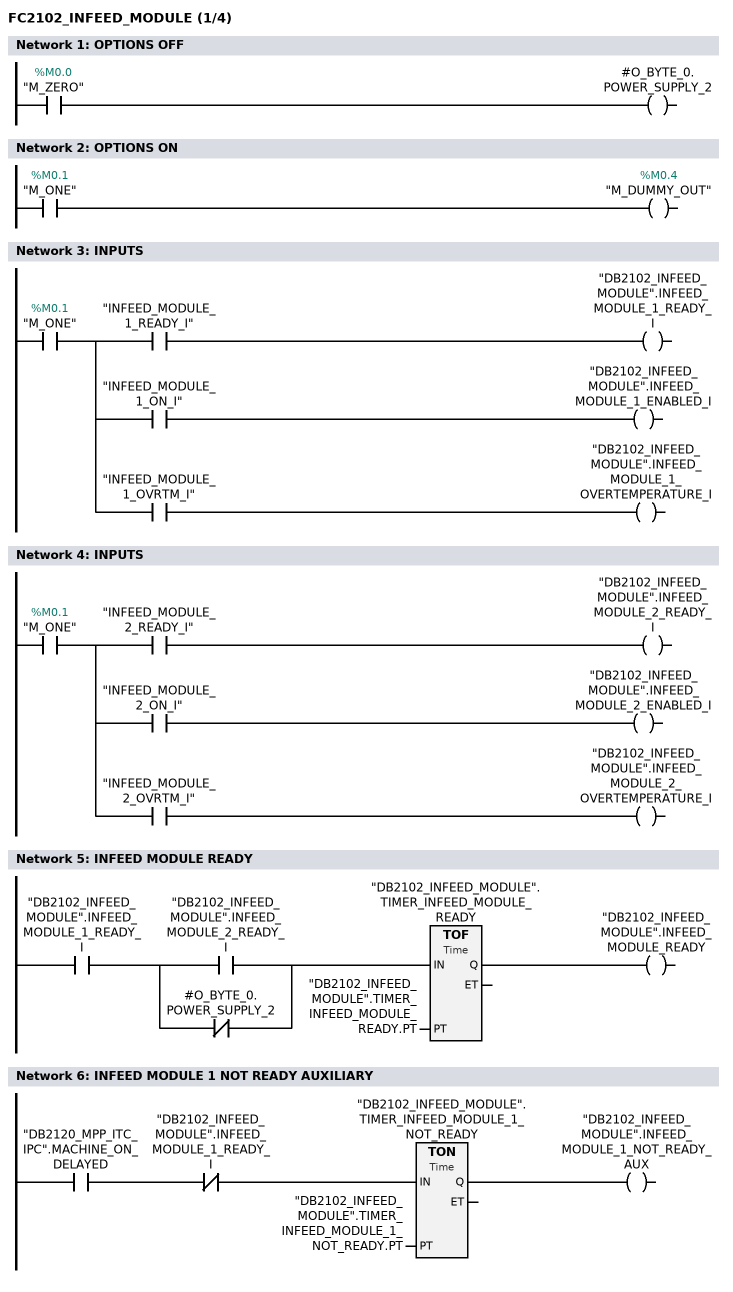
   RUNG wire#powerrail
      Contact( "M_ZERO" )
      Coil( #O_BYTE_0.POWER_SUPPLY_2 )
   END_RUNG
   // the same network as SCL:
   #O_BYTE_0.POWER_SUPPLY_2 := "M_ZERO";
END_REGION

REGION Network 2: OPTIONS ON
   RUNG wire#powerrail
      Contact( "M_ONE" )
      Coil( "M_DUMMY_OUT" )
   END_RUNG
   // the same network as SCL:
   "M_DUMMY_OUT" := "M_ONE";
END_REGION

REGION Network 3: INPUTS
   RUNG wire#powerrail
      Contact( "M_ONE" )
      wire#w1
      Contact( "INFEED_MODULE_1_READY_I" )
      Coil( "DB2102_INFEED_MODULE".INFEED_MODULE_1_READY_I )
   END_RUNG
   RUNG wire#w1
      Contact( "INFEED_MODULE_1_ON_I" )
      Coil( "DB2102_INFEED_MODULE".INFEED_MODULE_1_ENABLED_I )
   END_RUNG
   RUNG wire#w1
      Contact( "INFEED_MODULE_1_OVRTM_I" )
      Coil( "DB2102_INFEED_MODULE".INFEED_MODULE_1_OVERTEMPERATURE_I )
   END_RUNG
   // the same network as SCL:
   "DB2102_INFEED_MODULE".INFEED_MODULE_1_READY_I := "M_ONE" AND "INFEED_MODULE_1_READY_I";
   "DB2102_INFEED_MODULE".INFEED_MODULE_1_ENABLED_I := "M_ONE" AND "INFEED_MODULE_1_ON_I";
   "DB2102_INFEED_MODULE".INFEED_MODULE_1_OVERTEMPERATURE_I := "M_ONE" AND "INFEED_MODULE_1_OVRTM_I";
END_REGION

REGION Network 4: INPUTS
   RUNG wire#powerrail
      Contact( "M_ONE" )
      wire#w1
      Contact( "INFEED_MODULE_2_READY_I" )
      Coil( "DB2102_INFEED_MODULE".INFEED_MODULE_2_READY_I )
   END_RUNG
   RUNG wire#w1
      Contact( "INFEED_MODULE_2_ON_I" )
      Coil( "DB2102_INFEED_MODULE".INFEED_MODULE_2_ENABLED_I )
   END_RUNG
   RUNG wire#w1
      Contact( "INFEED_MODULE_2_OVRTM_I" )
      Coil( "DB2102_INFEED_MODULE".INFEED_MODULE_2_OVERTEMPERATURE_I )
   END_RUNG
   // the same network as SCL:
   "DB2102_INFEED_MODULE".INFEED_MODULE_2_READY_I := "M_ONE" AND "INFEED_MODULE_2_READY_I";
   "DB2102_INFEED_MODULE".INFEED_MODULE_2_ENABLED_I := "M_ONE" AND "INFEED_MODULE_2_ON_I";
   "DB2102_INFEED_MODULE".INFEED_MODULE_2_OVERTEMPERATURE_I := "M_ONE" AND "INFEED_MODULE_2_OVRTM_I";
END_REGION

REGION Network 5: INFEED MODULE READY
   RUNG wire#powerrail
      Contact( "DB2102_INFEED_MODULE".INFEED_MODULE_1_READY_I )
      wire#w1
      Contact( "DB2102_INFEED_MODULE".INFEED_MODULE_2_READY_I )
      wire#w2
      { S7_Templates := "time_type := Time" } "DB2102_INFEED_MODULE".TIMER_INFEED_MODULE_READY.TOF(pt := "DB2102_INFEED_MODULE".TIMER_INFEED_MODULE_READY.PT, et =>)
      Coil( "DB2102_INFEED_MODULE".INFEED_MODULE_READY )
   END_RUNG
   RUNG wire#w1
      I_Contact( #O_BYTE_0.POWER_SUPPLY_2 )
   END_RUNG wire#w2
   // the same network as SCL:
   "DB2102_INFEED_MODULE".TIMER_INFEED_MODULE_READY.TOF(IN := "DB2102_INFEED_MODULE".INFEED_MODULE_1_READY_I AND ("DB2102_INFEED_MODULE".INFEED_MODULE_2_READY_I OR NOT #O_BYTE_0.POWER_SUPPLY_2),
                           PT := "DB2102_INFEED_MODULE".TIMER_INFEED_MODULE_READY.PT);
   "DB2102_INFEED_MODULE".INFEED_MODULE_READY := "DB2102_INFEED_MODULE".TIMER_INFEED_MODULE_READY.Q;
END_REGION

REGION Network 6: INFEED MODULE 1 NOT READY AUXILIARY
   RUNG wire#powerrail
      Contact( "DB2120_MPP_ITC_IPC".MACHINE_ON_DELAYED )
      I_Contact( "DB2102_INFEED_MODULE".INFEED_MODULE_1_READY_I )
      { S7_Templates := "time_type := Time" } "DB2102_INFEED_MODULE".TIMER_INFEED_MODULE_1_NOT_READY.TON(pt := "DB2102_INFEED_MODULE".TIMER_INFEED_MODULE_1_NOT_READY.PT, et =>)
      Coil( "DB2102_INFEED_MODULE".INFEED_MODULE_1_NOT_READY_AUX )
   END_RUNG
   // the same network as SCL:
   "DB2102_INFEED_MODULE".TIMER_INFEED_MODULE_1_NOT_READY.TON(IN := "DB2120_MPP_ITC_IPC".MACHINE_ON_DELAYED AND NOT "DB2102_INFEED_MODULE".INFEED_MODULE_1_READY_I,
                           PT := "DB2102_INFEED_MODULE".TIMER_INFEED_MODULE_1_NOT_READY.PT);
   "DB2102_INFEED_MODULE".INFEED_MODULE_1_NOT_READY_AUX := "DB2102_INFEED_MODULE".TIMER_INFEED_MODULE_1_NOT_READY.Q;
END_REGION

REGION Network 7: INFEED MODULE 1 NOT READY ALARM
